// TIA Portal V20 export
// export: Created 2025-12-01T14:56:38.9745421Z, ExportSetting None, DisplayName Totally Integrated Automation Portal, DisplayVersion V20 Update 3, DisplayName TIA Portal Openness, DisplayVersion V20 Update 3, DisplayName TIA Portal Version Control Interface, DisplayVersion V20 Update 3, DisplayName STEP 7 Professional, DisplayVersion V20 Update 3, DisplayName STEP 7 Safety, DisplayVersion V20 Update 2, DisplayName WinCC Basic/Comfort/Advanced, DisplayVersion V20 Update 3, DisplayName WinCC Professional, DisplayVersion V20 Update 3, DisplayName WinCC Unified, DisplayVersion V20 Update 3
FUNCTION_BLOCK "FB41_Mesa_ApiladorDesApilador_E0E1E3_S0S1S3"   // FB41, LAD
TITLE = Control del Ramal de Salidas
{ S7_Optimized_Access := 'FALSE' }
AUTHOR : MESA_MAQ
NAME : 20160509
VERSION : 3.6
// stored: AutoNumber false, SetENOAutomatically false
   VAR_INPUT
      Mesa : UInt;   // Mesa de la FB
      Error_Tx : Bool;   // Error en el Tx
      EnTension : Bool;   // Existe Tension en la Mesa
      Termico_Tx : Bool;   // Proteccion del Tx
      pHsMx_Carretilla : Bool;   // Detector de Carretilla Presente
      pHsMx_1 : Bool;   // pHs de la Mesa (Para Entrada por E3)
      pHsMx_2 : Bool;   // pHs de la Mesa (Para Entrada por E1)
      pHsMx_PR1 : Bool;   // pHs de Protrusion de la Mesa. Nota: No existe >> ON
      pHsMx_PR3 : Bool;   // pHs de Protrusion de la Mesa. Nota: No existe >> ON
      Avance_Tx : Bool;   // Avance del Tx
      Retroceso_Tx : Bool;   // Retroceso del Tx
      TP1_Up : Bool;   // TP1 Arriba. Nota Movimiento E1 >> S3
      TP1_Down : Bool;   // TP1 Abajo. Nota Movimiento E1 >> S3
      EnMovimiento_TP1 : Bool;   // En movimiento el TP1
      MAnt_DescargaAct : Bool;   // E1 >> Mesa Anterior DescargaAct
      AVTF_MAnt_Mx : Bool;   // E1 >> Mesa Anterior AVTF
      P_Mens_MAnt_Mx : Bool;   // E1 >> Mesa Anterior P_Mens
      MAnt_ExistePila : Bool;   // E1 >> Mesa Anterior Existe Pila
      MSig_DescargaAct : Bool;   // E3 >> Mesa Anterior DescargaAct
      AVTF_MSig_Mx : Bool;   // E3 >> Mesa Anterior AVTF
      P_Mens_MSig_Mx : Bool;   // E3 >> Mesa Anterior P_Mens
      MSig_ExistePila : Bool;   // E3 >> Mesa Anterior Existe Pila
      PTF_Mx_MSig : Bool;   // S1 >> Mesa Siguiente PTF
      FTF_Mx_MSig : Bool;   // S1 >> Mesa Siguiente FTF
      PTF_Mx_MAnt : Bool;   // S3 >> Mesa Siguiente PTF
      FTF_Mx_MAnt : Bool;   // S3 >> Mesa Siguiente FTF
      MAnt_CargaAct : Bool;
      MSig_CargaAct : Bool;
      ConCarga_Apilador : Bool;   // Existe Carga >>> Interlock Maquina
      Quieto_Apilador : Bool;   // Quieto >>> Interlock Maquina
      Lleno_Apilador : Bool;   // Lleno >>> Interlock Maquina
      FinMovimiento_Apilador : Bool;   // Fin Movimiento >>> Interlock Maquina
      Mx_VelocidadLenta_In : Bool;   // Forzar a Velociada Lenta
      Mx_Centraje : Bool;   // Config Mx >>> Centrar la Entrada
      F_ENV_MENS_Mx : Bool;   // Fin de Envio de Mensaje
      OrdSal_Pila_Mx_MAnt : Bool;   // Orden de Salida por S1 >> Pila
      OrdSal_Paleta_Mx_MAnt : Bool;   // Orden de Salida por S1 >> Paleta
      OrdSal_Pila_Mx_MSig : Bool;   // Orden de Salida por S3 >> Pila
      OrdSal_Paleta_Mx_MSig : Bool;   // Orden de Salida por S3 >> Paleta
      OrdSal_S00 : Bool;   // Orden de Salida por S0
      V_CNT_pHsMx : Int := 1000;   // Valor de Presencia
      V_CNT_pHsMx_FTF : Int := 200;   // Valor para activar FTF. Nota: < = V_CNT_pHsMx.
      V_CNTSeg_pHsMx : Int := 2000;   // Valor de Seguriadad para Presencia
      V_Subir_TP_Min : Int := 2000;   // Valor Minimo para Subir Tope
      V_Bajar_TP_Max : Int := 4000;   // Valor Maximo para Bajar Tope
      V_CNT_PasoLenta : Int := 2000;   // Valor de Paso a Lenta
      V_CNT_ApHsMx : Int := 500;   // Valor de Ausencia
      V_CNTSeg_ApHsMx : Int := 2000;   // Valor de Seguriadad para Ausencia
      V_TMP_Entrada : Int := 5000;   // Valor de Entrada de Carga >> E0
      V_TMP_Retirar : Int := 5000;   // Valor de Retirada de Carga >> S0
      V_CNT_Centrado : Int := 1000;   // Valor de Centrado de Carga
      V_CNT_Reposo : Int := 1500;   // Valor de Reposo de Carga Nota: > Centrado
      V_TOut_Tx_Mx : Int := 30000;   // TimeOut de Entrada por E1
      V_TOut_TP { ExternalWritable := 'False'} : Int := 5000;   // TimeOut de Tope
      V_TMP_Protrusion : Int := 200;   // TMP de Protrusion
      V_CNT_PerdidapHs : Int := 1000;   // CNT de Perdida de pHs
   END_VAR
   VAR_OUTPUT
      P_EnvMens_PMx : Bool;   // Permiso de Enviar Mensaje de Presencia
      P_EnvMens_AMx : Bool;   // Permiso de Enviar Mensaje de Ausencia
      P_RecepOK_Mx : Bool;   // Recepcion OK
      PTF_MAnt_Mx : Bool;   // E1 >> Mesa Anterior PTF
      FTF_MAnt_Mx : Bool;   // E1 >> Mesa Anterior FTF
      PTF_MSig_Mx : Bool;   // E3 >> Mesa Anterior PTF
      FTF_MSig_Mx : Bool;   // E3 >> Mesa Anterior FTF
      AVTF_Mx_MAnt : Bool;   // S1 >> Mesa Siguiente AVTF
      P_Mens_Mx_MAnt : Bool;   // S1 >> Mesa Siguiente P_Mens
      AVTF_Mx_MSig : Bool;   // S3 >> Mesa Siguiente AVTF
      P_Mens_Mx_MSig : Bool;   // S3 >> Mesa Siguiente P_Mens
      PasarReposo_Apilador : Bool;   // Pasar a Reposo >>> Interlock Maquina
      CogerPila_Apilador : Bool;   // Coger la Pila >>> Interlock Maquina
      DispensarPaleta_Apilador : Bool;   // Dispensar Paleta >>> Interlock Maquina
      DispensarpPila_Apilador : Bool;   // Dispensar Pila >>> Interlock Maquina
   END_VAR
   VAR_IN_OUT
      StatusLleno_Apilador : Bool;   // Status Lleno >>> Interlock Maquina
      StatusSemiLleno_Apilador : Bool;   // Status SemiLleno >>> Interlock Maquina
      StatusVacio_Apilador : Bool;   // Status Vacio >>> Interlock Maquina
   END_VAR
   VAR
      Anular_prE1 : Bool;   // ???
      Anular_prS3 : Bool;   // ???
      Mx_ET00 : Bool;
      Mx_ET01 : Bool;
      Mx_ET02 : Bool;
      Mx_ET08 : Bool;
      Mx_ET09 : Bool;
      Mx_ET10 : Bool;
      Mx_ET11 : Bool;
      Mx_ET12 : Bool;
      Mx_ET110 : Bool;
      Mx_ET111 : Bool;
      Mx_ET210 : Bool;
      Mx_ET211 : Bool;
      Mx_ET40 : Bool;
      Mx_ET41 : Bool;
      Mx_ET42 : Bool;
      Mx_ET43 : Bool;
      Mx_ET140 : Bool;
      Mx_ET141 : Bool;
      Mx_ET50 : Bool;
      Mx_ET51 : Bool;
      Mx_ET52 : Bool;
      Mx_ET53 : Bool;
      Mx_ET150 : Bool;
      Mx_ET151 : Bool;
      Mx_ET250 : Bool;
      Mx_ET251 : Bool;
      Mx_ET90 : Bool;
      Mx_ET91 : Bool;
      Mx_ET190 : Bool;
      Mx_ET191 : Bool;
      Mx_ET192 : Bool;
      ProtocoloIniciado : Bool;   // Iniciado el Envio del Mensaje de Presencia
      CNT_pHsMx_FTF_OK : Bool;   // Enviar ya FTF
      Memoria_EnReposoMaquina : Bool;   // Memoria >> Maquina en Reposo
      Carga_MAnt_Mx : Bool;   // Operacion de Carga MAnt >>> Mx
      Carga_MSig_Mx : Bool;   // Operacion de Carga MSig >>> Mx
      Descarga_Mx_MAnt : Bool;   // Operacion de DesCarga Mx >>> MAnt
      Descarga_Mx_MSig : Bool;   // Operacion de DesCarga Ms >>> MSig
      ActivaDesCarga_Mx_MAnt : Bool;
      ActivaDesCarga_Mx_MSig : Bool;
      STAT_EnvMens_PMx : Bool;   // Interna >> Envio del Mensaje de Presencia
      STAT_EnvMens_AMx : Bool;   // Interna >> Envio de Mensaje de Ausencia
      STAT_FTF_MAnt_Mx : Bool;   // Interna >> FTF de MAnt >> Mx
      STAT_FTF_MSig_Mx : Bool;   // Interna >> FTF de MSig >> Mx
      STAT_AVTF_Mx_MAnt : Bool;   // Interna >> AVTF de Mx >> MAnt
      STAT_AVTF_Mx_MSig : Bool;   // Interna >> AVTF de Mx >> MSig
      STAT_PasarReposo : Bool;   // Interna >> Pasar a Reposo >> Maquina
      STAT_CogerPila : Bool;   // Interna >> Coger la Pila >> Maquina
      STAT_DispensarPaleta : Bool;   // Interna >> Dispensar Paleta >> Maquina
      STAT_DispensarPila : Bool;   // Interna >> Dispensar Pila >> Maquina
      CNT_pHsMx { S7_SetPoint := 'True'} : "FB910_CNT_UHS";   // CNT de la Presencia
      CNTSeg_pHsMx { S7_SetPoint := 'True'} : "FB910_CNT_UHS";   // CNT de Seguridad de la Presencia
      CNT_ApHsMx { S7_SetPoint := 'True'} : "FB910_CNT_UHS";   // CNT de la Ausencia
      CNTSeg_ApHsMx { S7_SetPoint := 'True'} : "FB910_CNT_UHS";   // CNT de Seguridad de la Ausencia
      TMP_Entrada { S7_SetPoint := 'True'} : "FB910_CNT_UHS";   // TMP de Entrada de Carga
      TMP_Retirar { S7_SetPoint := 'True'} : "FB910_CNT_UHS";   // TMP de Retirada de Carga
      CNT_Centrado { S7_SetPoint := 'True'} : "FB910_CNT_UHS";   // Contador de Centrado de Carga
      TMP_EnTension { S7_SetPoint := 'True'} : "FB910_CNT_UHS";
      TOut_Av_Mx { S7_SetPoint := 'True'} : "FB910_CNT_UHS";   // Time Out de Entrada de E1
      TOut_Rt_Mx { S7_SetPoint := 'True'} : "FB910_CNT_UHS";   // Time Out de Entrada de E3
      TOut_Subir_TP { S7_SetPoint := 'True'} : "FB910_CNT_UHS";   // Time Out de Subida del TP
      TOut_Bajar_TP { S7_SetPoint := 'True'} : "FB910_CNT_UHS";   // Time Out de Bajada del TP
      TMP_Protrusion { S7_SetPoint := 'True'} : "FB910_CNT_UHS";   // TMP de la Protrusion
      CNT_PerdidapHs { S7_SetPoint := 'True'} : "FB910_CNT_UHS";   // CNT de Perdida de pHs
   END_VAR
   VAR_TEMP
      EstadoZona : "EstadoZona";   // Estado de Zona de la Mesa
      EstadoVI : "EstadosMesa";   // Estado del Vehiculo Inteliguente de la Mesa
      ConfigFB : "UDT_ConfigFB";   // Configuracion de la FB de la Mesa
      V_Protrusion : Int;
      Mx_SinPresenciaEnReset : Bool;
      Aux_ET00 : Bool;
   END_VAR
   VAR_TEMP   // added for the SCL form of the ladder/FBD networks
      _w1 : Bool;
      _w2 : Bool;
   END_VAR
BEGIN

REGION Network 1: Inicializaciones Especiales
   // Nota: En esta mesa no se envia presencia en el reset  >>>    #Mx_SinPresenciaEnReset
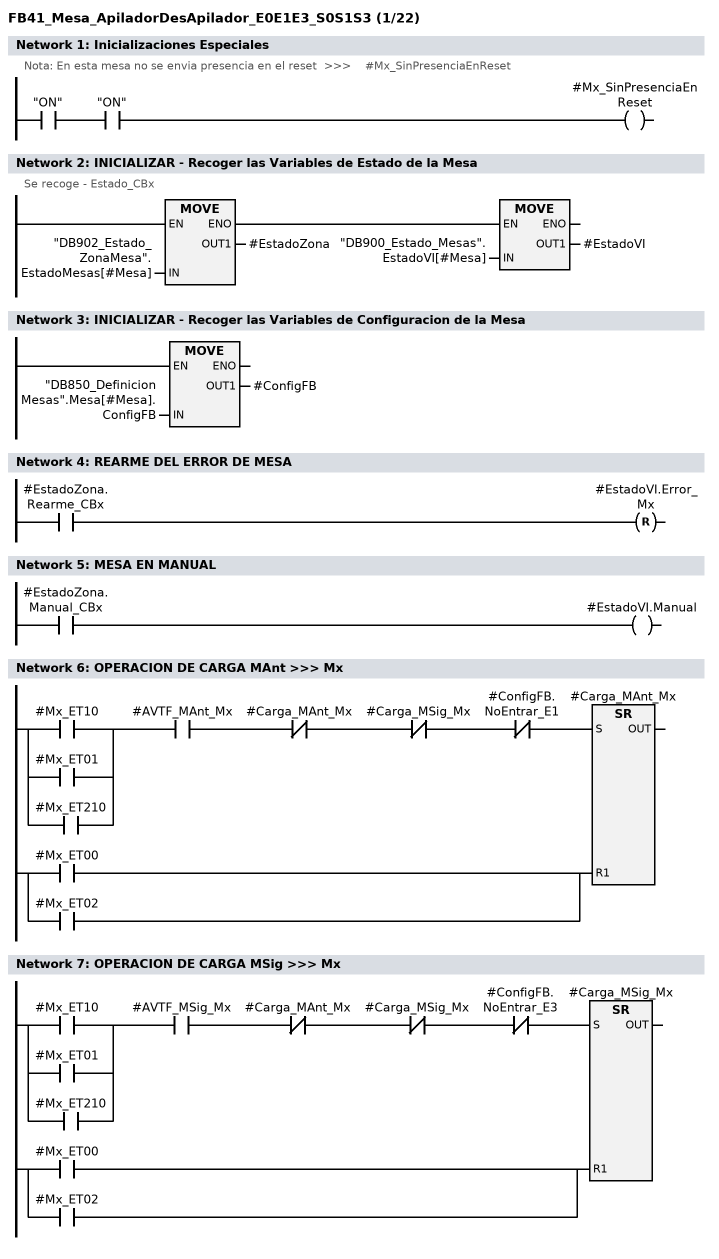
   RUNG wire#powerrail
      Contact( "ON" )
      Contact( "ON" )
      Coil( #Mx_SinPresenciaEnReset )
   END_RUNG
   // the same network as SCL:
   #Mx_SinPresenciaEnReset := "ON" AND "ON";
END_REGION

REGION Network 2: INICIALIZAR - Recoger las Variables de Estado de la Mesa
   // Se recoge - Estado_CBx
   RUNG wire#powerrail
      Move(in := "DB902_Estado_ZonaMesa".EstadoMesas[#Mesa], out1 => #EstadoZona)
      Move(in := "DB900_Estado_Mesas".EstadoVI[#Mesa], out1 => #EstadoVI)
   END_RUNG
   // the same network as SCL:
   #EstadoZona := "DB902_Estado_ZonaMesa".EstadoMesas[#Mesa];
   #EstadoVI := "DB900_Estado_Mesas".EstadoVI[#Mesa];
END_REGION

REGION Network 3: INICIALIZAR - Recoger las Variables de Configuracion de la Mesa
   RUNG wire#powerrail
      Move(in := "DB850_DefinicionMesas".Mesa[#Mesa].ConfigFB, out1 => #ConfigFB)
   END_RUNG
   // the same network as SCL:
   #ConfigFB := "DB850_DefinicionMesas".Mesa[#Mesa].ConfigFB;
END_REGION

REGION Network 4: REARME DEL ERROR DE MESA
   RUNG wire#powerrail
      Contact( #EstadoZona.Rearme_CBx )
      R_Coil( #EstadoVI.Error_Mx )
   END_RUNG
   // the same network as SCL:
   IF #EstadoZona.Rearme_CBx THEN #EstadoVI.Error_Mx := FALSE; END_IF;
END_REGION

REGION Network 5: MESA EN MANUAL
   RUNG wire#powerrail
      Contact( #EstadoZona.Manual_CBx )
      Coil( #EstadoVI.Manual )
   END_RUNG
   // the same network as SCL:
   #EstadoVI.Manual := #EstadoZona.Manual_CBx;
END_REGION

REGION Network 6: OPERACION DE CARGA MAnt >>> Mx
   RUNG wire#powerrail
      Contact( #Mx_ET10 )
      wire#w1
      Contact( #AVTF_MAnt_Mx )
      I_Contact( #Carga_MAnt_Mx )
      I_Contact( #Carga_MSig_Mx )
      I_Contact( #ConfigFB.NoEntrar_E1 )
      S_SR(operand := #Carga_MAnt_Mx, r1 := wire#w2)
   END_RUNG
   RUNG wire#powerrail
      Contact( #Mx_ET01 )
   END_RUNG wire#w1
   RUNG wire#powerrail
      Contact( #Mx_ET210 )
   END_RUNG wire#w1
   RUNG wire#powerrail
      Contact( #Mx_ET00 )
   END_RUNG wire#w2
   RUNG wire#powerrail
      Contact( #Mx_ET02 )
   END_RUNG wire#w2
   // the same network as SCL:
   IF (#Mx_ET10 OR #Mx_ET01 OR #Mx_ET210) AND #AVTF_MAnt_Mx AND NOT #Carga_MAnt_Mx AND NOT #Carga_MSig_Mx AND NOT #ConfigFB.NoEntrar_E1 THEN
       #Carga_MAnt_Mx := TRUE;   // SR flip-flop
   END_IF;
   IF #Mx_ET00 OR #Mx_ET02 THEN #Carga_MAnt_Mx := FALSE; END_IF;
END_REGION

REGION Network 7: OPERACION DE CARGA MSig >>> Mx
   RUNG wire#powerrail
      Contact( #Mx_ET10 )
      wire#w1
      Contact( #AVTF_MSig_Mx )
      I_Contact( #Carga_MAnt_Mx )
      I_Contact( #Carga_MSig_Mx )
      I_Contact( #ConfigFB.NoEntrar_E3 )
      S_SR(operand := #Carga_MSig_Mx, r1 := wire#w2)
   END_RUNG
   RUNG wire#powerrail
      Contact( #Mx_ET01 )
   END_RUNG wire#w1
   RUNG wire#powerrail
      Contact( #Mx_ET210 )
   END_RUNG wire#w1
   RUNG wire#powerrail
      Contact( #Mx_ET00 )
   END_RUNG wire#w2
   RUNG wire#powerrail
      Contact( #Mx_ET02 )
   END_RUNG wire#w2
   // the same network as SCL:
   IF (#Mx_ET10 OR #Mx_ET01 OR #Mx_ET210) AND #AVTF_MSig_Mx AND NOT #Carga_MAnt_Mx AND NOT #Carga_MSig_Mx AND NOT #ConfigFB.NoEntrar_E3 THEN
       #Carga_MSig_Mx := TRUE;   // SR flip-flop
   END_IF;
   IF #Mx_ET00 OR #Mx_ET02 THEN #Carga_MSig_Mx := FALSE; END_IF;
END_REGION

REGION Network 8: OPERACION DE DESCARGA Mx >>> MAnt
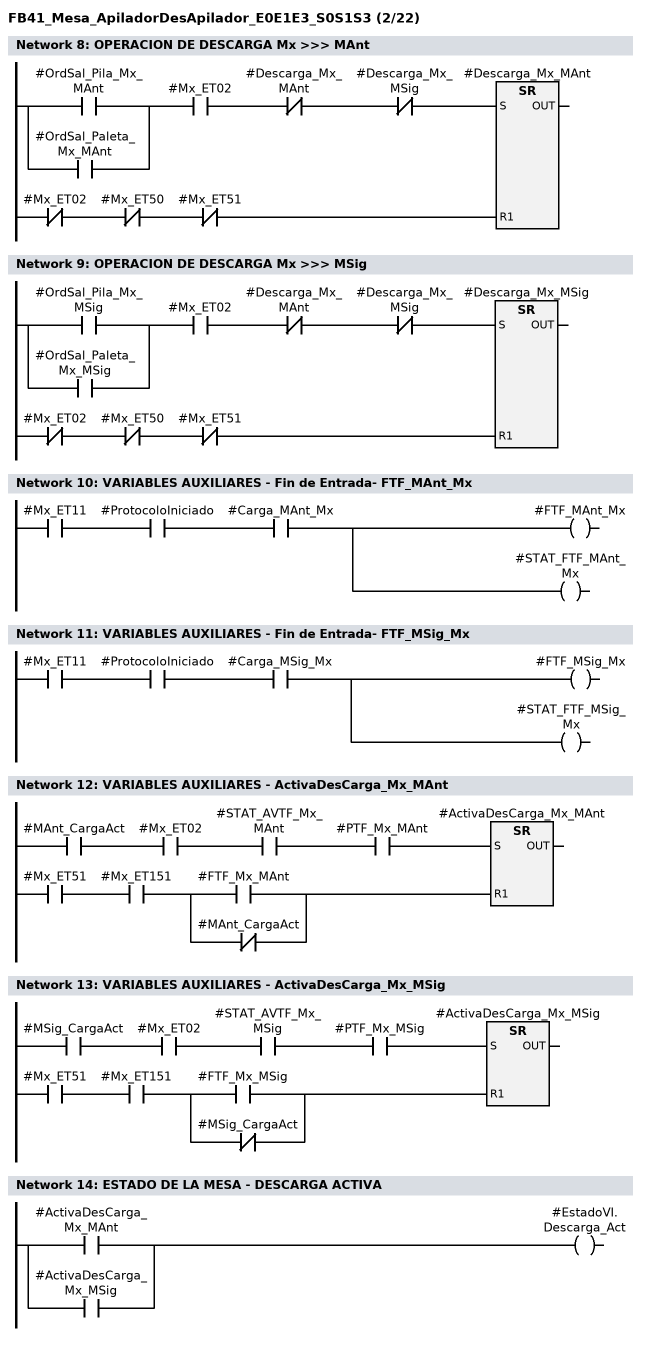
   RUNG wire#powerrail
      Contact( #OrdSal_Pila_Mx_MAnt )
      wire#w1
      Contact( #Mx_ET02 )
      I_Contact( #Descarga_Mx_MAnt )
      I_Contact( #Descarga_Mx_MSig )
      S_SR(operand := #Descarga_Mx_MAnt, r1 := wire#w2)
   END_RUNG
   RUNG wire#powerrail
      Contact( #OrdSal_Paleta_Mx_MAnt )
   END_RUNG wire#w1
   RUNG wire#powerrail
      I_Contact( #Mx_ET02 )
      I_Contact( #Mx_ET50 )
      I_Contact( #Mx_ET51 )
   END_RUNG wire#w2
   // the same network as SCL:
   IF (#OrdSal_Pila_Mx_MAnt OR #OrdSal_Paleta_Mx_MAnt) AND #Mx_ET02 AND NOT #Descarga_Mx_MAnt AND NOT #Descarga_Mx_MSig THEN
       #Descarga_Mx_MAnt := TRUE;   // SR flip-flop
   END_IF;
   IF NOT #Mx_ET02 AND NOT #Mx_ET50 AND NOT #Mx_ET51 THEN #Descarga_Mx_MAnt := FALSE; END_IF;
END_REGION

REGION Network 9: OPERACION DE DESCARGA Mx >>> MSig
   RUNG wire#powerrail
      Contact( #OrdSal_Pila_Mx_MSig )
      wire#w1
      Contact( #Mx_ET02 )
      I_Contact( #Descarga_Mx_MAnt )
      I_Contact( #Descarga_Mx_MSig )
      S_SR(operand := #Descarga_Mx_MSig, r1 := wire#w2)
   END_RUNG
   RUNG wire#powerrail
      Contact( #OrdSal_Paleta_Mx_MSig )
   END_RUNG wire#w1
   RUNG wire#powerrail
      I_Contact( #Mx_ET02 )
      I_Contact( #Mx_ET50 )
      I_Contact( #Mx_ET51 )
   END_RUNG wire#w2
   // the same network as SCL:
   IF (#OrdSal_Pila_Mx_MSig OR #OrdSal_Paleta_Mx_MSig) AND #Mx_ET02 AND NOT #Descarga_Mx_MAnt AND NOT #Descarga_Mx_MSig THEN
       #Descarga_Mx_MSig := TRUE;   // SR flip-flop
   END_IF;
   IF NOT #Mx_ET02 AND NOT #Mx_ET50 AND NOT #Mx_ET51 THEN #Descarga_Mx_MSig := FALSE; END_IF;
END_REGION

REGION Network 10: VARIABLES AUXILIARES - Fin de Entrada- FTF_MAnt_Mx
   RUNG wire#powerrail
      Contact( #Mx_ET11 )
      Contact( #ProtocoloIniciado )
      Contact( #Carga_MAnt_Mx )
      wire#w1
      Coil( #FTF_MAnt_Mx )
   END_RUNG
   RUNG wire#w1
      Coil( #STAT_FTF_MAnt_Mx )
   END_RUNG
   // the same network as SCL:
   #FTF_MAnt_Mx := #Mx_ET11 AND #ProtocoloIniciado AND #Carga_MAnt_Mx;
   #STAT_FTF_MAnt_Mx := #FTF_MAnt_Mx;
END_REGION

REGION Network 11: VARIABLES AUXILIARES - Fin de Entrada- FTF_MSig_Mx
   RUNG wire#powerrail
      Contact( #Mx_ET11 )
      Contact( #ProtocoloIniciado )
      Contact( #Carga_MSig_Mx )
      wire#w1
      Coil( #FTF_MSig_Mx )
   END_RUNG
   RUNG wire#w1
      Coil( #STAT_FTF_MSig_Mx )
   END_RUNG
   // the same network as SCL:
   #FTF_MSig_Mx := #Mx_ET11 AND #ProtocoloIniciado AND #Carga_MSig_Mx;
   #STAT_FTF_MSig_Mx := #FTF_MSig_Mx;
END_REGION

REGION Network 12: VARIABLES AUXILIARES - ActivaDesCarga_Mx_MAnt
   RUNG wire#powerrail
      Contact( #MAnt_CargaAct )
      Contact( #Mx_ET02 )
      Contact( #STAT_AVTF_Mx_MAnt )
      Contact( #PTF_Mx_MAnt )
      S_SR(operand := #ActivaDesCarga_Mx_MAnt, r1 := wire#w2)
   END_RUNG
   RUNG wire#powerrail
      Contact( #Mx_ET51 )
      Contact( #Mx_ET151 )
      wire#w1
      Contact( #FTF_Mx_MAnt )
   END_RUNG wire#w2
   RUNG wire#w1
      I_Contact( #MAnt_CargaAct )
   END_RUNG wire#w2
   // the same network as SCL:
   IF #MAnt_CargaAct AND #Mx_ET02 AND #STAT_AVTF_Mx_MAnt AND #PTF_Mx_MAnt THEN
       #ActivaDesCarga_Mx_MAnt := TRUE;   // SR flip-flop
   END_IF;
   IF #Mx_ET51 AND #Mx_ET151 AND (#FTF_Mx_MAnt OR NOT #MAnt_CargaAct) THEN
       #ActivaDesCarga_Mx_MAnt := FALSE;
   END_IF;
END_REGION

REGION Network 13: VARIABLES AUXILIARES - ActivaDesCarga_Mx_MSig
   RUNG wire#powerrail
      Contact( #MSig_CargaAct )
      Contact( #Mx_ET02 )
      Contact( #STAT_AVTF_Mx_MSig )
      Contact( #PTF_Mx_MSig )
      S_SR(operand := #ActivaDesCarga_Mx_MSig, r1 := wire#w2)
   END_RUNG
   RUNG wire#powerrail
      Contact( #Mx_ET51 )
      Contact( #Mx_ET151 )
      wire#w1
      Contact( #FTF_Mx_MSig )
   END_RUNG wire#w2
   RUNG wire#w1
      I_Contact( #MSig_CargaAct )
   END_RUNG wire#w2
   // the same network as SCL:
   IF #MSig_CargaAct AND #Mx_ET02 AND #STAT_AVTF_Mx_MSig AND #PTF_Mx_MSig THEN
       #ActivaDesCarga_Mx_MSig := TRUE;   // SR flip-flop
   END_IF;
   IF #Mx_ET51 AND #Mx_ET151 AND (#FTF_Mx_MSig OR NOT #MSig_CargaAct) THEN
       #ActivaDesCarga_Mx_MSig := FALSE;
   END_IF;
END_REGION

REGION Network 14: ESTADO DE LA MESA - DESCARGA ACTIVA
   RUNG wire#powerrail
      Contact( #ActivaDesCarga_Mx_MAnt )
      wire#w1
      Coil( #EstadoVI.Descarga_Act )
   END_RUNG
   RUNG wire#powerrail
      Contact( #ActivaDesCarga_Mx_MSig )
   END_RUNG wire#w1
   // the same network as SCL:
   #EstadoVI.Descarga_Act := #ActivaDesCarga_Mx_MAnt OR #ActivaDesCarga_Mx_MSig;
END_REGION

REGION Network 15: ET192 - CONTROL RETIRADA MESA - PROTOCOLO ORDEN
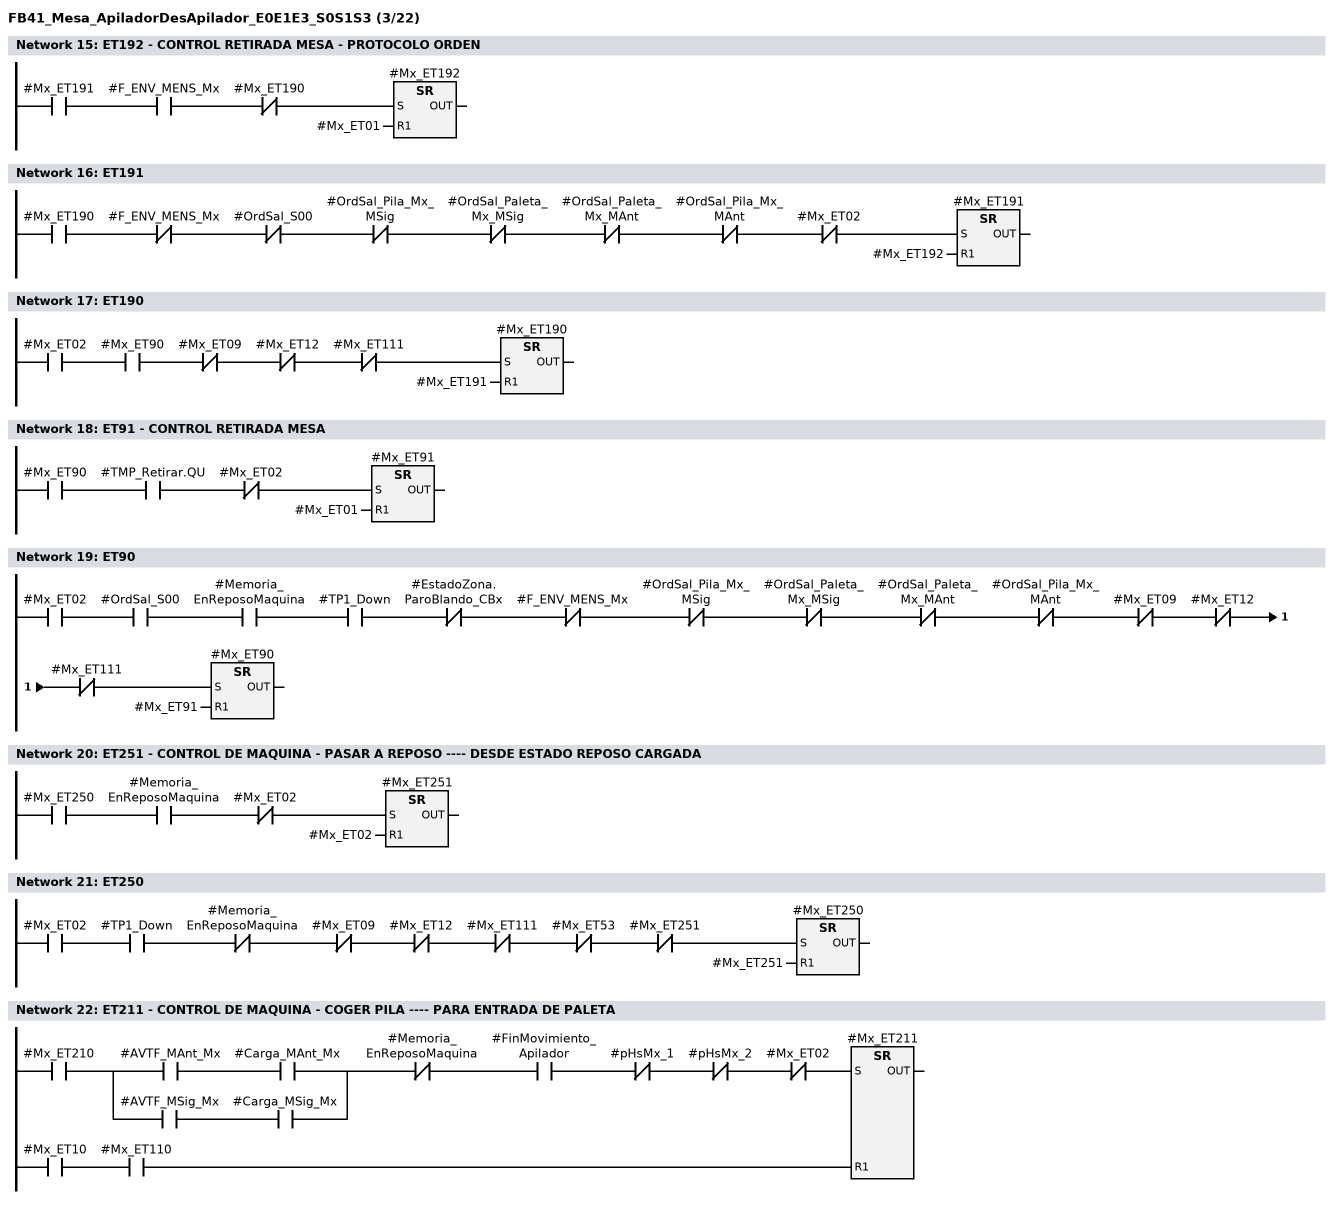
   RUNG wire#powerrail
      Contact( #Mx_ET191 )
      Contact( #F_ENV_MENS_Mx )
      I_Contact( #Mx_ET190 )
      S_SR(operand := #Mx_ET192, r1 := #Mx_ET01)
   END_RUNG
   // the same network as SCL:
   IF #Mx_ET191 AND #F_ENV_MENS_Mx AND NOT #Mx_ET190 THEN
       #Mx_ET192 := TRUE;   // SR flip-flop
   END_IF;
   IF #Mx_ET01 THEN #Mx_ET192 := FALSE; END_IF;
END_REGION

REGION Network 16: ET191
   RUNG wire#powerrail
      Contact( #Mx_ET190 )
      I_Contact( #F_ENV_MENS_Mx )
      I_Contact( #OrdSal_S00 )
      I_Contact( #OrdSal_Pila_Mx_MSig )
      I_Contact( #OrdSal_Paleta_Mx_MSig )
      I_Contact( #OrdSal_Paleta_Mx_MAnt )
      I_Contact( #OrdSal_Pila_Mx_MAnt )
      I_Contact( #Mx_ET02 )
      S_SR(operand := #Mx_ET191, r1 := #Mx_ET192)
   END_RUNG
   // the same network as SCL:
   IF #Mx_ET190 AND NOT #F_ENV_MENS_Mx AND NOT #OrdSal_S00 AND NOT #OrdSal_Pila_Mx_MSig AND NOT #OrdSal_Paleta_Mx_MSig AND NOT #OrdSal_Paleta_Mx_MAnt AND NOT #OrdSal_Pila_Mx_MAnt AND NOT #Mx_ET02 THEN
       #Mx_ET191 := TRUE;   // SR flip-flop
   END_IF;
   IF #Mx_ET192 THEN #Mx_ET191 := FALSE; END_IF;
END_REGION

REGION Network 17: ET190
   RUNG wire#powerrail
      Contact( #Mx_ET02 )
      Contact( #Mx_ET90 )
      I_Contact( #Mx_ET09 )
      I_Contact( #Mx_ET12 )
      I_Contact( #Mx_ET111 )
      S_SR(operand := #Mx_ET190, r1 := #Mx_ET191)
   END_RUNG
   // the same network as SCL:
   IF #Mx_ET02 AND #Mx_ET90 AND NOT #Mx_ET09 AND NOT #Mx_ET12 AND NOT #Mx_ET111 THEN
       #Mx_ET190 := TRUE;   // SR flip-flop
   END_IF;
   IF #Mx_ET191 THEN #Mx_ET190 := FALSE; END_IF;
END_REGION

REGION Network 18: ET91 - CONTROL RETIRADA MESA
   RUNG wire#powerrail
      Contact( #Mx_ET90 )
      Contact( #TMP_Retirar.QU )
      I_Contact( #Mx_ET02 )
      S_SR(operand := #Mx_ET91, r1 := #Mx_ET01)
   END_RUNG
   // the same network as SCL:
   IF #Mx_ET90 AND #TMP_Retirar.QU AND NOT #Mx_ET02 THEN
       #Mx_ET91 := TRUE;   // SR flip-flop
   END_IF;
   IF #Mx_ET01 THEN #Mx_ET91 := FALSE; END_IF;
END_REGION

REGION Network 19: ET90
   RUNG wire#powerrail
      Contact( #Mx_ET02 )
      Contact( #OrdSal_S00 )
      Contact( #Memoria_EnReposoMaquina )
      Contact( #TP1_Down )
      I_Contact( #EstadoZona.ParoBlando_CBx )
      I_Contact( #F_ENV_MENS_Mx )
      I_Contact( #OrdSal_Pila_Mx_MSig )
      I_Contact( #OrdSal_Paleta_Mx_MSig )
      I_Contact( #OrdSal_Paleta_Mx_MAnt )
      I_Contact( #OrdSal_Pila_Mx_MAnt )
      I_Contact( #Mx_ET09 )
      I_Contact( #Mx_ET12 )
      I_Contact( #Mx_ET111 )
      S_SR(operand := #Mx_ET90, r1 := #Mx_ET91)
   END_RUNG
   // the same network as SCL:
   IF #Mx_ET02 AND #OrdSal_S00 AND #Memoria_EnReposoMaquina AND #TP1_Down AND NOT #EstadoZona.ParoBlando_CBx AND NOT #F_ENV_MENS_Mx AND NOT #OrdSal_Pila_Mx_MSig AND NOT #OrdSal_Paleta_Mx_MSig AND NOT #OrdSal_Paleta_Mx_MAnt AND NOT #OrdSal_Pila_Mx_MAnt AND NOT #Mx_ET09 AND NOT #Mx_ET12 AND NOT #Mx_ET111 THEN
       #Mx_ET90 := TRUE;   // SR flip-flop
   END_IF;
   IF #Mx_ET91 THEN #Mx_ET90 := FALSE; END_IF;
END_REGION

REGION Network 20: ET251 - CONTROL DE MAQUINA - PASAR A REPOSO ---- DESDE ESTADO REPOSO CARGADA
   RUNG wire#powerrail
      Contact( #Mx_ET250 )
      Contact( #Memoria_EnReposoMaquina )
      I_Contact( #Mx_ET02 )
      S_SR(operand := #Mx_ET251, r1 := #Mx_ET02)
   END_RUNG
   // the same network as SCL:
   IF #Mx_ET250 AND #Memoria_EnReposoMaquina AND NOT #Mx_ET02 THEN
       #Mx_ET251 := TRUE;   // SR flip-flop
   END_IF;
   IF #Mx_ET02 THEN #Mx_ET251 := FALSE; END_IF;
END_REGION

REGION Network 21: ET250
   RUNG wire#powerrail
      Contact( #Mx_ET02 )
      Contact( #TP1_Down )
      I_Contact( #Memoria_EnReposoMaquina )
      I_Contact( #Mx_ET09 )
      I_Contact( #Mx_ET12 )
      I_Contact( #Mx_ET111 )
      I_Contact( #Mx_ET53 )
      I_Contact( #Mx_ET251 )
      S_SR(operand := #Mx_ET250, r1 := #Mx_ET251)
   END_RUNG
   // the same network as SCL:
   IF #Mx_ET02 AND #TP1_Down AND NOT #Memoria_EnReposoMaquina AND NOT #Mx_ET09 AND NOT #Mx_ET12 AND NOT #Mx_ET111 AND NOT #Mx_ET53 AND NOT #Mx_ET251 THEN
       #Mx_ET250 := TRUE;   // SR flip-flop
   END_IF;
   IF #Mx_ET251 THEN #Mx_ET250 := FALSE; END_IF;
END_REGION

REGION Network 22: ET211 - CONTROL DE MAQUINA - COGER PILA ---- PARA ENTRADA DE PALETA
   RUNG wire#powerrail
      Contact( #Mx_ET210 )
      wire#w1
      Contact( #AVTF_MAnt_Mx )
      Contact( #Carga_MAnt_Mx )
      wire#w2
      I_Contact( #Memoria_EnReposoMaquina )
      Contact( #FinMovimiento_Apilador )
      I_Contact( #pHsMx_1 )
      I_Contact( #pHsMx_2 )
      I_Contact( #Mx_ET02 )
      S_SR(operand := #Mx_ET211, r1 := wire#w3)
   END_RUNG
   RUNG wire#w1
      Contact( #AVTF_MSig_Mx )
      Contact( #Carga_MSig_Mx )
   END_RUNG wire#w2
   RUNG wire#powerrail
      Contact( #Mx_ET10 )
      Contact( #Mx_ET110 )
   END_RUNG wire#w3
   // the same network as SCL:
   IF #Mx_ET210 AND ((#AVTF_MAnt_Mx AND #Carga_MAnt_Mx) OR (#AVTF_MSig_Mx AND #Carga_MSig_Mx)) AND NOT #Memoria_EnReposoMaquina AND #FinMovimiento_Apilador AND NOT #pHsMx_1 AND NOT #pHsMx_2 AND NOT #Mx_ET02 THEN
       #Mx_ET211 := TRUE;   // SR flip-flop
   END_IF;
   IF #Mx_ET10 AND #Mx_ET110 THEN #Mx_ET211 := FALSE; END_IF;
END_REGION

REGION Network 23: ET210
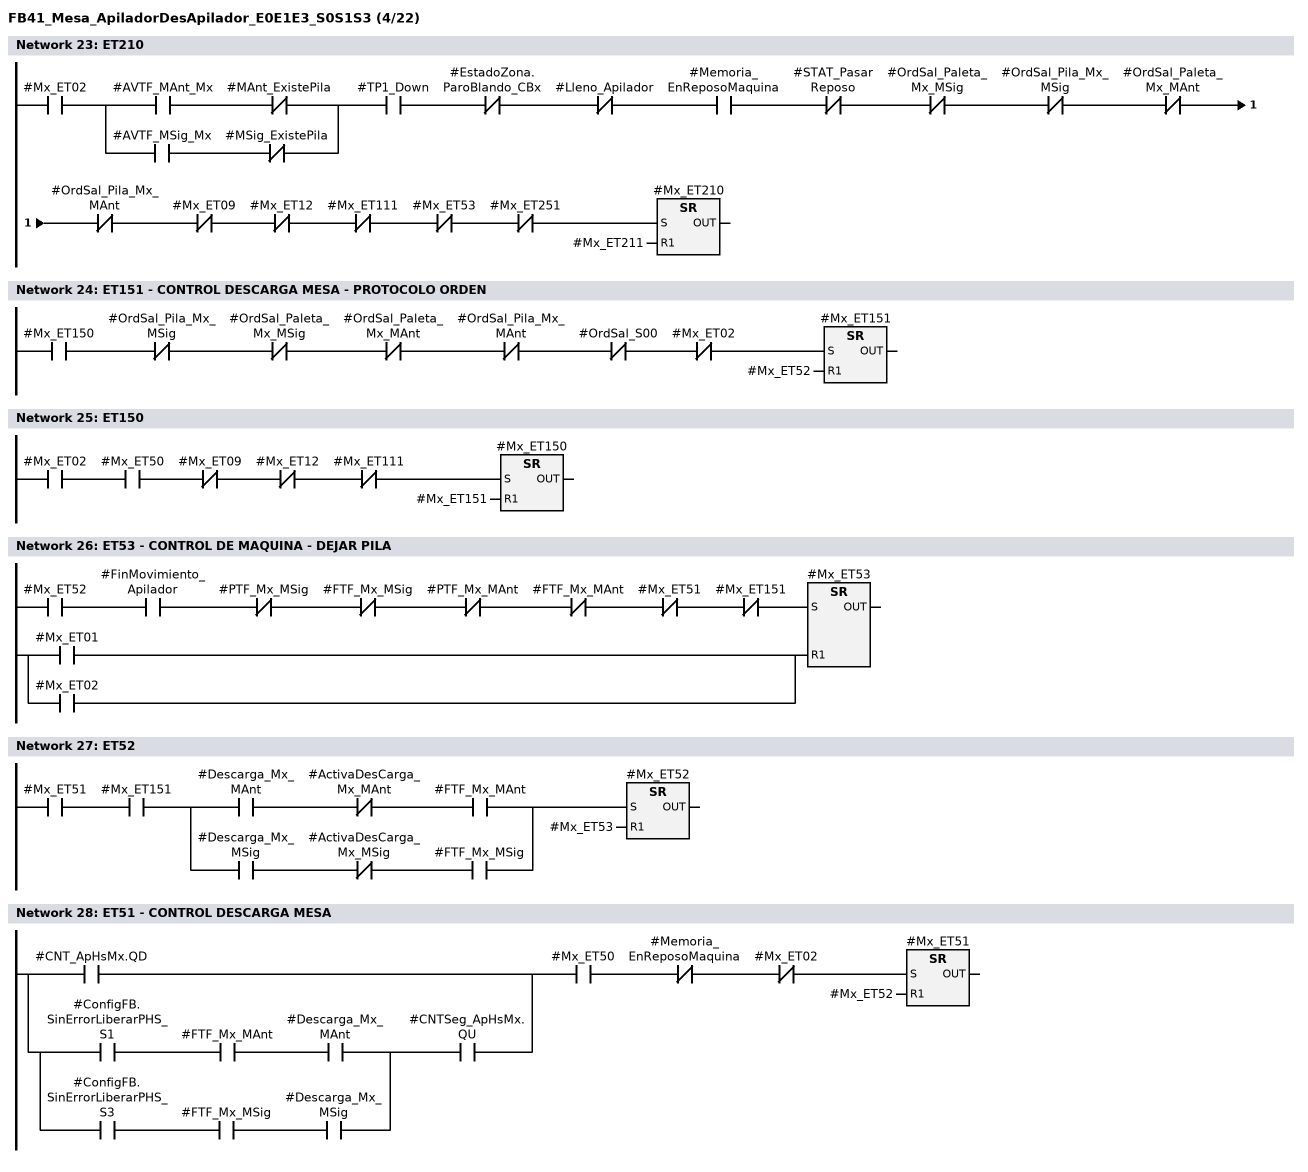
   RUNG wire#powerrail
      Contact( #Mx_ET02 )
      wire#w1
      Contact( #AVTF_MAnt_Mx )
      I_Contact( #MAnt_ExistePila )
      wire#w2
      Contact( #TP1_Down )
      I_Contact( #EstadoZona.ParoBlando_CBx )
      I_Contact( #Lleno_Apilador )
      Contact( #Memoria_EnReposoMaquina )
      I_Contact( #STAT_PasarReposo )
      I_Contact( #OrdSal_Paleta_Mx_MSig )
      I_Contact( #OrdSal_Pila_Mx_MSig )
      I_Contact( #OrdSal_Paleta_Mx_MAnt )
      I_Contact( #OrdSal_Pila_Mx_MAnt )
      I_Contact( #Mx_ET09 )
      I_Contact( #Mx_ET12 )
      I_Contact( #Mx_ET111 )
      I_Contact( #Mx_ET53 )
      I_Contact( #Mx_ET251 )
      S_SR(operand := #Mx_ET210, r1 := #Mx_ET211)
   END_RUNG
   RUNG wire#w1
      Contact( #AVTF_MSig_Mx )
      I_Contact( #MSig_ExistePila )
   END_RUNG wire#w2
   // the same network as SCL:
   IF #Mx_ET02 AND ((#AVTF_MAnt_Mx AND NOT #MAnt_ExistePila) OR (#AVTF_MSig_Mx AND NOT #MSig_ExistePila)) AND #TP1_Down AND NOT #EstadoZona.ParoBlando_CBx AND NOT #Lleno_Apilador AND #Memoria_EnReposoMaquina AND NOT #STAT_PasarReposo AND NOT #OrdSal_Paleta_Mx_MSig AND NOT #OrdSal_Pila_Mx_MSig AND NOT #OrdSal_Paleta_Mx_MAnt AND NOT #OrdSal_Pila_Mx_MAnt AND NOT #Mx_ET09 AND NOT #Mx_ET12 AND NOT #Mx_ET111 AND NOT #Mx_ET53 AND NOT #Mx_ET251 THEN
       #Mx_ET210 := TRUE;   // SR flip-flop
   END_IF;
   IF #Mx_ET211 THEN #Mx_ET210 := FALSE; END_IF;
END_REGION

REGION Network 24: ET151 - CONTROL DESCARGA MESA - PROTOCOLO ORDEN
   RUNG wire#powerrail
      Contact( #Mx_ET150 )
      I_Contact( #OrdSal_Pila_Mx_MSig )
      I_Contact( #OrdSal_Paleta_Mx_MSig )
      I_Contact( #OrdSal_Paleta_Mx_MAnt )
      I_Contact( #OrdSal_Pila_Mx_MAnt )
      I_Contact( #OrdSal_S00 )
      I_Contact( #Mx_ET02 )
      S_SR(operand := #Mx_ET151, r1 := #Mx_ET52)
   END_RUNG
   // the same network as SCL:
   IF #Mx_ET150 AND NOT #OrdSal_Pila_Mx_MSig AND NOT #OrdSal_Paleta_Mx_MSig AND NOT #OrdSal_Paleta_Mx_MAnt AND NOT #OrdSal_Pila_Mx_MAnt AND NOT #OrdSal_S00 AND NOT #Mx_ET02 THEN
       #Mx_ET151 := TRUE;   // SR flip-flop
   END_IF;
   IF #Mx_ET52 THEN #Mx_ET151 := FALSE; END_IF;
END_REGION

REGION Network 25: ET150
   RUNG wire#powerrail
      Contact( #Mx_ET02 )
      Contact( #Mx_ET50 )
      I_Contact( #Mx_ET09 )
      I_Contact( #Mx_ET12 )
      I_Contact( #Mx_ET111 )
      S_SR(operand := #Mx_ET150, r1 := #Mx_ET151)
   END_RUNG
   // the same network as SCL:
   IF #Mx_ET02 AND #Mx_ET50 AND NOT #Mx_ET09 AND NOT #Mx_ET12 AND NOT #Mx_ET111 THEN
       #Mx_ET150 := TRUE;   // SR flip-flop
   END_IF;
   IF #Mx_ET151 THEN #Mx_ET150 := FALSE; END_IF;
END_REGION

REGION Network 26: ET53 - CONTROL DE MAQUINA - DEJAR PILA
   RUNG wire#powerrail
      Contact( #Mx_ET52 )
      Contact( #FinMovimiento_Apilador )
      I_Contact( #PTF_Mx_MSig )
      I_Contact( #FTF_Mx_MSig )
      I_Contact( #PTF_Mx_MAnt )
      I_Contact( #FTF_Mx_MAnt )
      I_Contact( #Mx_ET51 )
      I_Contact( #Mx_ET151 )
      S_SR(operand := #Mx_ET53, r1 := wire#w1)
   END_RUNG
   RUNG wire#powerrail
      Contact( #Mx_ET01 )
   END_RUNG wire#w1
   RUNG wire#powerrail
      Contact( #Mx_ET02 )
   END_RUNG wire#w1
   // the same network as SCL:
   IF #Mx_ET52 AND #FinMovimiento_Apilador AND NOT #PTF_Mx_MSig AND NOT #FTF_Mx_MSig AND NOT #PTF_Mx_MAnt AND NOT #FTF_Mx_MAnt AND NOT #Mx_ET51 AND NOT #Mx_ET151 THEN
       #Mx_ET53 := TRUE;   // SR flip-flop
   END_IF;
   IF #Mx_ET01 OR #Mx_ET02 THEN #Mx_ET53 := FALSE; END_IF;
END_REGION

REGION Network 27: ET52
   RUNG wire#powerrail
      Contact( #Mx_ET51 )
      Contact( #Mx_ET151 )
      wire#w1
      Contact( #Descarga_Mx_MAnt )
      I_Contact( #ActivaDesCarga_Mx_MAnt )
      Contact( #FTF_Mx_MAnt )
      wire#w2
      S_SR(operand := #Mx_ET52, r1 := #Mx_ET53)
   END_RUNG
   RUNG wire#w1
      Contact( #Descarga_Mx_MSig )
      I_Contact( #ActivaDesCarga_Mx_MSig )
      Contact( #FTF_Mx_MSig )
   END_RUNG wire#w2
   // the same network as SCL:
   IF #Mx_ET51 AND #Mx_ET151 AND ((#Descarga_Mx_MAnt AND NOT #ActivaDesCarga_Mx_MAnt AND #FTF_Mx_MAnt) OR (#Descarga_Mx_MSig AND NOT #ActivaDesCarga_Mx_MSig AND #FTF_Mx_MSig)) THEN
       #Mx_ET52 := TRUE;   // SR flip-flop
   END_IF;
   IF #Mx_ET53 THEN #Mx_ET52 := FALSE; END_IF;
END_REGION

REGION Network 28: ET51 - CONTROL DESCARGA MESA
   RUNG wire#powerrail
      Contact( #CNT_ApHsMx.QD )
      wire#w1
      Contact( #Mx_ET50 )
      I_Contact( #Memoria_EnReposoMaquina )
      I_Contact( #Mx_ET02 )
      S_SR(operand := #Mx_ET51, r1 := #Mx_ET52)
   END_RUNG
   RUNG wire#powerrail
      Contact( #ConfigFB.SinErrorLiberarPHS_S1 )
      Contact( #FTF_Mx_MAnt )
      Contact( #Descarga_Mx_MAnt )
      wire#w2
      Contact( #CNTSeg_ApHsMx.QU )
   END_RUNG wire#w1
   RUNG wire#powerrail
      Contact( #ConfigFB.SinErrorLiberarPHS_S3 )
      Contact( #FTF_Mx_MSig )
      Contact( #Descarga_Mx_MSig )
   END_RUNG wire#w2
   // the same network as SCL:
   IF (#CNT_ApHsMx.QD OR (((#ConfigFB.SinErrorLiberarPHS_S1 AND #FTF_Mx_MAnt AND #Descarga_Mx_MAnt) OR (#ConfigFB.SinErrorLiberarPHS_S3 AND #FTF_Mx_MSig AND #Descarga_Mx_MSig)) AND #CNTSeg_ApHsMx.QU)) AND #Mx_ET50 AND NOT #Memoria_EnReposoMaquina AND NOT #Mx_ET02 THEN
       #Mx_ET51 := TRUE;   // SR flip-flop
   END_IF;
   IF #Mx_ET52 THEN #Mx_ET51 := FALSE; END_IF;
END_REGION

REGION Network 29: ET50
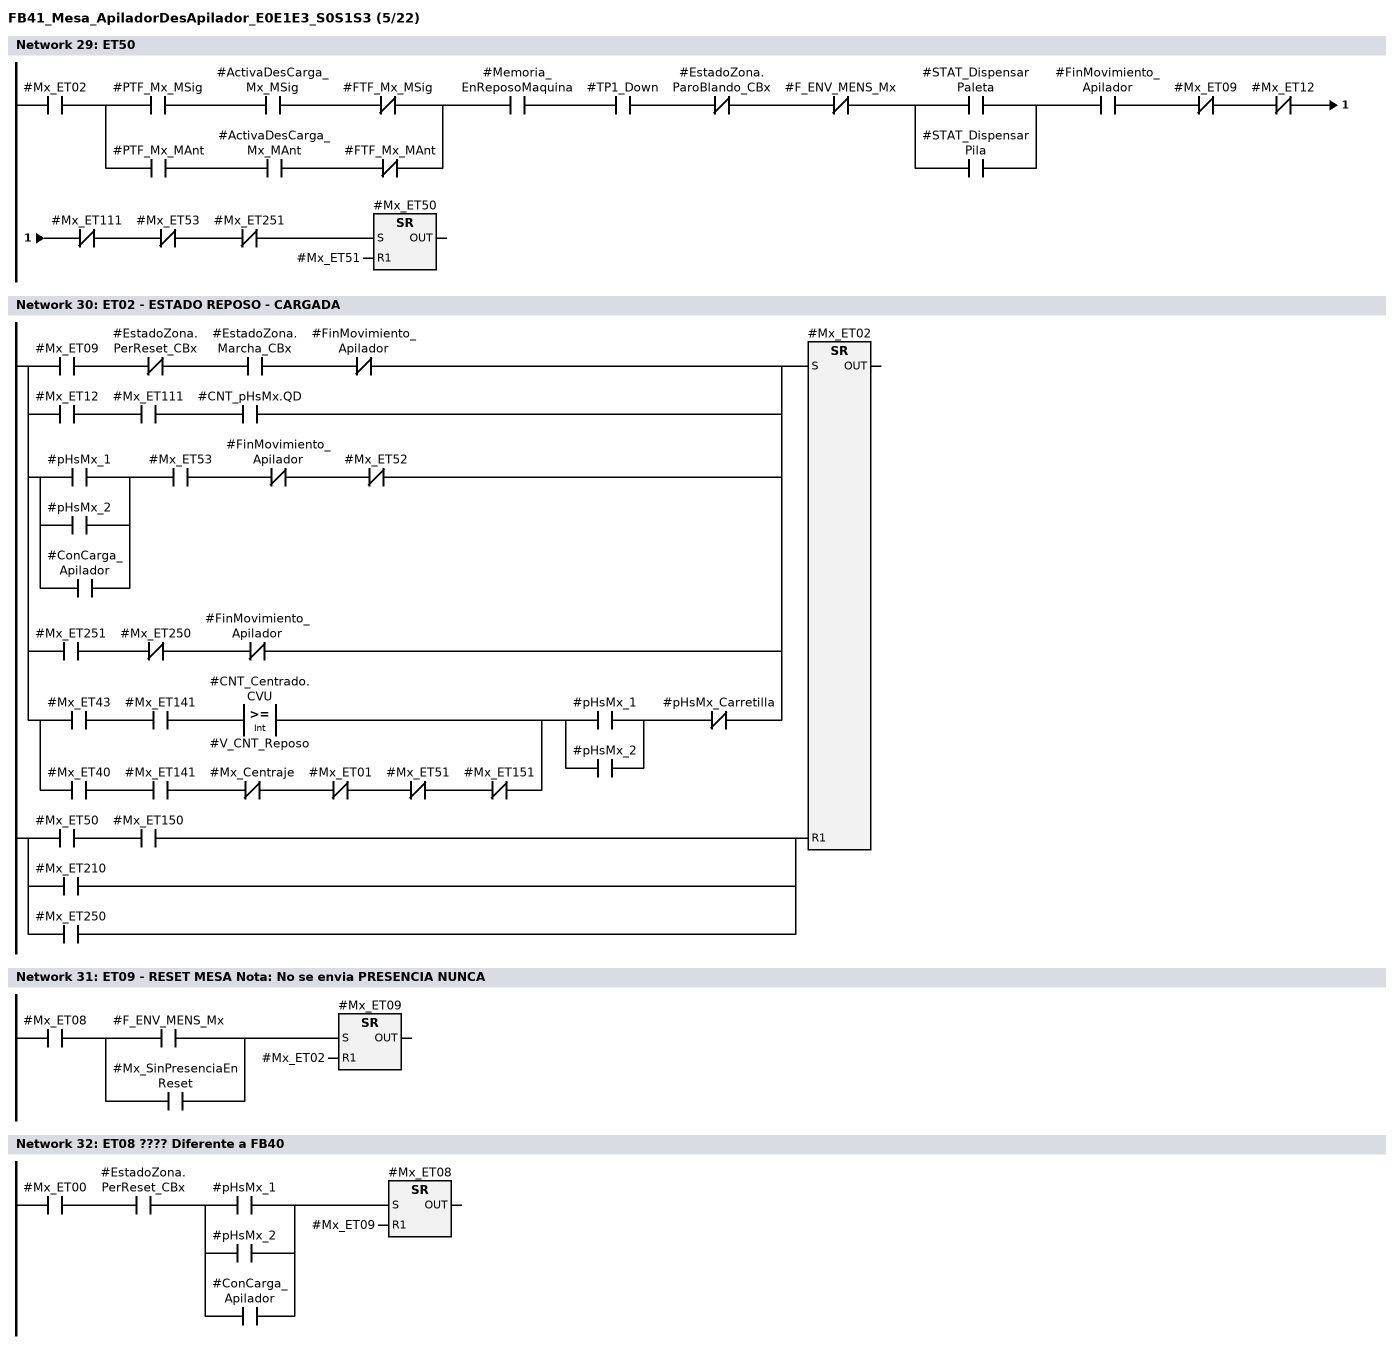
   RUNG wire#powerrail
      Contact( #Mx_ET02 )
      wire#w1
      Contact( #PTF_Mx_MSig )
      Contact( #ActivaDesCarga_Mx_MSig )
      I_Contact( #FTF_Mx_MSig )
      wire#w2
      Contact( #Memoria_EnReposoMaquina )
      Contact( #TP1_Down )
      I_Contact( #EstadoZona.ParoBlando_CBx )
      I_Contact( #F_ENV_MENS_Mx )
      wire#w3
      Contact( #STAT_DispensarPaleta )
      wire#w4
      Contact( #FinMovimiento_Apilador )
      I_Contact( #Mx_ET09 )
      I_Contact( #Mx_ET12 )
      I_Contact( #Mx_ET111 )
      I_Contact( #Mx_ET53 )
      I_Contact( #Mx_ET251 )
      S_SR(operand := #Mx_ET50, r1 := #Mx_ET51)
   END_RUNG
   RUNG wire#w1
      Contact( #PTF_Mx_MAnt )
      Contact( #ActivaDesCarga_Mx_MAnt )
      I_Contact( #FTF_Mx_MAnt )
   END_RUNG wire#w2
   RUNG wire#w3
      Contact( #STAT_DispensarPila )
   END_RUNG wire#w4
   // the same network as SCL:
   IF #Mx_ET02 AND ((#PTF_Mx_MSig AND #ActivaDesCarga_Mx_MSig AND NOT #FTF_Mx_MSig) OR (#PTF_Mx_MAnt AND #ActivaDesCarga_Mx_MAnt AND NOT #FTF_Mx_MAnt)) AND #Memoria_EnReposoMaquina AND #TP1_Down AND NOT #EstadoZona.ParoBlando_CBx AND NOT #F_ENV_MENS_Mx AND (#STAT_DispensarPaleta OR #STAT_DispensarPila) AND #FinMovimiento_Apilador AND NOT #Mx_ET09 AND NOT #Mx_ET12 AND NOT #Mx_ET111 AND NOT #Mx_ET53 AND NOT #Mx_ET251 THEN
       #Mx_ET50 := TRUE;   // SR flip-flop
   END_IF;
   IF #Mx_ET51 THEN #Mx_ET50 := FALSE; END_IF;
END_REGION

REGION Network 30: ET02 - ESTADO REPOSO - CARGADA
   RUNG wire#powerrail
      Contact( #Mx_ET09 )
      I_Contact( #EstadoZona.PerReset_CBx )
      Contact( #EstadoZona.Marcha_CBx )
      I_Contact( #FinMovimiento_Apilador )
      wire#w1
      S_SR(operand := #Mx_ET02, r1 := wire#w5)
   END_RUNG
   RUNG wire#powerrail
      Contact( #Mx_ET12 )
      Contact( #Mx_ET111 )
      Contact( #CNT_pHsMx.QD )
   END_RUNG wire#w1
   RUNG wire#powerrail
      Contact( #pHsMx_1 )
      wire#w2
      Contact( #Mx_ET53 )
      I_Contact( #FinMovimiento_Apilador )
      I_Contact( #Mx_ET52 )
   END_RUNG wire#w1
   RUNG wire#powerrail
      Contact( #pHsMx_2 )
   END_RUNG wire#w2
   RUNG wire#powerrail
      Contact( #ConCarga_Apilador )
   END_RUNG wire#w2
   RUNG wire#powerrail
      Contact( #Mx_ET251 )
      I_Contact( #Mx_ET250 )
      I_Contact( #FinMovimiento_Apilador )
   END_RUNG wire#w1
   RUNG wire#powerrail
      Contact( #Mx_ET43 )
      Contact( #Mx_ET141 )
      { S7_Templates := "SrcType := Int" } GE_Contact(in1 := #CNT_Centrado.CVU, in2 := #V_CNT_Reposo)
      wire#w3
      Contact( #pHsMx_1 )
      wire#w4
      I_Contact( #pHsMx_Carretilla )
   END_RUNG wire#w1
   RUNG wire#powerrail
      Contact( #Mx_ET40 )
      Contact( #Mx_ET141 )
      I_Contact( #Mx_Centraje )
      I_Contact( #Mx_ET01 )
      I_Contact( #Mx_ET51 )
      I_Contact( #Mx_ET151 )
   END_RUNG wire#w3
   RUNG wire#w3
      Contact( #pHsMx_2 )
   END_RUNG wire#w4
   RUNG wire#powerrail
      Contact( #Mx_ET50 )
      Contact( #Mx_ET150 )
   END_RUNG wire#w5
   RUNG wire#powerrail
      Contact( #Mx_ET210 )
   END_RUNG wire#w5
   RUNG wire#powerrail
      Contact( #Mx_ET250 )
   END_RUNG wire#w5
   // the same network as SCL:
   IF (#Mx_ET09 AND NOT #EstadoZona.PerReset_CBx AND #EstadoZona.Marcha_CBx AND NOT #FinMovimiento_Apilador) OR (#Mx_ET12 AND #Mx_ET111 AND #CNT_pHsMx.QD) OR ((#pHsMx_1 OR #pHsMx_2 OR #ConCarga_Apilador) AND #Mx_ET53 AND NOT #FinMovimiento_Apilador AND NOT #Mx_ET52) OR (#Mx_ET251 AND NOT #Mx_ET250 AND NOT #FinMovimiento_Apilador) OR (((#Mx_ET43 AND #Mx_ET141 AND (#CNT_Centrado.CVU >= #V_CNT_Reposo)) OR (#Mx_ET40 AND #Mx_ET141 AND NOT #Mx_Centraje AND NOT #Mx_ET01 AND NOT #Mx_ET51 AND NOT #Mx_ET151)) AND (#pHsMx_1 OR #pHsMx_2) AND NOT #pHsMx_Carretilla) THEN
       #Mx_ET02 := TRUE;   // SR flip-flop
   END_IF;
   IF (#Mx_ET50 AND #Mx_ET150) OR #Mx_ET210 OR #Mx_ET250 THEN #Mx_ET02 := FALSE; END_IF;
END_REGION

REGION Network 31: ET09 - RESET MESA Nota: No se envia PRESENCIA NUNCA
   RUNG wire#powerrail
      Contact( #Mx_ET08 )
      wire#w1
      Contact( #F_ENV_MENS_Mx )
      wire#w2
      S_SR(operand := #Mx_ET09, r1 := #Mx_ET02)
   END_RUNG
   RUNG wire#w1
      Contact( #Mx_SinPresenciaEnReset )
   END_RUNG wire#w2
   // the same network as SCL:
   IF #Mx_ET08 AND (#F_ENV_MENS_Mx OR #Mx_SinPresenciaEnReset) THEN
       #Mx_ET09 := TRUE;   // SR flip-flop
   END_IF;
   IF #Mx_ET02 THEN #Mx_ET09 := FALSE; END_IF;
END_REGION

REGION Network 32: ET08 ???? Diferente a FB40
   RUNG wire#powerrail
      Contact( #Mx_ET00 )
      Contact( #EstadoZona.PerReset_CBx )
      wire#w1
      Contact( #pHsMx_1 )
      wire#w2
      S_SR(operand := #Mx_ET08, r1 := #Mx_ET09)
   END_RUNG
   RUNG wire#w1
      Contact( #pHsMx_2 )
   END_RUNG wire#w2
   RUNG wire#w1
      Contact( #ConCarga_Apilador )
   END_RUNG wire#w2
   // the same network as SCL:
   IF #Mx_ET00 AND #EstadoZona.PerReset_CBx AND (#pHsMx_1 OR #pHsMx_2 OR #ConCarga_Apilador) THEN
       #Mx_ET08 := TRUE;   // SR flip-flop
   END_IF;
   IF #Mx_ET09 THEN #Mx_ET08 := FALSE; END_IF;
END_REGION

REGION Network 33: ET141 - CONTROL ENTRADA MESA - MENSAJE DE PRESENCIA
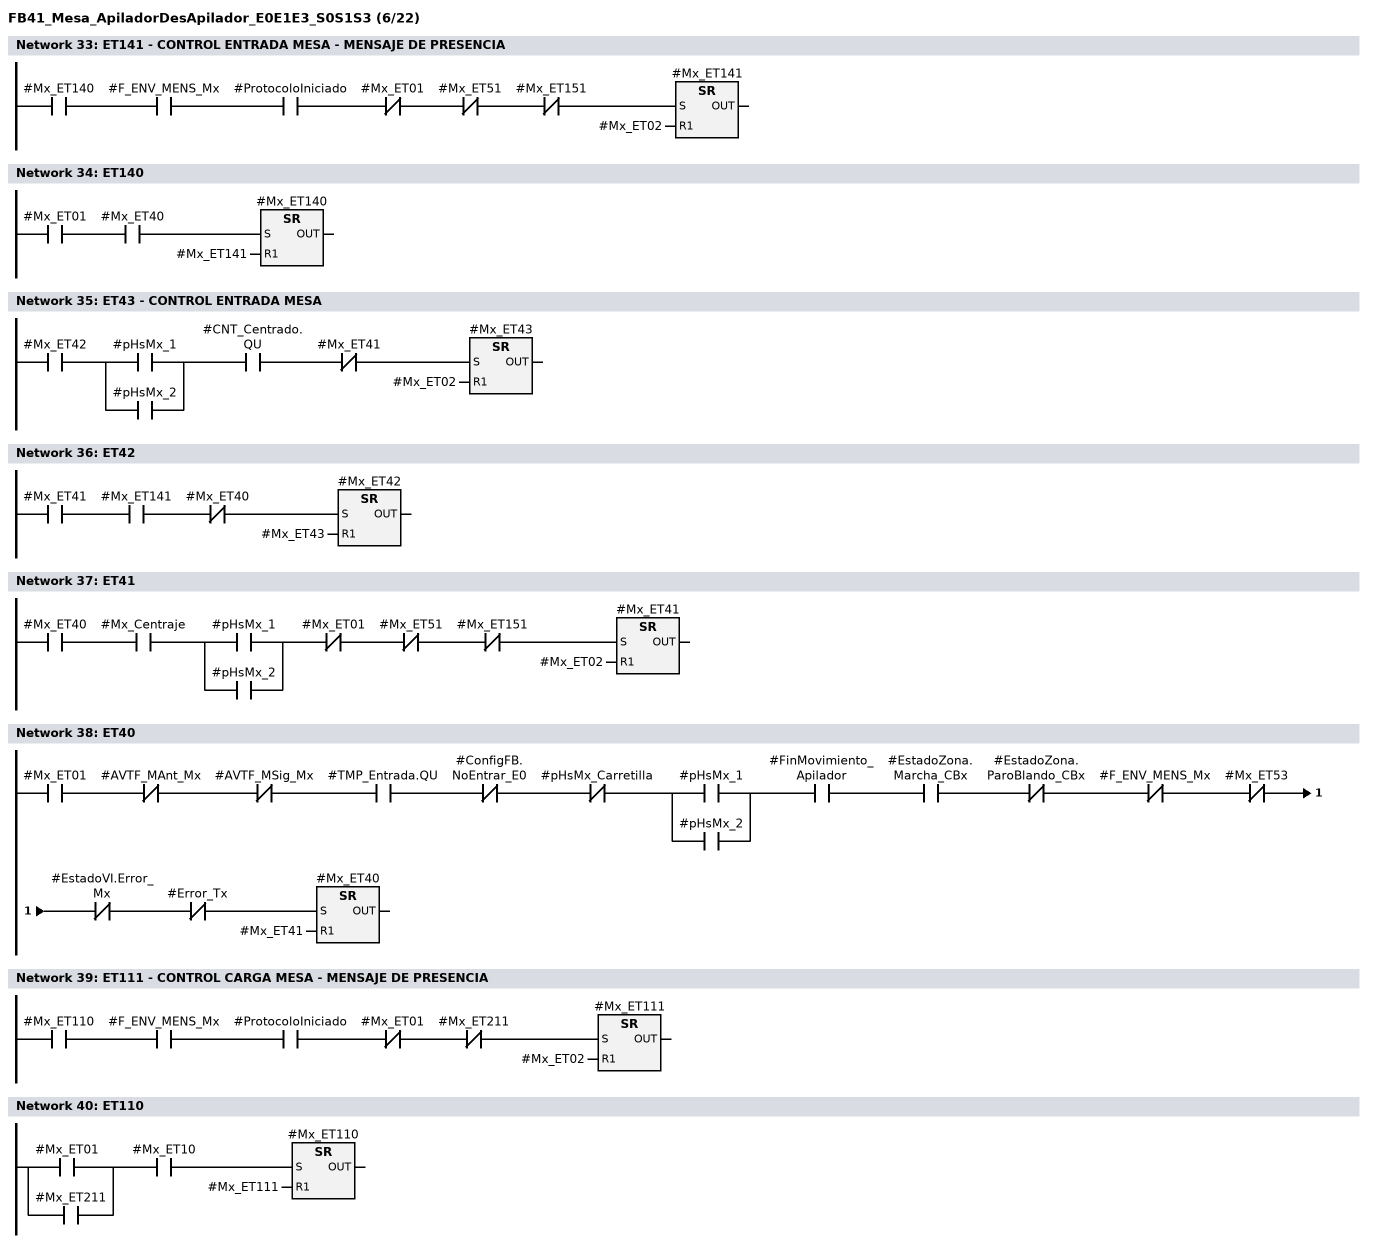
   RUNG wire#powerrail
      Contact( #Mx_ET140 )
      Contact( #F_ENV_MENS_Mx )
      Contact( #ProtocoloIniciado )
      I_Contact( #Mx_ET01 )
      I_Contact( #Mx_ET51 )
      I_Contact( #Mx_ET151 )
      S_SR(operand := #Mx_ET141, r1 := #Mx_ET02)
   END_RUNG
   // the same network as SCL:
   IF #Mx_ET140 AND #F_ENV_MENS_Mx AND #ProtocoloIniciado AND NOT #Mx_ET01 AND NOT #Mx_ET51 AND NOT #Mx_ET151 THEN
       #Mx_ET141 := TRUE;   // SR flip-flop
   END_IF;
   IF #Mx_ET02 THEN #Mx_ET141 := FALSE; END_IF;
END_REGION

REGION Network 34: ET140
   RUNG wire#powerrail
      Contact( #Mx_ET01 )
      Contact( #Mx_ET40 )
      S_SR(operand := #Mx_ET140, r1 := #Mx_ET141)
   END_RUNG
   // the same network as SCL:
   IF #Mx_ET01 AND #Mx_ET40 THEN
       #Mx_ET140 := TRUE;   // SR flip-flop
   END_IF;
   IF #Mx_ET141 THEN #Mx_ET140 := FALSE; END_IF;
END_REGION

REGION Network 35: ET43 - CONTROL ENTRADA MESA
   RUNG wire#powerrail
      Contact( #Mx_ET42 )
      wire#w1
      Contact( #pHsMx_1 )
      wire#w2
      Contact( #CNT_Centrado.QU )
      I_Contact( #Mx_ET41 )
      S_SR(operand := #Mx_ET43, r1 := #Mx_ET02)
   END_RUNG
   RUNG wire#w1
      Contact( #pHsMx_2 )
   END_RUNG wire#w2
   // the same network as SCL:
   IF #Mx_ET42 AND (#pHsMx_1 OR #pHsMx_2) AND #CNT_Centrado.QU AND NOT #Mx_ET41 THEN
       #Mx_ET43 := TRUE;   // SR flip-flop
   END_IF;
   IF #Mx_ET02 THEN #Mx_ET43 := FALSE; END_IF;
END_REGION

REGION Network 36: ET42
   RUNG wire#powerrail
      Contact( #Mx_ET41 )
      Contact( #Mx_ET141 )
      I_Contact( #Mx_ET40 )
      S_SR(operand := #Mx_ET42, r1 := #Mx_ET43)
   END_RUNG
   // the same network as SCL:
   IF #Mx_ET41 AND #Mx_ET141 AND NOT #Mx_ET40 THEN
       #Mx_ET42 := TRUE;   // SR flip-flop
   END_IF;
   IF #Mx_ET43 THEN #Mx_ET42 := FALSE; END_IF;
END_REGION

REGION Network 37: ET41
   RUNG wire#powerrail
      Contact( #Mx_ET40 )
      Contact( #Mx_Centraje )
      wire#w1
      Contact( #pHsMx_1 )
      wire#w2
      I_Contact( #Mx_ET01 )
      I_Contact( #Mx_ET51 )
      I_Contact( #Mx_ET151 )
      S_SR(operand := #Mx_ET41, r1 := #Mx_ET02)
   END_RUNG
   RUNG wire#w1
      Contact( #pHsMx_2 )
   END_RUNG wire#w2
   // the same network as SCL:
   IF #Mx_ET40 AND #Mx_Centraje AND (#pHsMx_1 OR #pHsMx_2) AND NOT #Mx_ET01 AND NOT #Mx_ET51 AND NOT #Mx_ET151 THEN
       #Mx_ET41 := TRUE;   // SR flip-flop
   END_IF;
   IF #Mx_ET02 THEN #Mx_ET41 := FALSE; END_IF;
END_REGION

REGION Network 38: ET40
   RUNG wire#powerrail
      Contact( #Mx_ET01 )
      I_Contact( #AVTF_MAnt_Mx )
      I_Contact( #AVTF_MSig_Mx )
      Contact( #TMP_Entrada.QU )
      I_Contact( #ConfigFB.NoEntrar_E0 )
      I_Contact( #pHsMx_Carretilla )
      wire#w1
      Contact( #pHsMx_1 )
      wire#w2
      Contact( #FinMovimiento_Apilador )
      Contact( #EstadoZona.Marcha_CBx )
      I_Contact( #EstadoZona.ParoBlando_CBx )
      I_Contact( #F_ENV_MENS_Mx )
      I_Contact( #Mx_ET53 )
      I_Contact( #EstadoVI.Error_Mx )
      I_Contact( #Error_Tx )
      S_SR(operand := #Mx_ET40, r1 := #Mx_ET41)
   END_RUNG
   RUNG wire#w1
      Contact( #pHsMx_2 )
   END_RUNG wire#w2
   // the same network as SCL:
   IF #Mx_ET01 AND NOT #AVTF_MAnt_Mx AND NOT #AVTF_MSig_Mx AND #TMP_Entrada.QU AND NOT #ConfigFB.NoEntrar_E0 AND NOT #pHsMx_Carretilla AND (#pHsMx_1 OR #pHsMx_2) AND #FinMovimiento_Apilador AND #EstadoZona.Marcha_CBx AND NOT #EstadoZona.ParoBlando_CBx AND NOT #F_ENV_MENS_Mx AND NOT #Mx_ET53 AND NOT #EstadoVI.Error_Mx AND NOT #Error_Tx THEN
       #Mx_ET40 := TRUE;   // SR flip-flop
   END_IF;
   IF #Mx_ET41 THEN #Mx_ET40 := FALSE; END_IF;
END_REGION

REGION Network 39: ET111 - CONTROL CARGA MESA - MENSAJE DE PRESENCIA
   RUNG wire#powerrail
      Contact( #Mx_ET110 )
      Contact( #F_ENV_MENS_Mx )
      Contact( #ProtocoloIniciado )
      I_Contact( #Mx_ET01 )
      I_Contact( #Mx_ET211 )
      S_SR(operand := #Mx_ET111, r1 := #Mx_ET02)
   END_RUNG
   // the same network as SCL:
   IF #Mx_ET110 AND #F_ENV_MENS_Mx AND #ProtocoloIniciado AND NOT #Mx_ET01 AND NOT #Mx_ET211 THEN
       #Mx_ET111 := TRUE;   // SR flip-flop
   END_IF;
   IF #Mx_ET02 THEN #Mx_ET111 := FALSE; END_IF;
END_REGION

REGION Network 40: ET110
   RUNG wire#powerrail
      Contact( #Mx_ET01 )
      wire#w1
      Contact( #Mx_ET10 )
      S_SR(operand := #Mx_ET110, r1 := #Mx_ET111)
   END_RUNG
   RUNG wire#powerrail
      Contact( #Mx_ET211 )
   END_RUNG wire#w1
   // the same network as SCL:
   IF (#Mx_ET01 OR #Mx_ET211) AND #Mx_ET10 THEN
       #Mx_ET110 := TRUE;   // SR flip-flop
   END_IF;
   IF #Mx_ET111 THEN #Mx_ET110 := FALSE; END_IF;
END_REGION

REGION Network 41: ET12 - CONTROL CARGA MESA
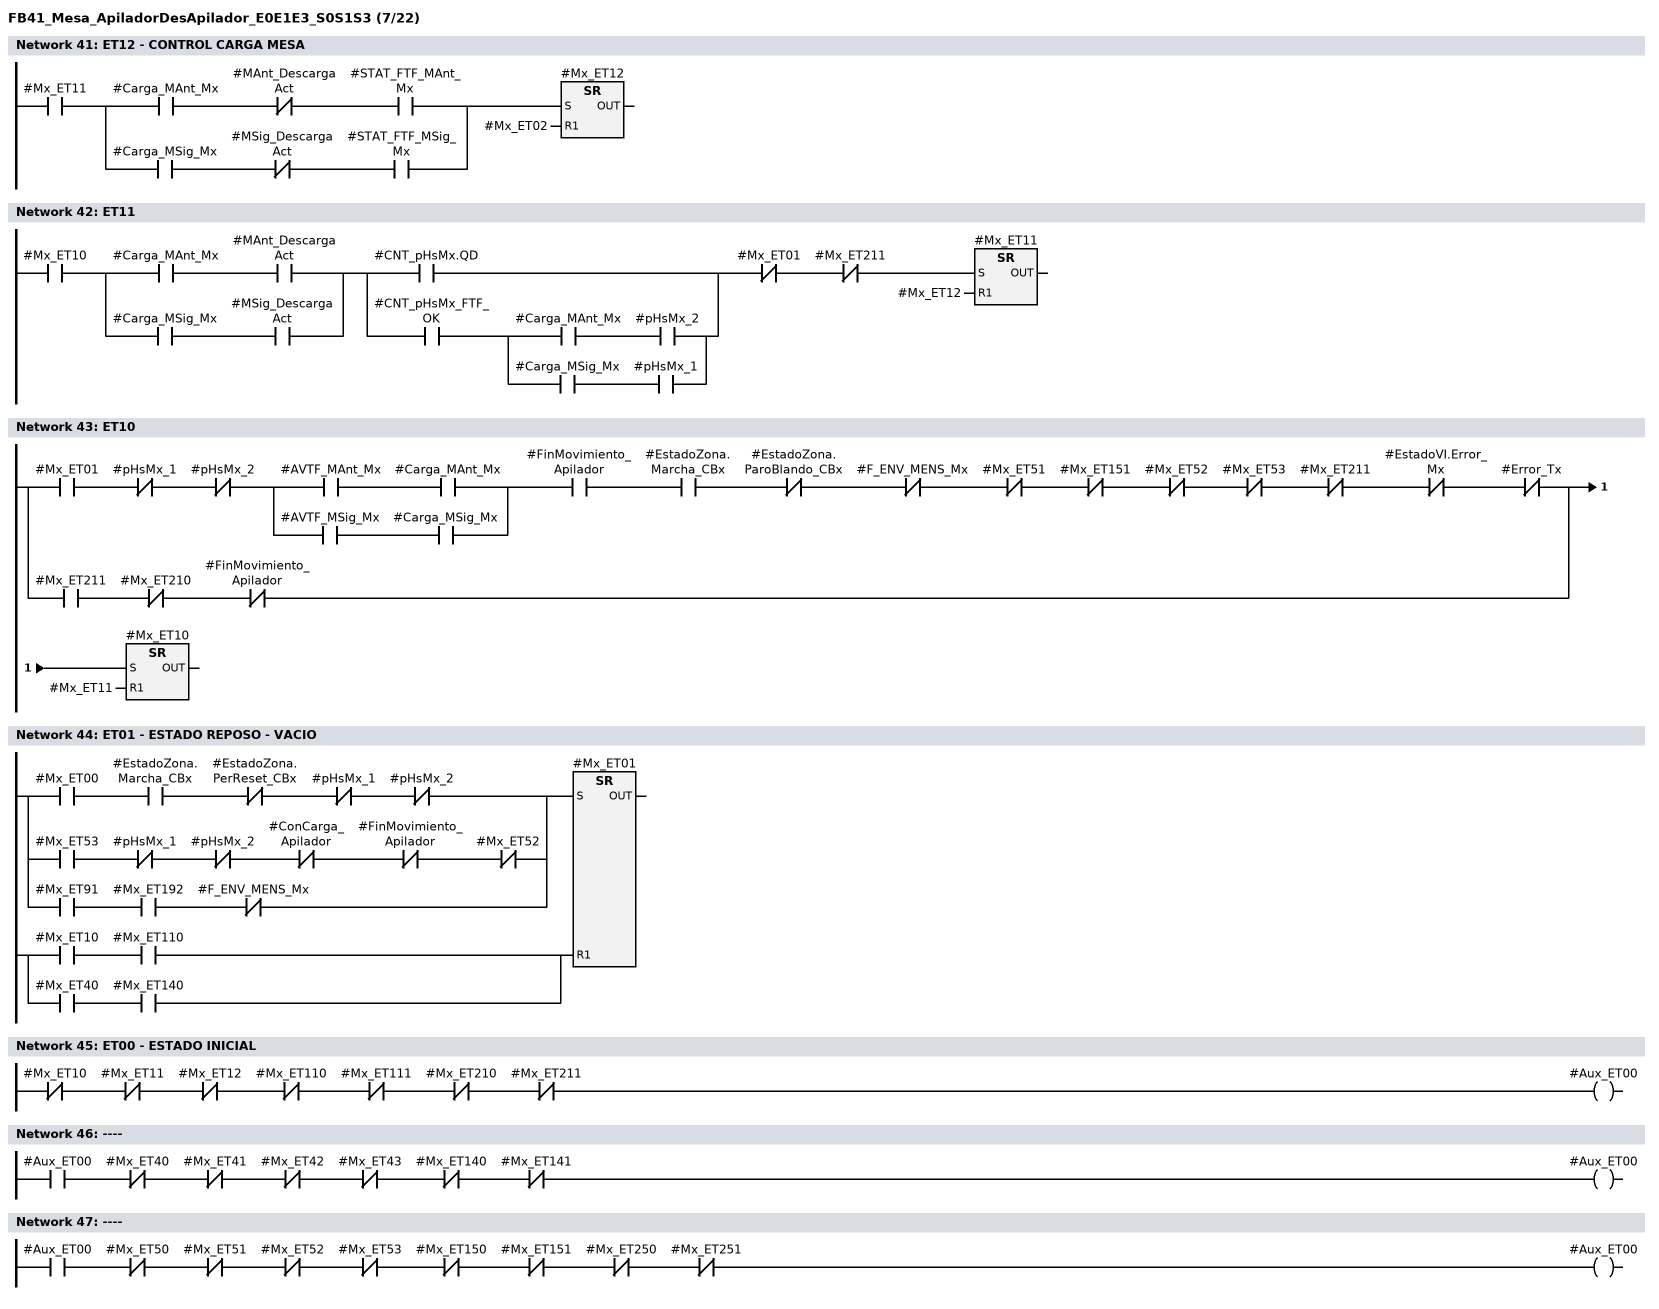
   RUNG wire#powerrail
      Contact( #Mx_ET11 )
      wire#w1
      Contact( #Carga_MAnt_Mx )
      I_Contact( #MAnt_DescargaAct )
      Contact( #STAT_FTF_MAnt_Mx )
      wire#w2
      S_SR(operand := #Mx_ET12, r1 := #Mx_ET02)
   END_RUNG
   RUNG wire#w1
      Contact( #Carga_MSig_Mx )
      I_Contact( #MSig_DescargaAct )
      Contact( #STAT_FTF_MSig_Mx )
   END_RUNG wire#w2
   // the same network as SCL:
   IF #Mx_ET11 AND ((#Carga_MAnt_Mx AND NOT #MAnt_DescargaAct AND #STAT_FTF_MAnt_Mx) OR (#Carga_MSig_Mx AND NOT #MSig_DescargaAct AND #STAT_FTF_MSig_Mx)) THEN
       #Mx_ET12 := TRUE;   // SR flip-flop
   END_IF;
   IF #Mx_ET02 THEN #Mx_ET12 := FALSE; END_IF;
END_REGION

REGION Network 42: ET11
   RUNG wire#powerrail
      Contact( #Mx_ET10 )
      wire#w1
      Contact( #Carga_MAnt_Mx )
      Contact( #MAnt_DescargaAct )
      wire#w2
      Contact( #CNT_pHsMx.QD )
      wire#w3
      I_Contact( #Mx_ET01 )
      I_Contact( #Mx_ET211 )
      S_SR(operand := #Mx_ET11, r1 := #Mx_ET12)
   END_RUNG
   RUNG wire#w1
      Contact( #Carga_MSig_Mx )
      Contact( #MSig_DescargaAct )
   END_RUNG wire#w2
   RUNG wire#w2
      Contact( #CNT_pHsMx_FTF_OK )
      wire#w4
      Contact( #Carga_MAnt_Mx )
      Contact( #pHsMx_2 )
   END_RUNG wire#w3
   RUNG wire#w4
      Contact( #Carga_MSig_Mx )
      Contact( #pHsMx_1 )
   END_RUNG wire#w3
   // the same network as SCL:
   IF #Mx_ET10 AND ((#Carga_MAnt_Mx AND #MAnt_DescargaAct) OR (#Carga_MSig_Mx AND #MSig_DescargaAct)) AND (#CNT_pHsMx.QD OR (#CNT_pHsMx_FTF_OK AND ((#Carga_MAnt_Mx AND #pHsMx_2) OR (#Carga_MSig_Mx AND #pHsMx_1)))) AND NOT #Mx_ET01 AND NOT #Mx_ET211 THEN
       #Mx_ET11 := TRUE;   // SR flip-flop
   END_IF;
   IF #Mx_ET12 THEN #Mx_ET11 := FALSE; END_IF;
END_REGION

REGION Network 43: ET10
   RUNG wire#powerrail
      Contact( #Mx_ET01 )
      I_Contact( #pHsMx_1 )
      I_Contact( #pHsMx_2 )
      wire#w1
      Contact( #AVTF_MAnt_Mx )
      Contact( #Carga_MAnt_Mx )
      wire#w2
      Contact( #FinMovimiento_Apilador )
      Contact( #EstadoZona.Marcha_CBx )
      I_Contact( #EstadoZona.ParoBlando_CBx )
      I_Contact( #F_ENV_MENS_Mx )
      I_Contact( #Mx_ET51 )
      I_Contact( #Mx_ET151 )
      I_Contact( #Mx_ET52 )
      I_Contact( #Mx_ET53 )
      I_Contact( #Mx_ET211 )
      I_Contact( #EstadoVI.Error_Mx )
      I_Contact( #Error_Tx )
      wire#w3
      S_SR(operand := #Mx_ET10, r1 := #Mx_ET11)
   END_RUNG
   RUNG wire#w1
      Contact( #AVTF_MSig_Mx )
      Contact( #Carga_MSig_Mx )
   END_RUNG wire#w2
   RUNG wire#powerrail
      Contact( #Mx_ET211 )
      I_Contact( #Mx_ET210 )
      I_Contact( #FinMovimiento_Apilador )
   END_RUNG wire#w3
   // the same network as SCL:
   IF (#Mx_ET01 AND NOT #pHsMx_1 AND NOT #pHsMx_2 AND ((#AVTF_MAnt_Mx AND #Carga_MAnt_Mx) OR (#AVTF_MSig_Mx AND #Carga_MSig_Mx)) AND #FinMovimiento_Apilador AND #EstadoZona.Marcha_CBx AND NOT #EstadoZona.ParoBlando_CBx AND NOT #F_ENV_MENS_Mx AND NOT #Mx_ET51 AND NOT #Mx_ET151 AND NOT #Mx_ET52 AND NOT #Mx_ET53 AND NOT #Mx_ET211 AND NOT #EstadoVI.Error_Mx AND NOT #Error_Tx) OR (#Mx_ET211 AND NOT #Mx_ET210 AND NOT #FinMovimiento_Apilador) THEN
       #Mx_ET10 := TRUE;   // SR flip-flop
   END_IF;
   IF #Mx_ET11 THEN #Mx_ET10 := FALSE; END_IF;
END_REGION

REGION Network 44: ET01 - ESTADO REPOSO - VACIO
   RUNG wire#powerrail
      Contact( #Mx_ET00 )
      Contact( #EstadoZona.Marcha_CBx )
      I_Contact( #EstadoZona.PerReset_CBx )
      I_Contact( #pHsMx_1 )
      I_Contact( #pHsMx_2 )
      wire#w1
      S_SR(operand := #Mx_ET01, r1 := wire#w2)
   END_RUNG
   RUNG wire#powerrail
      Contact( #Mx_ET53 )
      I_Contact( #pHsMx_1 )
      I_Contact( #pHsMx_2 )
      I_Contact( #ConCarga_Apilador )
      I_Contact( #FinMovimiento_Apilador )
      I_Contact( #Mx_ET52 )
   END_RUNG wire#w1
   RUNG wire#powerrail
      Contact( #Mx_ET91 )
      Contact( #Mx_ET192 )
      I_Contact( #F_ENV_MENS_Mx )
   END_RUNG wire#w1
   RUNG wire#powerrail
      Contact( #Mx_ET10 )
      Contact( #Mx_ET110 )
   END_RUNG wire#w2
   RUNG wire#powerrail
      Contact( #Mx_ET40 )
      Contact( #Mx_ET140 )
   END_RUNG wire#w2
   // the same network as SCL:
   IF (#Mx_ET00 AND #EstadoZona.Marcha_CBx AND NOT #EstadoZona.PerReset_CBx AND NOT #pHsMx_1 AND NOT #pHsMx_2) OR (#Mx_ET53 AND NOT #pHsMx_1 AND NOT #pHsMx_2 AND NOT #ConCarga_Apilador AND NOT #FinMovimiento_Apilador AND NOT #Mx_ET52) OR (#Mx_ET91 AND #Mx_ET192 AND NOT #F_ENV_MENS_Mx) THEN
       #Mx_ET01 := TRUE;   // SR flip-flop
   END_IF;
   IF (#Mx_ET10 AND #Mx_ET110) OR (#Mx_ET40 AND #Mx_ET140) THEN #Mx_ET01 := FALSE; END_IF;
END_REGION

REGION Network 45: ET00 - ESTADO INICIAL
   RUNG wire#powerrail
      I_Contact( #Mx_ET10 )
      I_Contact( #Mx_ET11 )
      I_Contact( #Mx_ET12 )
      I_Contact( #Mx_ET110 )
      I_Contact( #Mx_ET111 )
      I_Contact( #Mx_ET210 )
      I_Contact( #Mx_ET211 )
      Coil( #Aux_ET00 )
   END_RUNG
   // the same network as SCL:
   #Aux_ET00 := NOT #Mx_ET10 AND NOT #Mx_ET11 AND NOT #Mx_ET12 AND NOT #Mx_ET110 AND NOT #Mx_ET111 AND NOT #Mx_ET210 AND NOT #Mx_ET211;
END_REGION

REGION Network 46: ----
   RUNG wire#powerrail
      Contact( #Aux_ET00 )
      I_Contact( #Mx_ET40 )
      I_Contact( #Mx_ET41 )
      I_Contact( #Mx_ET42 )
      I_Contact( #Mx_ET43 )
      I_Contact( #Mx_ET140 )
      I_Contact( #Mx_ET141 )
      Coil( #Aux_ET00 )
   END_RUNG
   // the same network as SCL:
   #Aux_ET00 := #Aux_ET00 AND NOT #Mx_ET40 AND NOT #Mx_ET41 AND NOT #Mx_ET42 AND NOT #Mx_ET43 AND NOT #Mx_ET140 AND NOT #Mx_ET141;
END_REGION

REGION Network 47: ----
   RUNG wire#powerrail
      Contact( #Aux_ET00 )
      I_Contact( #Mx_ET50 )
      I_Contact( #Mx_ET51 )
      I_Contact( #Mx_ET52 )
      I_Contact( #Mx_ET53 )
      I_Contact( #Mx_ET150 )
      I_Contact( #Mx_ET151 )
      I_Contact( #Mx_ET250 )
      I_Contact( #Mx_ET251 )
      Coil( #Aux_ET00 )
   END_RUNG
   // the same network as SCL:
   #Aux_ET00 := #Aux_ET00 AND NOT #Mx_ET50 AND NOT #Mx_ET51 AND NOT #Mx_ET52 AND NOT #Mx_ET53 AND NOT #Mx_ET150 AND NOT #Mx_ET151 AND NOT #Mx_ET250 AND NOT #Mx_ET251;
END_REGION

REGION Network 48: -----
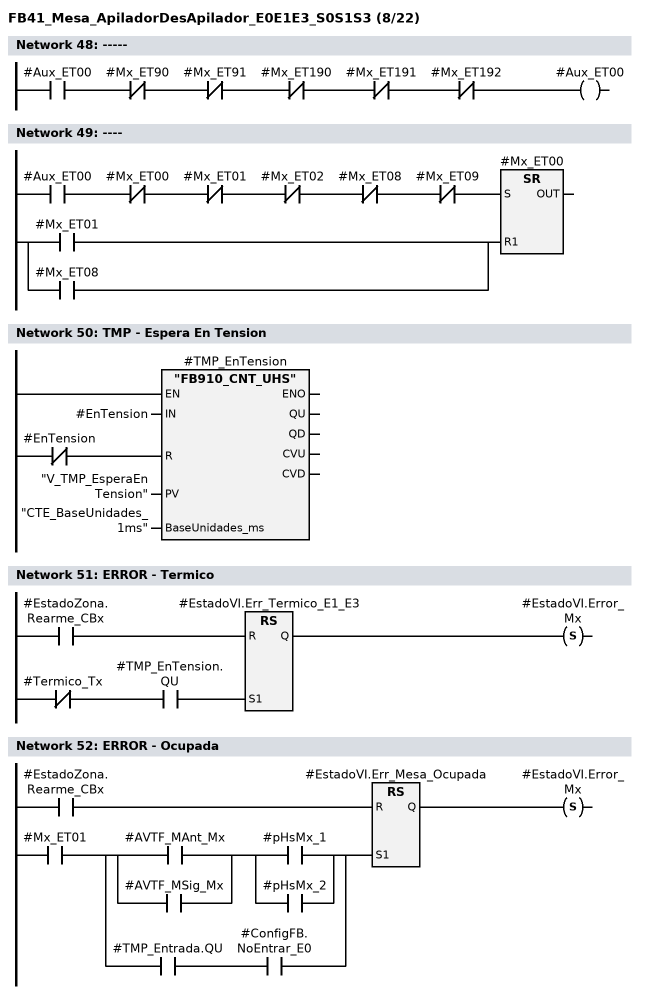
   RUNG wire#powerrail
      Contact( #Aux_ET00 )
      I_Contact( #Mx_ET90 )
      I_Contact( #Mx_ET91 )
      I_Contact( #Mx_ET190 )
      I_Contact( #Mx_ET191 )
      I_Contact( #Mx_ET192 )
      Coil( #Aux_ET00 )
   END_RUNG
   // the same network as SCL:
   #Aux_ET00 := #Aux_ET00 AND NOT #Mx_ET90 AND NOT #Mx_ET91 AND NOT #Mx_ET190 AND NOT #Mx_ET191 AND NOT #Mx_ET192;
END_REGION

REGION Network 49: ----
   RUNG wire#powerrail
      Contact( #Aux_ET00 )
      I_Contact( #Mx_ET00 )
      I_Contact( #Mx_ET01 )
      I_Contact( #Mx_ET02 )
      I_Contact( #Mx_ET08 )
      I_Contact( #Mx_ET09 )
      S_SR(operand := #Mx_ET00, r1 := wire#w1)
   END_RUNG
   RUNG wire#powerrail
      Contact( #Mx_ET01 )
   END_RUNG wire#w1
   RUNG wire#powerrail
      Contact( #Mx_ET08 )
   END_RUNG wire#w1
   // the same network as SCL:
   IF #Aux_ET00 AND NOT #Mx_ET00 AND NOT #Mx_ET01 AND NOT #Mx_ET02 AND NOT #Mx_ET08 AND NOT #Mx_ET09 THEN
       #Mx_ET00 := TRUE;   // SR flip-flop
   END_IF;
   IF #Mx_ET01 OR #Mx_ET08 THEN #Mx_ET00 := FALSE; END_IF;
END_REGION

REGION Network 50: TMP - Espera En Tension
   RUNG wire#powerrail
      #TMP_EnTension(R := wire#w1, IN := #EnTension, PV := "V_TMP_EsperaEnTension", BaseUnidades_ms := "CTE_BaseUnidades_1ms", QU =>, QD =>, CVU =>, CVD =>)
   END_RUNG
   RUNG wire#powerrail
      I_Contact( #EnTension )
   END_RUNG wire#w1
   // the same network as SCL:
   #TMP_EnTension(IN := #EnTension,   // "FB910_CNT_UHS"
                  R := NOT #EnTension,
                  PV := "V_TMP_EsperaEnTension",
                  BaseUnidades_ms := "CTE_BaseUnidades_1ms");
END_REGION

REGION Network 51: ERROR - Termico
   RUNG wire#powerrail
      Contact( #EstadoZona.Rearme_CBx )
      S_RS(operand := #EstadoVI.Err_Termico_E1_E3, s1 := wire#w1)
      S_Coil( #EstadoVI.Error_Mx )
   END_RUNG
   RUNG wire#powerrail
      I_Contact( #Termico_Tx )
      Contact( #TMP_EnTension.QU )
   END_RUNG wire#w1
   // the same network as SCL:
   IF #EstadoZona.Rearme_CBx THEN
       #EstadoVI.Err_Termico_E1_E3 := FALSE;   // RS flip-flop
   END_IF;
   IF NOT #Termico_Tx AND #TMP_EnTension.QU THEN #EstadoVI.Err_Termico_E1_E3 := TRUE; END_IF;
   IF #EstadoVI.Err_Termico_E1_E3 THEN #EstadoVI.Error_Mx := TRUE; END_IF;
END_REGION

REGION Network 52: ERROR - Ocupada
   RUNG wire#powerrail
      Contact( #EstadoZona.Rearme_CBx )
      S_RS(operand := #EstadoVI.Err_Mesa_Ocupada, s1 := wire#w3)
      S_Coil( #EstadoVI.Error_Mx )
   END_RUNG
   RUNG wire#powerrail
      Contact( #Mx_ET01 )
      wire#w1
      Contact( #AVTF_MAnt_Mx )
      wire#w2
      Contact( #pHsMx_1 )
   END_RUNG wire#w3
   RUNG wire#w1
      Contact( #AVTF_MSig_Mx )
   END_RUNG wire#w2
   RUNG wire#w2
      Contact( #pHsMx_2 )
   END_RUNG wire#w3
   RUNG wire#w1
      Contact( #TMP_Entrada.QU )
      Contact( #ConfigFB.NoEntrar_E0 )
   END_RUNG wire#w3
   // the same network as SCL:
   IF #EstadoZona.Rearme_CBx THEN
       #EstadoVI.Err_Mesa_Ocupada := FALSE;   // RS flip-flop
   END_IF;
   IF #Mx_ET01 AND (((#AVTF_MAnt_Mx OR #AVTF_MSig_Mx) AND (#pHsMx_1 OR #pHsMx_2)) OR (#TMP_Entrada.QU AND #ConfigFB.NoEntrar_E0)) THEN
       #EstadoVI.Err_Mesa_Ocupada := TRUE;
   END_IF;
   IF #EstadoVI.Err_Mesa_Ocupada THEN #EstadoVI.Error_Mx := TRUE; END_IF;
END_REGION

REGION Network 53: CNT - ERROR - Arrastre
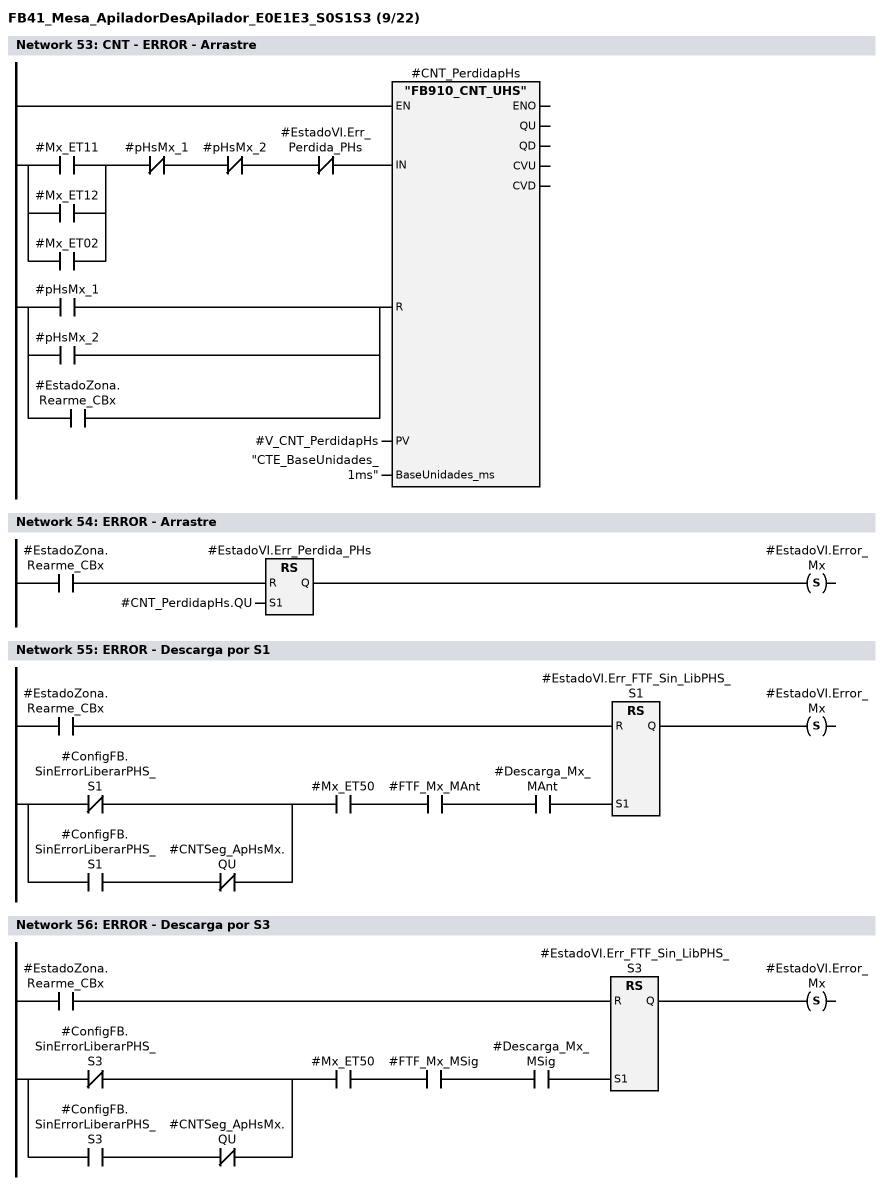
   RUNG wire#powerrail
      #CNT_PerdidapHs(IN := wire#w2, R := wire#w3, PV := #V_CNT_PerdidapHs, BaseUnidades_ms := "CTE_BaseUnidades_1ms", QU =>, QD =>, CVU =>, CVD =>)
   END_RUNG
   RUNG wire#powerrail
      Contact( #Mx_ET11 )
      wire#w1
      I_Contact( #pHsMx_1 )
      I_Contact( #pHsMx_2 )
      I_Contact( #EstadoVI.Err_Perdida_PHs )
   END_RUNG wire#w2
   RUNG wire#powerrail
      Contact( #Mx_ET12 )
   END_RUNG wire#w1
   RUNG wire#powerrail
      Contact( #Mx_ET02 )
   END_RUNG wire#w1
   RUNG wire#powerrail
      Contact( #pHsMx_1 )
   END_RUNG wire#w3
   RUNG wire#powerrail
      Contact( #pHsMx_2 )
   END_RUNG wire#w3
   RUNG wire#powerrail
      Contact( #EstadoZona.Rearme_CBx )
   END_RUNG wire#w3
   // the same network as SCL:
   #CNT_PerdidapHs(IN := (#Mx_ET11 OR #Mx_ET12 OR #Mx_ET02) AND NOT #pHsMx_1 AND NOT #pHsMx_2 AND NOT #EstadoVI.Err_Perdida_PHs,   // "FB910_CNT_UHS"
                   R := #pHsMx_1 OR #pHsMx_2 OR #EstadoZona.Rearme_CBx,
                   PV := #V_CNT_PerdidapHs,
                   BaseUnidades_ms := "CTE_BaseUnidades_1ms");
END_REGION

REGION Network 54: ERROR - Arrastre
   RUNG wire#powerrail
      Contact( #EstadoZona.Rearme_CBx )
      S_RS(operand := #EstadoVI.Err_Perdida_PHs, s1 := #CNT_PerdidapHs.QU)
      S_Coil( #EstadoVI.Error_Mx )
   END_RUNG
   // the same network as SCL:
   IF #EstadoZona.Rearme_CBx THEN
       #EstadoVI.Err_Perdida_PHs := FALSE;   // RS flip-flop
   END_IF;
   IF #CNT_PerdidapHs.QU THEN #EstadoVI.Err_Perdida_PHs := TRUE; END_IF;
   IF #EstadoVI.Err_Perdida_PHs THEN #EstadoVI.Error_Mx := TRUE; END_IF;
END_REGION

REGION Network 55: ERROR - Descarga por S1
   RUNG wire#powerrail
      Contact( #EstadoZona.Rearme_CBx )
      S_RS(operand := #EstadoVI.Err_FTF_Sin_LibPHS_S1, s1 := wire#w2)
      S_Coil( #EstadoVI.Error_Mx )
   END_RUNG
   RUNG wire#powerrail
      I_Contact( #ConfigFB.SinErrorLiberarPHS_S1 )
      wire#w1
      Contact( #Mx_ET50 )
      Contact( #FTF_Mx_MAnt )
      Contact( #Descarga_Mx_MAnt )
   END_RUNG wire#w2
   RUNG wire#powerrail
      Contact( #ConfigFB.SinErrorLiberarPHS_S1 )
      I_Contact( #CNTSeg_ApHsMx.QU )
   END_RUNG wire#w1
   // the same network as SCL:
   IF #EstadoZona.Rearme_CBx THEN
       #EstadoVI.Err_FTF_Sin_LibPHS_S1 := FALSE;   // RS flip-flop
   END_IF;
   IF (NOT #ConfigFB.SinErrorLiberarPHS_S1 OR (#ConfigFB.SinErrorLiberarPHS_S1 AND NOT #CNTSeg_ApHsMx.QU)) AND #Mx_ET50 AND #FTF_Mx_MAnt AND #Descarga_Mx_MAnt THEN
       #EstadoVI.Err_FTF_Sin_LibPHS_S1 := TRUE;
   END_IF;
   IF #EstadoVI.Err_FTF_Sin_LibPHS_S1 THEN #EstadoVI.Error_Mx := TRUE; END_IF;
END_REGION

REGION Network 56: ERROR - Descarga por S3
   RUNG wire#powerrail
      Contact( #EstadoZona.Rearme_CBx )
      S_RS(operand := #EstadoVI.Err_FTF_Sin_LibPHS_S3, s1 := wire#w2)
      S_Coil( #EstadoVI.Error_Mx )
   END_RUNG
   RUNG wire#powerrail
      I_Contact( #ConfigFB.SinErrorLiberarPHS_S3 )
      wire#w1
      Contact( #Mx_ET50 )
      Contact( #FTF_Mx_MSig )
      Contact( #Descarga_Mx_MSig )
   END_RUNG wire#w2
   RUNG wire#powerrail
      Contact( #ConfigFB.SinErrorLiberarPHS_S3 )
      I_Contact( #CNTSeg_ApHsMx.QU )
   END_RUNG wire#w1
   // the same network as SCL:
   IF #EstadoZona.Rearme_CBx THEN
       #EstadoVI.Err_FTF_Sin_LibPHS_S3 := FALSE;   // RS flip-flop
   END_IF;
   IF (NOT #ConfigFB.SinErrorLiberarPHS_S3 OR (#ConfigFB.SinErrorLiberarPHS_S3 AND NOT #CNTSeg_ApHsMx.QU)) AND #Mx_ET50 AND #FTF_Mx_MSig AND #Descarga_Mx_MSig THEN
       #EstadoVI.Err_FTF_Sin_LibPHS_S3 := TRUE;
   END_IF;
   IF #EstadoVI.Err_FTF_Sin_LibPHS_S3 THEN #EstadoVI.Error_Mx := TRUE; END_IF;
END_REGION

REGION Network 57: TMP - ERROR - TimeOut Avance
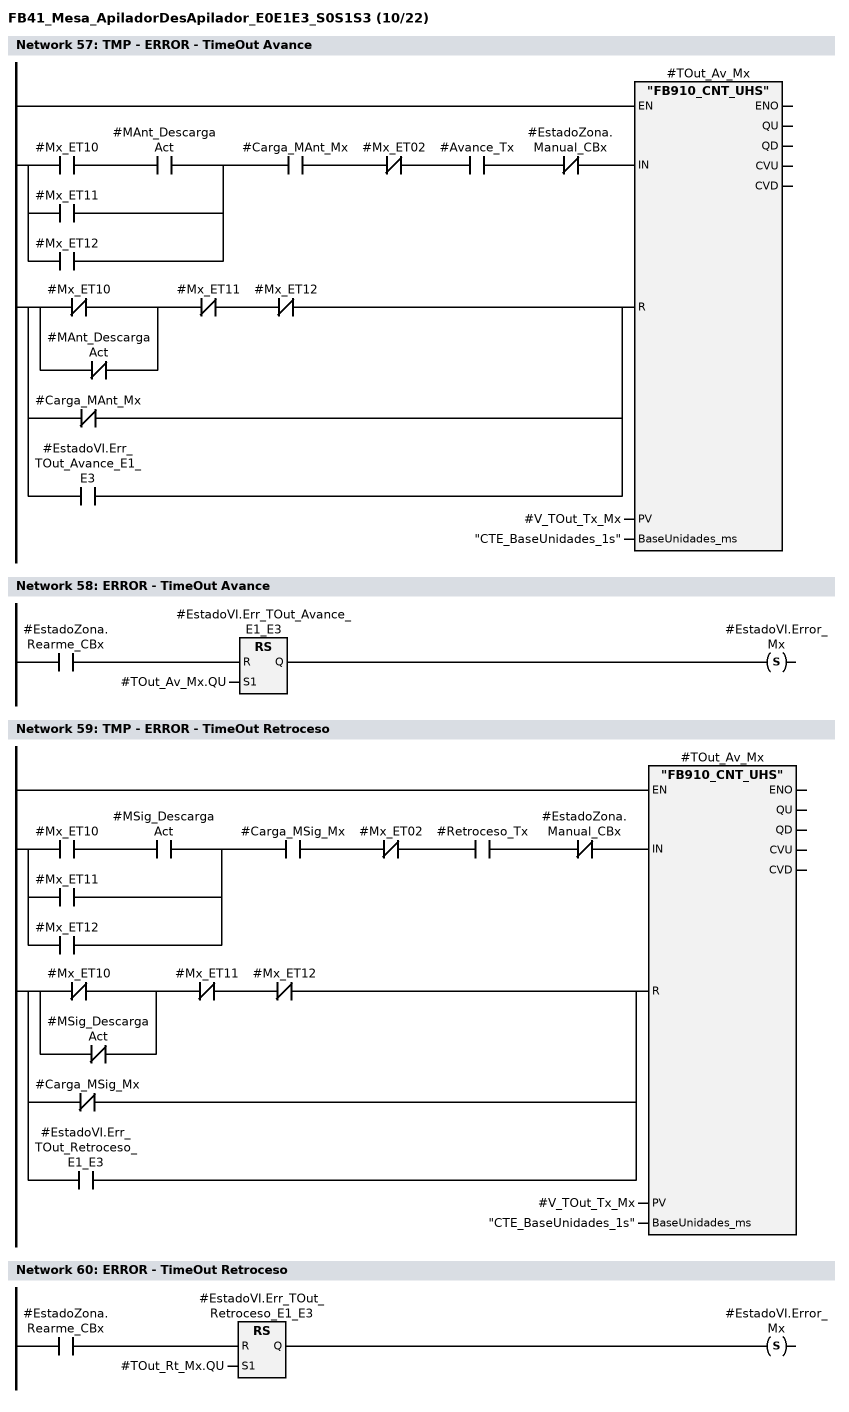
   RUNG wire#powerrail
      #TOut_Av_Mx(IN := wire#w2, R := wire#w4, PV := #V_TOut_Tx_Mx, BaseUnidades_ms := "CTE_BaseUnidades_1s", QU =>, QD =>, CVU =>, CVD =>)
   END_RUNG
   RUNG wire#powerrail
      Contact( #Mx_ET10 )
      Contact( #MAnt_DescargaAct )
      wire#w1
      Contact( #Carga_MAnt_Mx )
      I_Contact( #Mx_ET02 )
      Contact( #Avance_Tx )
      I_Contact( #EstadoZona.Manual_CBx )
   END_RUNG wire#w2
   RUNG wire#powerrail
      Contact( #Mx_ET11 )
   END_RUNG wire#w1
   RUNG wire#powerrail
      Contact( #Mx_ET12 )
   END_RUNG wire#w1
   RUNG wire#powerrail
      I_Contact( #Mx_ET10 )
      wire#w3
      I_Contact( #Mx_ET11 )
      I_Contact( #Mx_ET12 )
   END_RUNG wire#w4
   RUNG wire#powerrail
      I_Contact( #MAnt_DescargaAct )
   END_RUNG wire#w3
   RUNG wire#powerrail
      I_Contact( #Carga_MAnt_Mx )
   END_RUNG wire#w4
   RUNG wire#powerrail
      Contact( #EstadoVI.Err_TOut_Avance_E1_E3 )
   END_RUNG wire#w4
   // the same network as SCL:
   #TOut_Av_Mx(IN := ((#Mx_ET10 AND #MAnt_DescargaAct) OR #Mx_ET11 OR #Mx_ET12) AND #Carga_MAnt_Mx AND NOT #Mx_ET02 AND #Avance_Tx AND NOT #EstadoZona.Manual_CBx,   // "FB910_CNT_UHS"
               R := ((NOT #Mx_ET10 OR NOT #MAnt_DescargaAct) AND NOT #Mx_ET11 AND NOT #Mx_ET12) OR NOT #Carga_MAnt_Mx OR #EstadoVI.Err_TOut_Avance_E1_E3,
               PV := #V_TOut_Tx_Mx,
               BaseUnidades_ms := "CTE_BaseUnidades_1s");
END_REGION

REGION Network 58: ERROR - TimeOut Avance
   RUNG wire#powerrail
      Contact( #EstadoZona.Rearme_CBx )
      S_RS(operand := #EstadoVI.Err_TOut_Avance_E1_E3, s1 := #TOut_Av_Mx.QU)
      S_Coil( #EstadoVI.Error_Mx )
   END_RUNG
   // the same network as SCL:
   IF #EstadoZona.Rearme_CBx THEN
       #EstadoVI.Err_TOut_Avance_E1_E3 := FALSE;   // RS flip-flop
   END_IF;
   IF #TOut_Av_Mx.QU THEN #EstadoVI.Err_TOut_Avance_E1_E3 := TRUE; END_IF;
   IF #EstadoVI.Err_TOut_Avance_E1_E3 THEN #EstadoVI.Error_Mx := TRUE; END_IF;
END_REGION

REGION Network 59: TMP - ERROR - TimeOut Retroceso
   RUNG wire#powerrail
      #TOut_Av_Mx(IN := wire#w2, R := wire#w4, PV := #V_TOut_Tx_Mx, BaseUnidades_ms := "CTE_BaseUnidades_1s", QU =>, QD =>, CVU =>, CVD =>)
   END_RUNG
   RUNG wire#powerrail
      Contact( #Mx_ET10 )
      Contact( #MSig_DescargaAct )
      wire#w1
      Contact( #Carga_MSig_Mx )
      I_Contact( #Mx_ET02 )
      Contact( #Retroceso_Tx )
      I_Contact( #EstadoZona.Manual_CBx )
   END_RUNG wire#w2
   RUNG wire#powerrail
      Contact( #Mx_ET11 )
   END_RUNG wire#w1
   RUNG wire#powerrail
      Contact( #Mx_ET12 )
   END_RUNG wire#w1
   RUNG wire#powerrail
      I_Contact( #Mx_ET10 )
      wire#w3
      I_Contact( #Mx_ET11 )
      I_Contact( #Mx_ET12 )
   END_RUNG wire#w4
   RUNG wire#powerrail
      I_Contact( #MSig_DescargaAct )
   END_RUNG wire#w3
   RUNG wire#powerrail
      I_Contact( #Carga_MSig_Mx )
   END_RUNG wire#w4
   RUNG wire#powerrail
      Contact( #EstadoVI.Err_TOut_Retroceso_E1_E3 )
   END_RUNG wire#w4
   // the same network as SCL:
   #TOut_Av_Mx(IN := ((#Mx_ET10 AND #MSig_DescargaAct) OR #Mx_ET11 OR #Mx_ET12) AND #Carga_MSig_Mx AND NOT #Mx_ET02 AND #Retroceso_Tx AND NOT #EstadoZona.Manual_CBx,   // "FB910_CNT_UHS"
               R := ((NOT #Mx_ET10 OR NOT #MSig_DescargaAct) AND NOT #Mx_ET11 AND NOT #Mx_ET12) OR NOT #Carga_MSig_Mx OR #EstadoVI.Err_TOut_Retroceso_E1_E3,
               PV := #V_TOut_Tx_Mx,
               BaseUnidades_ms := "CTE_BaseUnidades_1s");
END_REGION

REGION Network 60: ERROR - TimeOut Retroceso
   RUNG wire#powerrail
      Contact( #EstadoZona.Rearme_CBx )
      S_RS(operand := #EstadoVI.Err_TOut_Retroceso_E1_E3, s1 := #TOut_Rt_Mx.QU)
      S_Coil( #EstadoVI.Error_Mx )
   END_RUNG
   // the same network as SCL:
   IF #EstadoZona.Rearme_CBx THEN
       #EstadoVI.Err_TOut_Retroceso_E1_E3 := FALSE;   // RS flip-flop
   END_IF;
   IF #TOut_Rt_Mx.QU THEN #EstadoVI.Err_TOut_Retroceso_E1_E3 := TRUE; END_IF;
   IF #EstadoVI.Err_TOut_Retroceso_E1_E3 THEN #EstadoVI.Error_Mx := TRUE; END_IF;
END_REGION

REGION Network 61: TMP - ERROR - TimeOut Subir TP
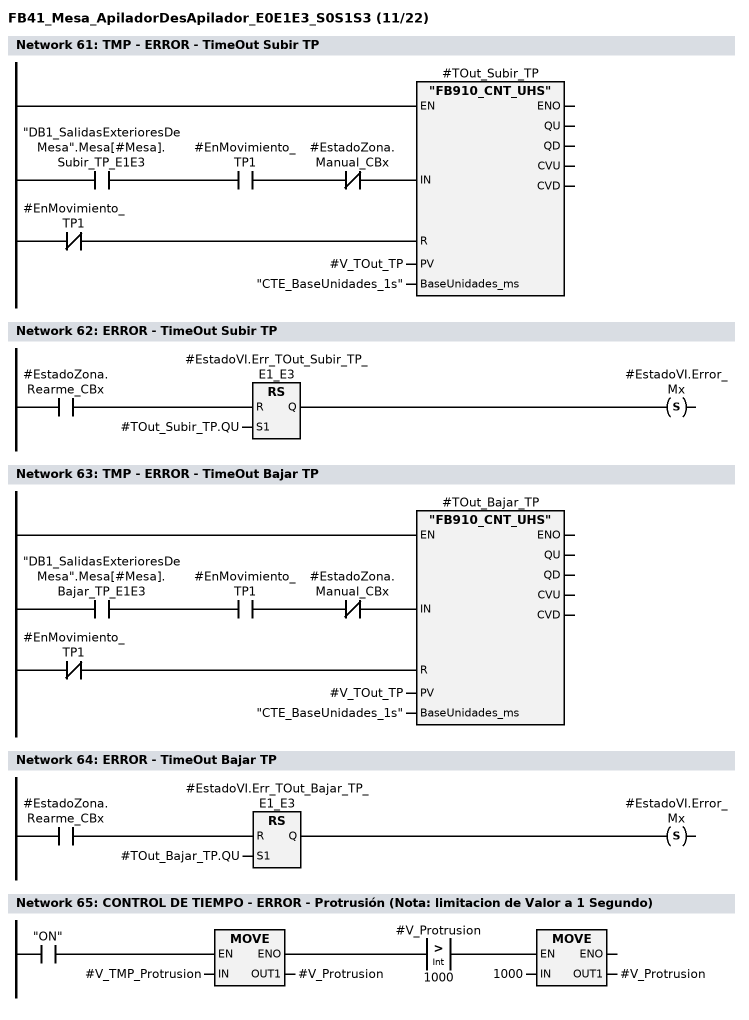
   RUNG wire#powerrail
      #TOut_Subir_TP(IN := wire#w1, R := wire#w2, PV := #V_TOut_TP, BaseUnidades_ms := "CTE_BaseUnidades_1s", QU =>, QD =>, CVU =>, CVD =>)
   END_RUNG
   RUNG wire#powerrail
      Contact( "DB1_SalidasExterioresDeMesa".Mesa[#Mesa].Subir_TP_E1E3 )
      Contact( #EnMovimiento_TP1 )
      I_Contact( #EstadoZona.Manual_CBx )
   END_RUNG wire#w1
   RUNG wire#powerrail
      I_Contact( #EnMovimiento_TP1 )
   END_RUNG wire#w2
   // the same network as SCL:
   #TOut_Subir_TP(IN := "DB1_SalidasExterioresDeMesa".Mesa[#Mesa].Subir_TP_E1E3 AND #EnMovimiento_TP1 AND NOT #EstadoZona.Manual_CBx,   // "FB910_CNT_UHS"
                  R := NOT #EnMovimiento_TP1,
                  PV := #V_TOut_TP,
                  BaseUnidades_ms := "CTE_BaseUnidades_1s");
END_REGION

REGION Network 62: ERROR - TimeOut Subir TP
   RUNG wire#powerrail
      Contact( #EstadoZona.Rearme_CBx )
      S_RS(operand := #EstadoVI.Err_TOut_Subir_TP_E1_E3, s1 := #TOut_Subir_TP.QU)
      S_Coil( #EstadoVI.Error_Mx )
   END_RUNG
   // the same network as SCL:
   IF #EstadoZona.Rearme_CBx THEN
       #EstadoVI.Err_TOut_Subir_TP_E1_E3 := FALSE;   // RS flip-flop
   END_IF;
   IF #TOut_Subir_TP.QU THEN #EstadoVI.Err_TOut_Subir_TP_E1_E3 := TRUE; END_IF;
   IF #EstadoVI.Err_TOut_Subir_TP_E1_E3 THEN #EstadoVI.Error_Mx := TRUE; END_IF;
END_REGION

REGION Network 63: TMP - ERROR - TimeOut Bajar TP
   RUNG wire#powerrail
      #TOut_Bajar_TP(IN := wire#w1, R := wire#w2, PV := #V_TOut_TP, BaseUnidades_ms := "CTE_BaseUnidades_1s", QU =>, QD =>, CVU =>, CVD =>)
   END_RUNG
   RUNG wire#powerrail
      Contact( "DB1_SalidasExterioresDeMesa".Mesa[#Mesa].Bajar_TP_E1E3 )
      Contact( #EnMovimiento_TP1 )
      I_Contact( #EstadoZona.Manual_CBx )
   END_RUNG wire#w1
   RUNG wire#powerrail
      I_Contact( #EnMovimiento_TP1 )
   END_RUNG wire#w2
   // the same network as SCL:
   #TOut_Bajar_TP(IN := "DB1_SalidasExterioresDeMesa".Mesa[#Mesa].Bajar_TP_E1E3 AND #EnMovimiento_TP1 AND NOT #EstadoZona.Manual_CBx,   // "FB910_CNT_UHS"
                  R := NOT #EnMovimiento_TP1,
                  PV := #V_TOut_TP,
                  BaseUnidades_ms := "CTE_BaseUnidades_1s");
END_REGION

REGION Network 64: ERROR - TimeOut Bajar TP
   RUNG wire#powerrail
      Contact( #EstadoZona.Rearme_CBx )
      S_RS(operand := #EstadoVI.Err_TOut_Bajar_TP_E1_E3, s1 := #TOut_Bajar_TP.QU)
      S_Coil( #EstadoVI.Error_Mx )
   END_RUNG
   // the same network as SCL:
   IF #EstadoZona.Rearme_CBx THEN
       #EstadoVI.Err_TOut_Bajar_TP_E1_E3 := FALSE;   // RS flip-flop
   END_IF;
   IF #TOut_Bajar_TP.QU THEN #EstadoVI.Err_TOut_Bajar_TP_E1_E3 := TRUE; END_IF;
   IF #EstadoVI.Err_TOut_Bajar_TP_E1_E3 THEN #EstadoVI.Error_Mx := TRUE; END_IF;
END_REGION

REGION Network 65: CONTROL DE TIEMPO - ERROR - Protrusión (Nota: limitacion de Valor a 1 Segundo)
   RUNG wire#powerrail
      Contact( "ON" )
      Move(in := #V_TMP_Protrusion, out1 => #V_Protrusion)
      { S7_Templates := "SrcType := Int" } GT_Contact(in1 := #V_Protrusion, in2 := 1000)
      Move(in := 1000, out1 => #V_Protrusion)
   END_RUNG
   // the same network as SCL:
   IF "ON" THEN #V_Protrusion := #V_TMP_Protrusion; END_IF;
   IF "ON" AND (#V_Protrusion > 1000) THEN #V_Protrusion := 1000; END_IF;
END_REGION

REGION Network 66: TMP - ERROR - Protrusión
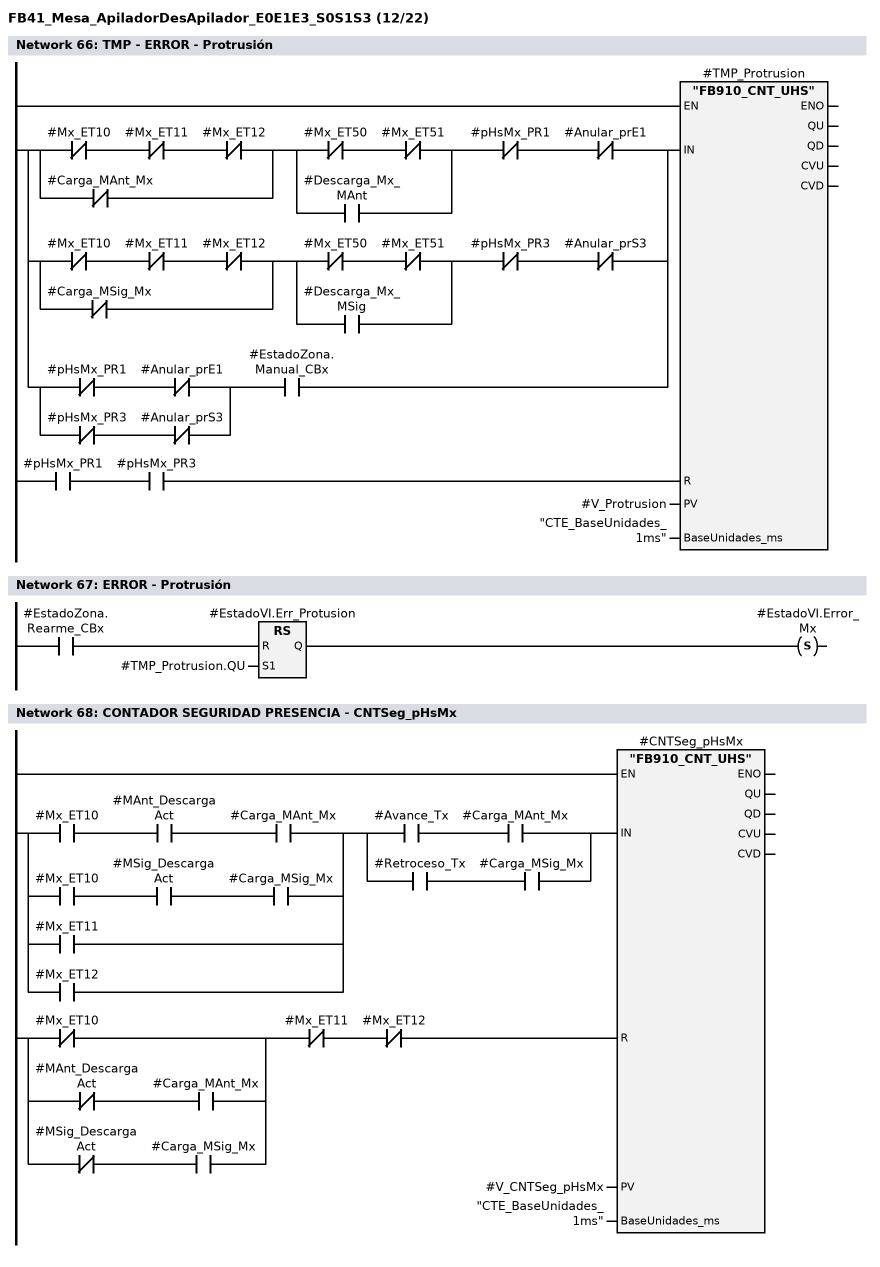
   RUNG wire#powerrail
      #TMP_Protrusion(IN := wire#w6, R := wire#w7, PV := #V_Protrusion, BaseUnidades_ms := "CTE_BaseUnidades_1ms", QU =>, QD =>, CVU =>, CVD =>)
   END_RUNG
   RUNG wire#powerrail
      I_Contact( #Mx_ET10 )
      I_Contact( #Mx_ET11 )
      I_Contact( #Mx_ET12 )
      wire#w1
      I_Contact( #Mx_ET50 )
      I_Contact( #Mx_ET51 )
      wire#w2
      I_Contact( #pHsMx_PR1 )
      I_Contact( #Anular_prE1 )
   END_RUNG wire#w6
   RUNG wire#powerrail
      I_Contact( #Carga_MAnt_Mx )
   END_RUNG wire#w1
   RUNG wire#w1
      Contact( #Descarga_Mx_MAnt )
   END_RUNG wire#w2
   RUNG wire#powerrail
      I_Contact( #Mx_ET10 )
      I_Contact( #Mx_ET11 )
      I_Contact( #Mx_ET12 )
      wire#w3
      I_Contact( #Mx_ET50 )
      I_Contact( #Mx_ET51 )
      wire#w4
      I_Contact( #pHsMx_PR3 )
      I_Contact( #Anular_prS3 )
   END_RUNG wire#w6
   RUNG wire#powerrail
      I_Contact( #Carga_MSig_Mx )
   END_RUNG wire#w3
   RUNG wire#w3
      Contact( #Descarga_Mx_MSig )
   END_RUNG wire#w4
   RUNG wire#powerrail
      I_Contact( #pHsMx_PR1 )
      I_Contact( #Anular_prE1 )
      wire#w5
      Contact( #EstadoZona.Manual_CBx )
   END_RUNG wire#w6
   RUNG wire#powerrail
      I_Contact( #pHsMx_PR3 )
      I_Contact( #Anular_prS3 )
   END_RUNG wire#w5
   RUNG wire#powerrail
      Contact( #pHsMx_PR1 )
      Contact( #pHsMx_PR3 )
   END_RUNG wire#w7
   // the same network as SCL:
   #TMP_Protrusion(IN := (((NOT #Mx_ET10 AND NOT #Mx_ET11 AND NOT #Mx_ET12) OR NOT #Carga_MAnt_Mx) AND ((NOT #Mx_ET50 AND NOT #Mx_ET51) OR #Descarga_Mx_MAnt) AND NOT #pHsMx_PR1 AND NOT #Anular_prE1) OR (((NOT #Mx_ET10 AND NOT #Mx_ET11 AND NOT #Mx_ET12) OR NOT #Carga_MSig_Mx) AND ((NOT #Mx_ET50 AND NOT #Mx_ET51) OR #Descarga_Mx_MSig) AND NOT #pHsMx_PR3 AND NOT #Anular_prS3) OR (((NOT #pHsMx_PR1 AND NOT #Anular_prE1) OR (NOT #pHsMx_PR3 AND NOT #Anular_prS3)) AND #EstadoZona.Manual_CBx),   // "FB910_CNT_UHS"
                   R := #pHsMx_PR1 AND #pHsMx_PR3,
                   PV := #V_Protrusion,
                   BaseUnidades_ms := "CTE_BaseUnidades_1ms");
END_REGION

REGION Network 67: ERROR - Protrusión
   RUNG wire#powerrail
      Contact( #EstadoZona.Rearme_CBx )
      S_RS(operand := #EstadoVI.Err_Protusion, s1 := #TMP_Protrusion.QU)
      S_Coil( #EstadoVI.Error_Mx )
   END_RUNG
   // the same network as SCL:
   IF #EstadoZona.Rearme_CBx THEN
       #EstadoVI.Err_Protusion := FALSE;   // RS flip-flop
   END_IF;
   IF #TMP_Protrusion.QU THEN #EstadoVI.Err_Protusion := TRUE; END_IF;
   IF #EstadoVI.Err_Protusion THEN #EstadoVI.Error_Mx := TRUE; END_IF;
END_REGION

REGION Network 68: CONTADOR SEGURIDAD PRESENCIA - CNTSeg_pHsMx
   RUNG wire#powerrail
      #CNTSeg_pHsMx(IN := wire#w2, R := wire#w4, PV := #V_CNTSeg_pHsMx, BaseUnidades_ms := "CTE_BaseUnidades_1ms", QU =>, QD =>, CVU =>, CVD =>)
   END_RUNG
   RUNG wire#powerrail
      Contact( #Mx_ET10 )
      Contact( #MAnt_DescargaAct )
      Contact( #Carga_MAnt_Mx )
      wire#w1
      Contact( #Avance_Tx )
      Contact( #Carga_MAnt_Mx )
   END_RUNG wire#w2
   RUNG wire#powerrail
      Contact( #Mx_ET10 )
      Contact( #MSig_DescargaAct )
      Contact( #Carga_MSig_Mx )
   END_RUNG wire#w1
   RUNG wire#powerrail
      Contact( #Mx_ET11 )
   END_RUNG wire#w1
   RUNG wire#powerrail
      Contact( #Mx_ET12 )
   END_RUNG wire#w1
   RUNG wire#w1
      Contact( #Retroceso_Tx )
      Contact( #Carga_MSig_Mx )
   END_RUNG wire#w2
   RUNG wire#powerrail
      I_Contact( #Mx_ET10 )
      wire#w3
      I_Contact( #Mx_ET11 )
      I_Contact( #Mx_ET12 )
   END_RUNG wire#w4
   RUNG wire#powerrail
      I_Contact( #MAnt_DescargaAct )
      Contact( #Carga_MAnt_Mx )
   END_RUNG wire#w3
   RUNG wire#powerrail
      I_Contact( #MSig_DescargaAct )
      Contact( #Carga_MSig_Mx )
   END_RUNG wire#w3
   // the same network as SCL:
   #CNTSeg_pHsMx(IN := ((#Mx_ET10 AND #MAnt_DescargaAct AND #Carga_MAnt_Mx) OR (#Mx_ET10 AND #MSig_DescargaAct AND #Carga_MSig_Mx) OR #Mx_ET11 OR #Mx_ET12) AND ((#Avance_Tx AND #Carga_MAnt_Mx) OR (#Retroceso_Tx AND #Carga_MSig_Mx)),   // "FB910_CNT_UHS"
                 R := (NOT #Mx_ET10 OR (NOT #MAnt_DescargaAct AND #Carga_MAnt_Mx) OR (NOT #MSig_DescargaAct AND #Carga_MSig_Mx)) AND NOT #Mx_ET11 AND NOT #Mx_ET12,
                 PV := #V_CNTSeg_pHsMx,
                 BaseUnidades_ms := "CTE_BaseUnidades_1ms");
END_REGION

REGION Network 69: CONTADOR DE PRESENCIA - CNT_pHsMx
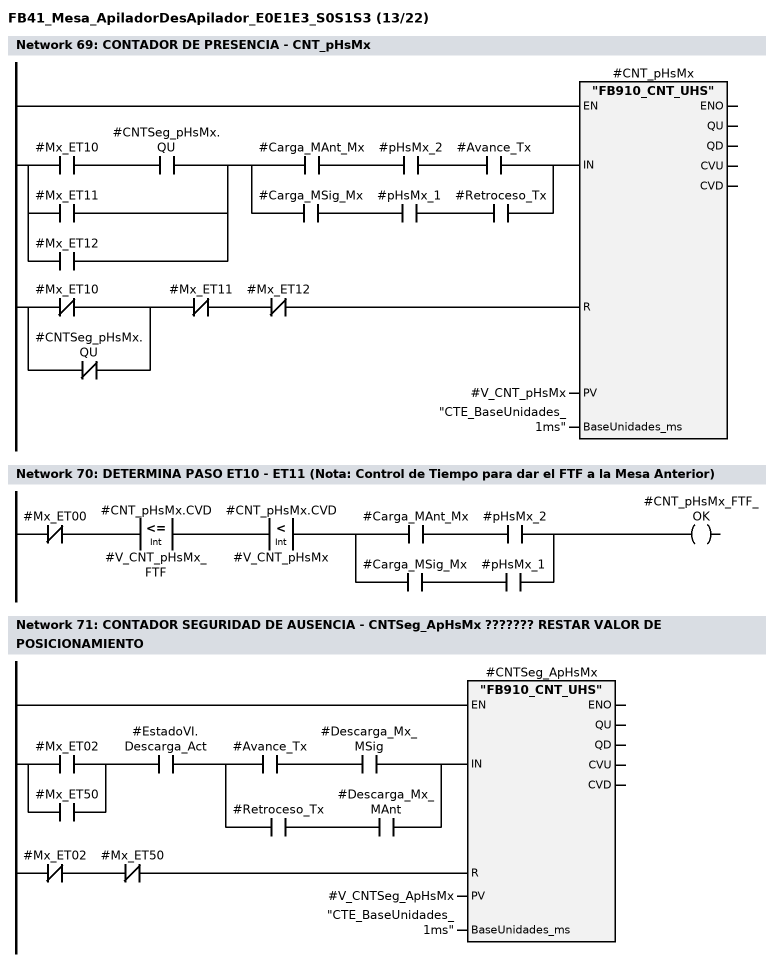
   RUNG wire#powerrail
      #CNT_pHsMx(IN := wire#w2, R := wire#w4, PV := #V_CNT_pHsMx, BaseUnidades_ms := "CTE_BaseUnidades_1ms", QU =>, QD =>, CVU =>, CVD =>)
   END_RUNG
   RUNG wire#powerrail
      Contact( #Mx_ET10 )
      Contact( #CNTSeg_pHsMx.QU )
      wire#w1
      Contact( #Carga_MAnt_Mx )
      Contact( #pHsMx_2 )
      Contact( #Avance_Tx )
   END_RUNG wire#w2
   RUNG wire#powerrail
      Contact( #Mx_ET11 )
   END_RUNG wire#w1
   RUNG wire#powerrail
      Contact( #Mx_ET12 )
   END_RUNG wire#w1
   RUNG wire#w1
      Contact( #Carga_MSig_Mx )
      Contact( #pHsMx_1 )
      Contact( #Retroceso_Tx )
   END_RUNG wire#w2
   RUNG wire#powerrail
      I_Contact( #Mx_ET10 )
      wire#w3
      I_Contact( #Mx_ET11 )
      I_Contact( #Mx_ET12 )
   END_RUNG wire#w4
   RUNG wire#powerrail
      I_Contact( #CNTSeg_pHsMx.QU )
   END_RUNG wire#w3
   // the same network as SCL:
   #CNT_pHsMx(IN := ((#Mx_ET10 AND #CNTSeg_pHsMx.QU) OR #Mx_ET11 OR #Mx_ET12) AND ((#Carga_MAnt_Mx AND #pHsMx_2 AND #Avance_Tx) OR (#Carga_MSig_Mx AND #pHsMx_1 AND #Retroceso_Tx)),   // "FB910_CNT_UHS"
              R := (NOT #Mx_ET10 OR NOT #CNTSeg_pHsMx.QU) AND NOT #Mx_ET11 AND NOT #Mx_ET12,
              PV := #V_CNT_pHsMx,
              BaseUnidades_ms := "CTE_BaseUnidades_1ms");
END_REGION

REGION Network 70: DETERMINA PASO ET10 - ET11 (Nota: Control de Tiempo para dar el FTF a la Mesa Anterior)
   RUNG wire#powerrail
      I_Contact( #Mx_ET00 )
      { S7_Templates := "SrcType := Int" } LE_Contact(in1 := #CNT_pHsMx.CVD, in2 := #V_CNT_pHsMx_FTF)
      { S7_Templates := "SrcType := Int" } LT_Contact(in1 := #CNT_pHsMx.CVD, in2 := #V_CNT_pHsMx)
      wire#w1
      Contact( #Carga_MAnt_Mx )
      Contact( #pHsMx_2 )
      wire#w2
      Coil( #CNT_pHsMx_FTF_OK )
   END_RUNG
   RUNG wire#w1
      Contact( #Carga_MSig_Mx )
      Contact( #pHsMx_1 )
   END_RUNG wire#w2
   // the same network as SCL:
   #CNT_pHsMx_FTF_OK := NOT #Mx_ET00 AND (#CNT_pHsMx.CVD <= #V_CNT_pHsMx_FTF) AND (#CNT_pHsMx.CVD < #V_CNT_pHsMx) AND ((#Carga_MAnt_Mx AND #pHsMx_2) OR (#Carga_MSig_Mx AND #pHsMx_1));
END_REGION

REGION Network 71: CONTADOR SEGURIDAD DE AUSENCIA - CNTSeg_ApHsMx ??????? RESTAR VALOR DE POSICIONAMIENTO
   RUNG wire#powerrail
      #CNTSeg_ApHsMx(IN := wire#w3, R := wire#w4, PV := #V_CNTSeg_ApHsMx, BaseUnidades_ms := "CTE_BaseUnidades_1ms", QU =>, QD =>, CVU =>, CVD =>)
   END_RUNG
   RUNG wire#powerrail
      Contact( #Mx_ET02 )
      wire#w1
      Contact( #EstadoVI.Descarga_Act )
      wire#w2
      Contact( #Avance_Tx )
      Contact( #Descarga_Mx_MSig )
   END_RUNG wire#w3
   RUNG wire#powerrail
      Contact( #Mx_ET50 )
   END_RUNG wire#w1
   RUNG wire#w2
      Contact( #Retroceso_Tx )
      Contact( #Descarga_Mx_MAnt )
   END_RUNG wire#w3
   RUNG wire#powerrail
      I_Contact( #Mx_ET02 )
      I_Contact( #Mx_ET50 )
   END_RUNG wire#w4
   // the same network as SCL:
   #CNTSeg_ApHsMx(IN := (#Mx_ET02 OR #Mx_ET50) AND #EstadoVI.Descarga_Act AND ((#Avance_Tx AND #Descarga_Mx_MSig) OR (#Retroceso_Tx AND #Descarga_Mx_MAnt)),   // "FB910_CNT_UHS"
                  R := NOT #Mx_ET02 AND NOT #Mx_ET50,
                  PV := #V_CNTSeg_ApHsMx,
                  BaseUnidades_ms := "CTE_BaseUnidades_1ms");
END_REGION

REGION Network 72: CONTADOR DE LA AUSENCIA - CNT_ApHsMX
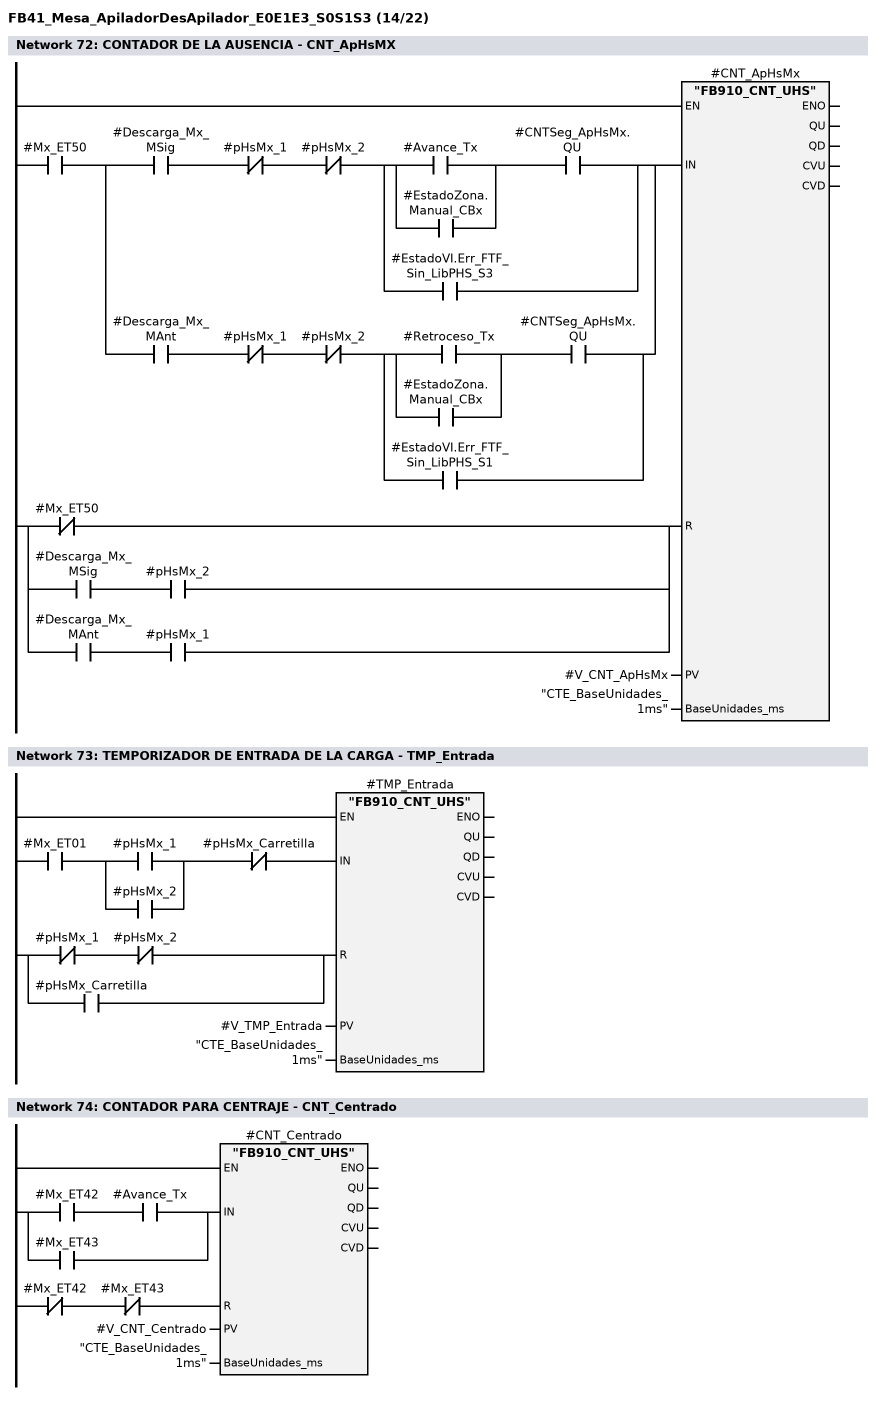
   RUNG wire#powerrail
      #CNT_ApHsMx(IN := wire#w6, R := wire#w7, PV := #V_CNT_ApHsMx, BaseUnidades_ms := "CTE_BaseUnidades_1ms", QU =>, QD =>, CVU =>, CVD =>)
   END_RUNG
   RUNG wire#powerrail
      Contact( #Mx_ET50 )
      wire#w1
      Contact( #Descarga_Mx_MSig )
      I_Contact( #pHsMx_1 )
      I_Contact( #pHsMx_2 )
      wire#w2
      Contact( #Avance_Tx )
      wire#w3
      Contact( #CNTSeg_ApHsMx.QU )
   END_RUNG wire#w6
   RUNG wire#w2
      Contact( #EstadoZona.Manual_CBx )
   END_RUNG wire#w3
   RUNG wire#w2
      Contact( #EstadoVI.Err_FTF_Sin_LibPHS_S3 )
   END_RUNG wire#w6
   RUNG wire#w1
      Contact( #Descarga_Mx_MAnt )
      I_Contact( #pHsMx_1 )
      I_Contact( #pHsMx_2 )
      wire#w4
      Contact( #Retroceso_Tx )
      wire#w5
      Contact( #CNTSeg_ApHsMx.QU )
   END_RUNG wire#w6
   RUNG wire#w4
      Contact( #EstadoZona.Manual_CBx )
   END_RUNG wire#w5
   RUNG wire#w4
      Contact( #EstadoVI.Err_FTF_Sin_LibPHS_S1 )
   END_RUNG wire#w6
   RUNG wire#powerrail
      I_Contact( #Mx_ET50 )
   END_RUNG wire#w7
   RUNG wire#powerrail
      Contact( #Descarga_Mx_MSig )
      Contact( #pHsMx_2 )
   END_RUNG wire#w7
   RUNG wire#powerrail
      Contact( #Descarga_Mx_MAnt )
      Contact( #pHsMx_1 )
   END_RUNG wire#w7
   // the same network as SCL:
   #CNT_ApHsMx(IN := #Mx_ET50 AND ((#Descarga_Mx_MSig AND NOT #pHsMx_1 AND NOT #pHsMx_2 AND (((#Avance_Tx OR #EstadoZona.Manual_CBx) AND #CNTSeg_ApHsMx.QU) OR #EstadoVI.Err_FTF_Sin_LibPHS_S3)) OR (#Descarga_Mx_MAnt AND NOT #pHsMx_1 AND NOT #pHsMx_2 AND (((#Retroceso_Tx OR #EstadoZona.Manual_CBx) AND #CNTSeg_ApHsMx.QU) OR #EstadoVI.Err_FTF_Sin_LibPHS_S1))),   // "FB910_CNT_UHS"
               R := NOT #Mx_ET50 OR (#Descarga_Mx_MSig AND #pHsMx_2) OR (#Descarga_Mx_MAnt AND #pHsMx_1),
               PV := #V_CNT_ApHsMx,
               BaseUnidades_ms := "CTE_BaseUnidades_1ms");
END_REGION

REGION Network 73: TEMPORIZADOR DE ENTRADA DE LA CARGA - TMP_Entrada
   RUNG wire#powerrail
      #TMP_Entrada(IN := wire#w3, R := wire#w4, PV := #V_TMP_Entrada, BaseUnidades_ms := "CTE_BaseUnidades_1ms", QU =>, QD =>, CVU =>, CVD =>)
   END_RUNG
   RUNG wire#powerrail
      Contact( #Mx_ET01 )
      wire#w1
      Contact( #pHsMx_1 )
      wire#w2
      I_Contact( #pHsMx_Carretilla )
   END_RUNG wire#w3
   RUNG wire#w1
      Contact( #pHsMx_2 )
   END_RUNG wire#w2
   RUNG wire#powerrail
      I_Contact( #pHsMx_1 )
      I_Contact( #pHsMx_2 )
   END_RUNG wire#w4
   RUNG wire#powerrail
      Contact( #pHsMx_Carretilla )
   END_RUNG wire#w4
   // the same network as SCL:
   #TMP_Entrada(IN := #Mx_ET01 AND (#pHsMx_1 OR #pHsMx_2) AND NOT #pHsMx_Carretilla,   // "FB910_CNT_UHS"
                R := (NOT #pHsMx_1 AND NOT #pHsMx_2) OR #pHsMx_Carretilla,
                PV := #V_TMP_Entrada,
                BaseUnidades_ms := "CTE_BaseUnidades_1ms");
END_REGION

REGION Network 74: CONTADOR PARA CENTRAJE - CNT_Centrado
   RUNG wire#powerrail
      #CNT_Centrado(IN := wire#w1, R := wire#w2, PV := #V_CNT_Centrado, BaseUnidades_ms := "CTE_BaseUnidades_1ms", QU =>, QD =>, CVU =>, CVD =>)
   END_RUNG
   RUNG wire#powerrail
      Contact( #Mx_ET42 )
      Contact( #Avance_Tx )
   END_RUNG wire#w1
   RUNG wire#powerrail
      Contact( #Mx_ET43 )
   END_RUNG wire#w1
   RUNG wire#powerrail
      I_Contact( #Mx_ET42 )
      I_Contact( #Mx_ET43 )
   END_RUNG wire#w2
   // the same network as SCL:
   #CNT_Centrado(IN := (#Mx_ET42 AND #Avance_Tx) OR #Mx_ET43,   // "FB910_CNT_UHS"
                 R := NOT #Mx_ET42 AND NOT #Mx_ET43,
                 PV := #V_CNT_Centrado,
                 BaseUnidades_ms := "CTE_BaseUnidades_1ms");
END_REGION

REGION Network 75: TEMPORIZADOR DE RETIRADA DE LA CARGA - TMP_Retirada
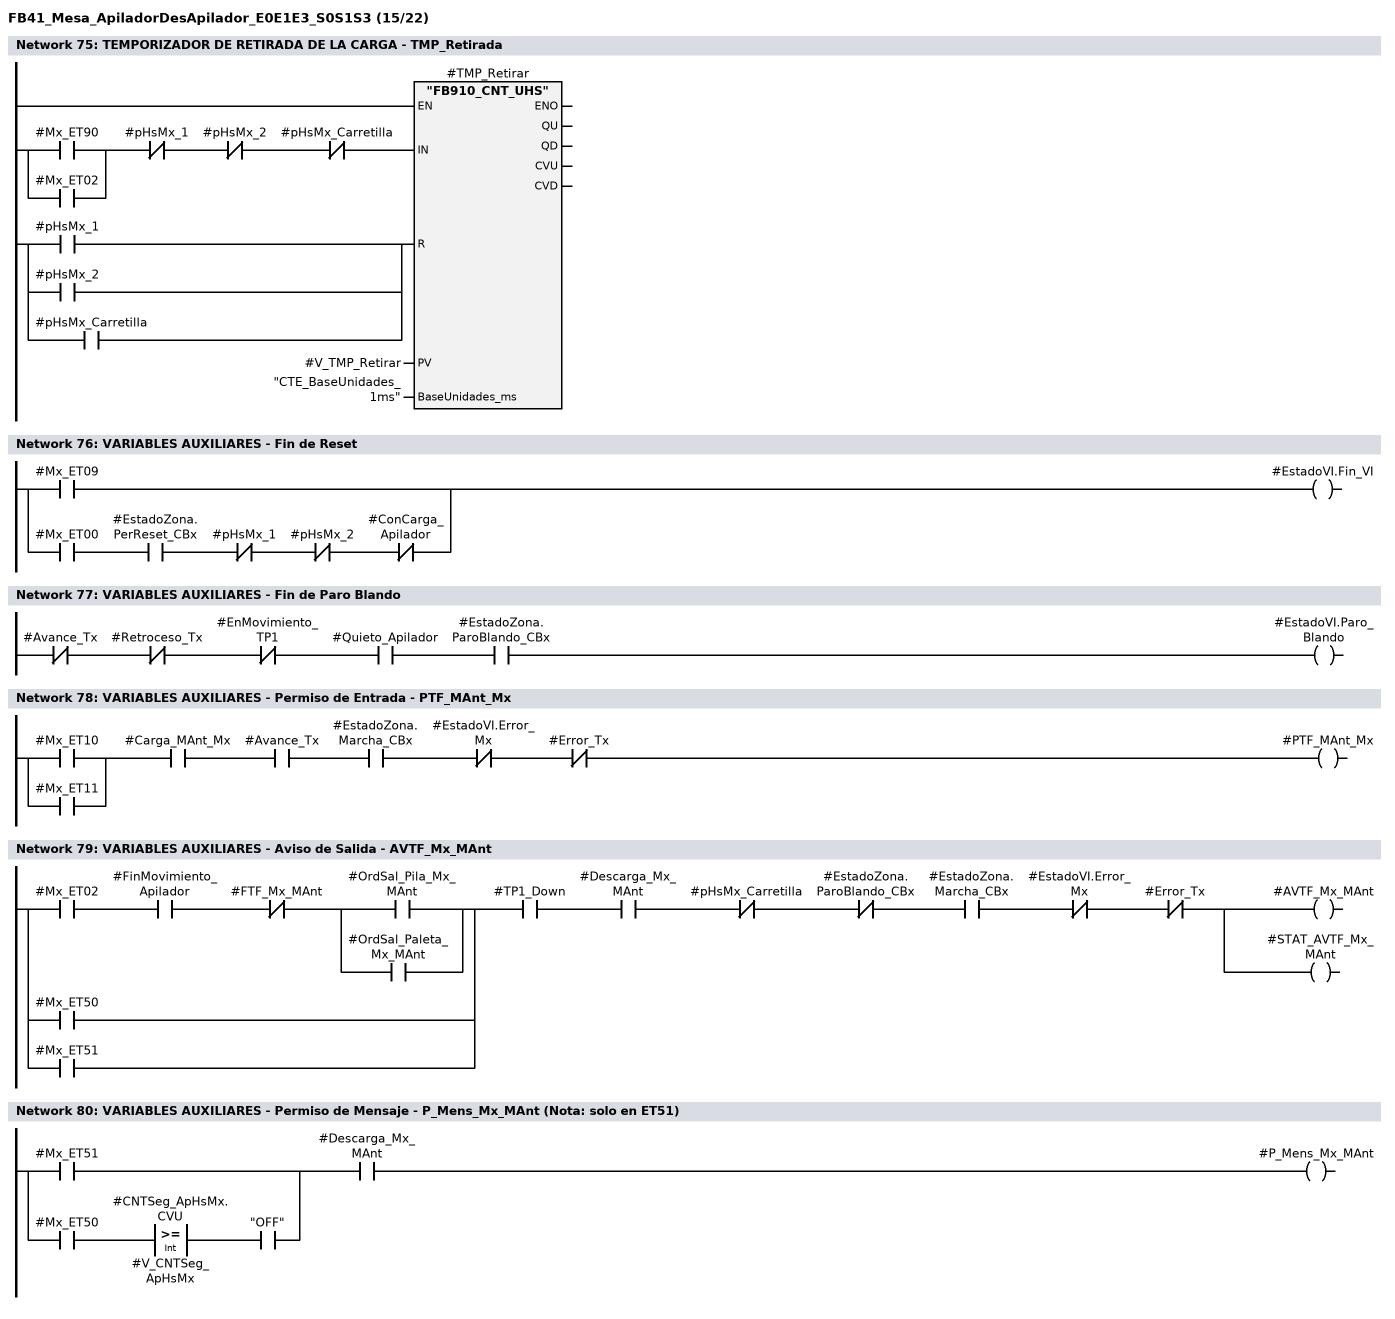
   RUNG wire#powerrail
      #TMP_Retirar(IN := wire#w2, R := wire#w3, PV := #V_TMP_Retirar, BaseUnidades_ms := "CTE_BaseUnidades_1ms", QU =>, QD =>, CVU =>, CVD =>)
   END_RUNG
   RUNG wire#powerrail
      Contact( #Mx_ET90 )
      wire#w1
      I_Contact( #pHsMx_1 )
      I_Contact( #pHsMx_2 )
      I_Contact( #pHsMx_Carretilla )
   END_RUNG wire#w2
   RUNG wire#powerrail
      Contact( #Mx_ET02 )
   END_RUNG wire#w1
   RUNG wire#powerrail
      Contact( #pHsMx_1 )
   END_RUNG wire#w3
   RUNG wire#powerrail
      Contact( #pHsMx_2 )
   END_RUNG wire#w3
   RUNG wire#powerrail
      Contact( #pHsMx_Carretilla )
   END_RUNG wire#w3
   // the same network as SCL:
   #TMP_Retirar(IN := (#Mx_ET90 OR #Mx_ET02) AND NOT #pHsMx_1 AND NOT #pHsMx_2 AND NOT #pHsMx_Carretilla,   // "FB910_CNT_UHS"
                R := #pHsMx_1 OR #pHsMx_2 OR #pHsMx_Carretilla,
                PV := #V_TMP_Retirar,
                BaseUnidades_ms := "CTE_BaseUnidades_1ms");
END_REGION

REGION Network 76: VARIABLES AUXILIARES - Fin de Reset
   RUNG wire#powerrail
      Contact( #Mx_ET09 )
      wire#w1
      Coil( #EstadoVI.Fin_VI )
   END_RUNG
   RUNG wire#powerrail
      Contact( #Mx_ET00 )
      Contact( #EstadoZona.PerReset_CBx )
      I_Contact( #pHsMx_1 )
      I_Contact( #pHsMx_2 )
      I_Contact( #ConCarga_Apilador )
   END_RUNG wire#w1
   // the same network as SCL:
   #EstadoVI.Fin_VI := #Mx_ET09 OR (#Mx_ET00 AND #EstadoZona.PerReset_CBx AND NOT #pHsMx_1 AND NOT #pHsMx_2 AND NOT #ConCarga_Apilador);
END_REGION

REGION Network 77: VARIABLES AUXILIARES - Fin de Paro Blando
   RUNG wire#powerrail
      I_Contact( #Avance_Tx )
      I_Contact( #Retroceso_Tx )
      I_Contact( #EnMovimiento_TP1 )
      Contact( #Quieto_Apilador )
      Contact( #EstadoZona.ParoBlando_CBx )
      Coil( #EstadoVI.Paro_Blando )
   END_RUNG
   // the same network as SCL:
   #EstadoVI.Paro_Blando := NOT #Avance_Tx AND NOT #Retroceso_Tx AND NOT #EnMovimiento_TP1 AND #Quieto_Apilador AND #EstadoZona.ParoBlando_CBx;
END_REGION

REGION Network 78: VARIABLES AUXILIARES - Permiso de Entrada - PTF_MAnt_Mx
   RUNG wire#powerrail
      Contact( #Mx_ET10 )
      wire#w1
      Contact( #Carga_MAnt_Mx )
      Contact( #Avance_Tx )
      Contact( #EstadoZona.Marcha_CBx )
      I_Contact( #EstadoVI.Error_Mx )
      I_Contact( #Error_Tx )
      Coil( #PTF_MAnt_Mx )
   END_RUNG
   RUNG wire#powerrail
      Contact( #Mx_ET11 )
   END_RUNG wire#w1
   // the same network as SCL:
   #PTF_MAnt_Mx := (#Mx_ET10 OR #Mx_ET11) AND #Carga_MAnt_Mx AND #Avance_Tx AND #EstadoZona.Marcha_CBx AND NOT #EstadoVI.Error_Mx AND NOT #Error_Tx;
END_REGION

REGION Network 79: VARIABLES AUXILIARES - Aviso de Salida - AVTF_Mx_MAnt
   RUNG wire#powerrail
      Contact( #Mx_ET02 )
      Contact( #FinMovimiento_Apilador )
      I_Contact( #FTF_Mx_MAnt )
      wire#w1
      Contact( #OrdSal_Pila_Mx_MAnt )
      wire#w2
      Contact( #TP1_Down )
      Contact( #Descarga_Mx_MAnt )
      I_Contact( #pHsMx_Carretilla )
      I_Contact( #EstadoZona.ParoBlando_CBx )
      Contact( #EstadoZona.Marcha_CBx )
      I_Contact( #EstadoVI.Error_Mx )
      I_Contact( #Error_Tx )
      wire#w3
      Coil( #AVTF_Mx_MAnt )
   END_RUNG
   RUNG wire#w1
      Contact( #OrdSal_Paleta_Mx_MAnt )
   END_RUNG wire#w2
   RUNG wire#powerrail
      Contact( #Mx_ET50 )
   END_RUNG wire#w2
   RUNG wire#powerrail
      Contact( #Mx_ET51 )
   END_RUNG wire#w2
   RUNG wire#w3
      Coil( #STAT_AVTF_Mx_MAnt )
   END_RUNG
   // the same network as SCL:
   #AVTF_Mx_MAnt := ((#Mx_ET02 AND #FinMovimiento_Apilador AND NOT #FTF_Mx_MAnt AND (#OrdSal_Pila_Mx_MAnt OR #OrdSal_Paleta_Mx_MAnt)) OR #Mx_ET50 OR #Mx_ET51) AND #TP1_Down AND #Descarga_Mx_MAnt AND NOT #pHsMx_Carretilla AND NOT #EstadoZona.ParoBlando_CBx AND #EstadoZona.Marcha_CBx AND NOT #EstadoVI.Error_Mx AND NOT #Error_Tx;
   #STAT_AVTF_Mx_MAnt := #AVTF_Mx_MAnt;
END_REGION

REGION Network 80: VARIABLES AUXILIARES - Permiso de Mensaje - P_Mens_Mx_MAnt (Nota: solo en ET51)
   RUNG wire#powerrail
      Contact( #Mx_ET51 )
      wire#w1
      Contact( #Descarga_Mx_MAnt )
      Coil( #P_Mens_Mx_MAnt )
   END_RUNG
   RUNG wire#powerrail
      Contact( #Mx_ET50 )
      { S7_Templates := "SrcType := Int" } GE_Contact(in1 := #CNTSeg_ApHsMx.CVU, in2 := #V_CNTSeg_ApHsMx)
      Contact( "OFF" )
   END_RUNG wire#w1
   // the same network as SCL:
   #P_Mens_Mx_MAnt := (#Mx_ET51 OR (#Mx_ET50 AND (#CNTSeg_ApHsMx.CVU >= #V_CNTSeg_ApHsMx) AND "OFF")) AND #Descarga_Mx_MAnt;
END_REGION

REGION Network 81: VARIABLES AUXILIARES - Permiso de Entrada - PTF_MSig_Mx
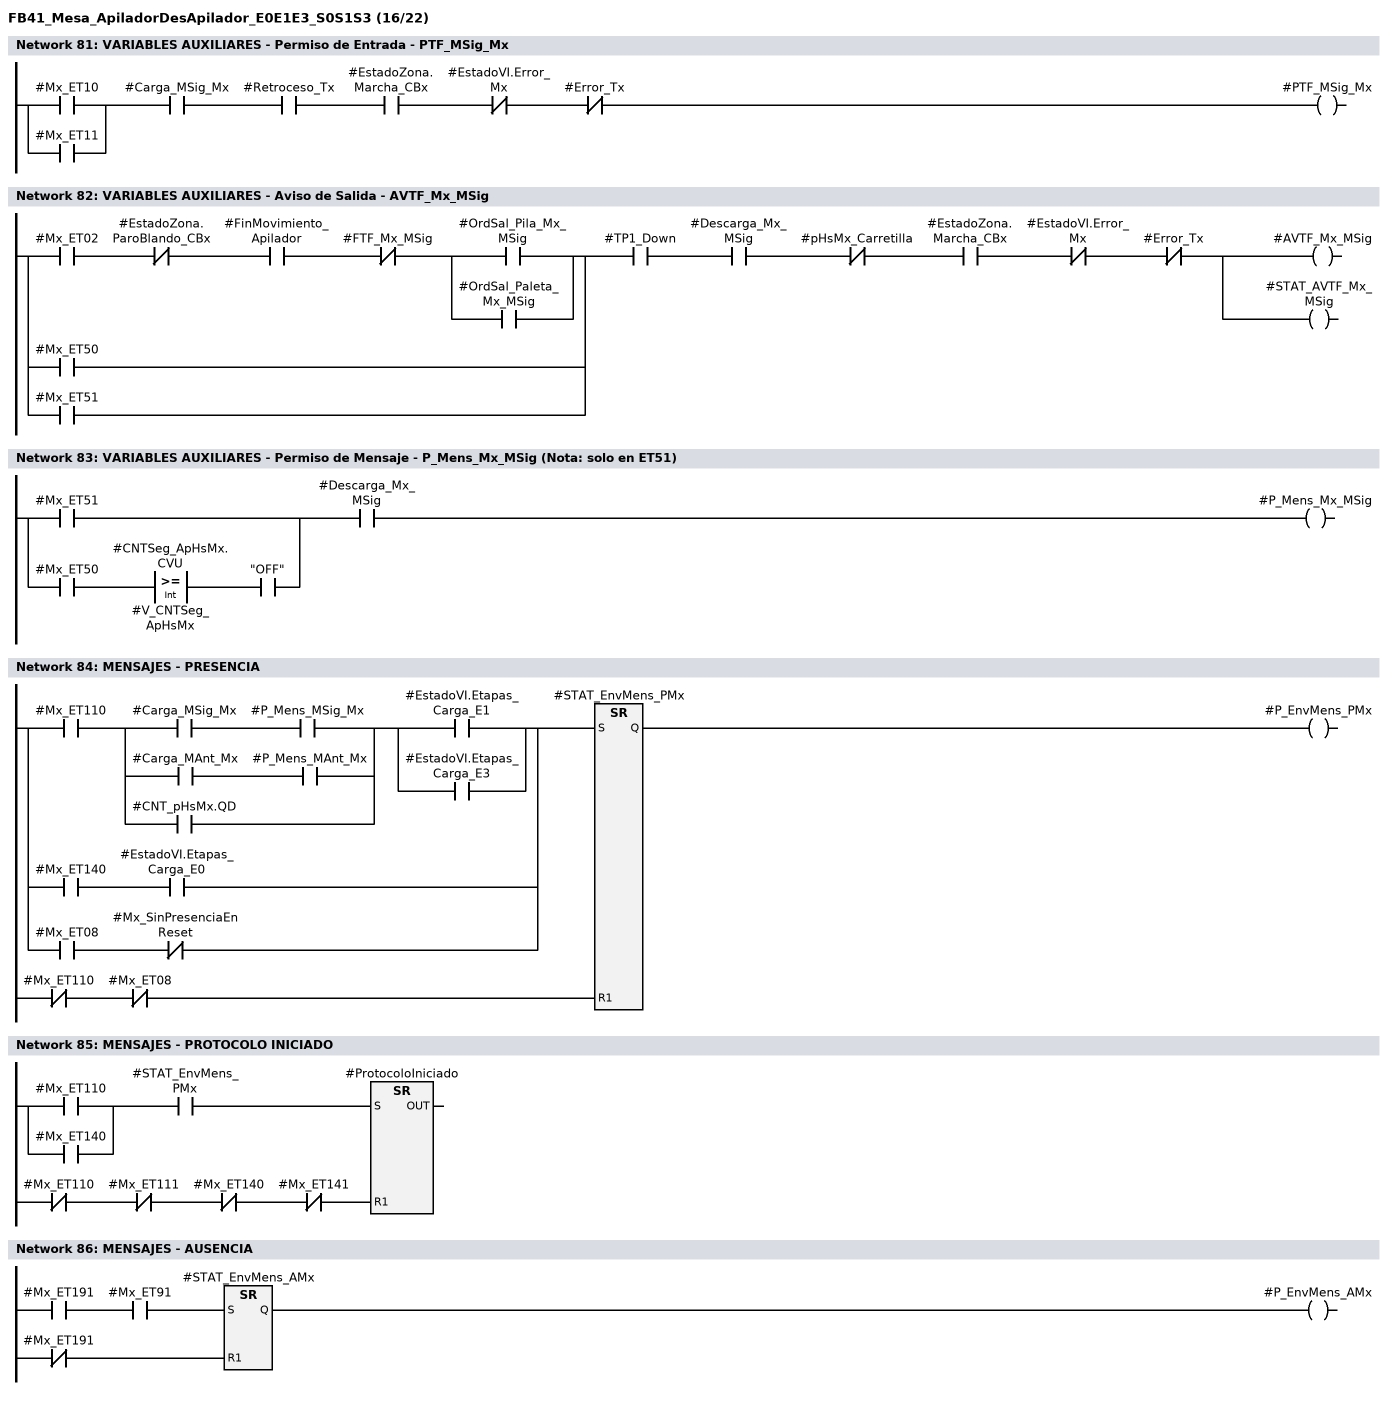
   RUNG wire#powerrail
      Contact( #Mx_ET10 )
      wire#w1
      Contact( #Carga_MSig_Mx )
      Contact( #Retroceso_Tx )
      Contact( #EstadoZona.Marcha_CBx )
      I_Contact( #EstadoVI.Error_Mx )
      I_Contact( #Error_Tx )
      Coil( #PTF_MSig_Mx )
   END_RUNG
   RUNG wire#powerrail
      Contact( #Mx_ET11 )
   END_RUNG wire#w1
   // the same network as SCL:
   #PTF_MSig_Mx := (#Mx_ET10 OR #Mx_ET11) AND #Carga_MSig_Mx AND #Retroceso_Tx AND #EstadoZona.Marcha_CBx AND NOT #EstadoVI.Error_Mx AND NOT #Error_Tx;
END_REGION

REGION Network 82: VARIABLES AUXILIARES - Aviso de Salida - AVTF_Mx_MSig
   RUNG wire#powerrail
      Contact( #Mx_ET02 )
      I_Contact( #EstadoZona.ParoBlando_CBx )
      Contact( #FinMovimiento_Apilador )
      I_Contact( #FTF_Mx_MSig )
      wire#w1
      Contact( #OrdSal_Pila_Mx_MSig )
      wire#w2
      Contact( #TP1_Down )
      Contact( #Descarga_Mx_MSig )
      I_Contact( #pHsMx_Carretilla )
      Contact( #EstadoZona.Marcha_CBx )
      I_Contact( #EstadoVI.Error_Mx )
      I_Contact( #Error_Tx )
      wire#w3
      Coil( #AVTF_Mx_MSig )
   END_RUNG
   RUNG wire#w1
      Contact( #OrdSal_Paleta_Mx_MSig )
   END_RUNG wire#w2
   RUNG wire#powerrail
      Contact( #Mx_ET50 )
   END_RUNG wire#w2
   RUNG wire#powerrail
      Contact( #Mx_ET51 )
   END_RUNG wire#w2
   RUNG wire#w3
      Coil( #STAT_AVTF_Mx_MSig )
   END_RUNG
   // the same network as SCL:
   #AVTF_Mx_MSig := ((#Mx_ET02 AND NOT #EstadoZona.ParoBlando_CBx AND #FinMovimiento_Apilador AND NOT #FTF_Mx_MSig AND (#OrdSal_Pila_Mx_MSig OR #OrdSal_Paleta_Mx_MSig)) OR #Mx_ET50 OR #Mx_ET51) AND #TP1_Down AND #Descarga_Mx_MSig AND NOT #pHsMx_Carretilla AND #EstadoZona.Marcha_CBx AND NOT #EstadoVI.Error_Mx AND NOT #Error_Tx;
   #STAT_AVTF_Mx_MSig := #AVTF_Mx_MSig;
END_REGION

REGION Network 83: VARIABLES AUXILIARES - Permiso de Mensaje - P_Mens_Mx_MSig (Nota: solo en ET51)
   RUNG wire#powerrail
      Contact( #Mx_ET51 )
      wire#w1
      Contact( #Descarga_Mx_MSig )
      Coil( #P_Mens_Mx_MSig )
   END_RUNG
   RUNG wire#powerrail
      Contact( #Mx_ET50 )
      { S7_Templates := "SrcType := Int" } GE_Contact(in1 := #CNTSeg_ApHsMx.CVU, in2 := #V_CNTSeg_ApHsMx)
      Contact( "OFF" )
   END_RUNG wire#w1
   // the same network as SCL:
   #P_Mens_Mx_MSig := (#Mx_ET51 OR (#Mx_ET50 AND (#CNTSeg_ApHsMx.CVU >= #V_CNTSeg_ApHsMx) AND "OFF")) AND #Descarga_Mx_MSig;
END_REGION

REGION Network 84: MENSAJES - PRESENCIA
   RUNG wire#powerrail
      Contact( #Mx_ET110 )
      wire#w1
      Contact( #Carga_MSig_Mx )
      Contact( #P_Mens_MSig_Mx )
      wire#w2
      Contact( #EstadoVI.Etapas_Carga_E1 )
      wire#w3
      S_SR(operand := #STAT_EnvMens_PMx, r1 := wire#w4)
      Coil( #P_EnvMens_PMx )
   END_RUNG
   RUNG wire#w1
      Contact( #Carga_MAnt_Mx )
      Contact( #P_Mens_MAnt_Mx )
   END_RUNG wire#w2
   RUNG wire#w1
      Contact( #CNT_pHsMx.QD )
   END_RUNG wire#w2
   RUNG wire#w2
      Contact( #EstadoVI.Etapas_Carga_E3 )
   END_RUNG wire#w3
   RUNG wire#powerrail
      Contact( #Mx_ET140 )
      Contact( #EstadoVI.Etapas_Carga_E0 )
   END_RUNG wire#w3
   RUNG wire#powerrail
      Contact( #Mx_ET08 )
      I_Contact( #Mx_SinPresenciaEnReset )
   END_RUNG wire#w3
   RUNG wire#powerrail
      I_Contact( #Mx_ET110 )
      I_Contact( #Mx_ET08 )
   END_RUNG wire#w4
   // the same network as SCL:
   IF (#Mx_ET110 AND ((#Carga_MSig_Mx AND #P_Mens_MSig_Mx) OR (#Carga_MAnt_Mx AND #P_Mens_MAnt_Mx) OR #CNT_pHsMx.QD) AND (#EstadoVI.Etapas_Carga_E1 OR #EstadoVI.Etapas_Carga_E3)) OR (#Mx_ET140 AND #EstadoVI.Etapas_Carga_E0) OR (#Mx_ET08 AND NOT #Mx_SinPresenciaEnReset) THEN
       #STAT_EnvMens_PMx := TRUE;   // SR flip-flop
   END_IF;
   IF NOT #Mx_ET110 AND NOT #Mx_ET08 THEN #STAT_EnvMens_PMx := FALSE; END_IF;
   #P_EnvMens_PMx := #STAT_EnvMens_PMx;
END_REGION

REGION Network 85: MENSAJES - PROTOCOLO INICIADO
   RUNG wire#powerrail
      Contact( #Mx_ET110 )
      wire#w1
      Contact( #STAT_EnvMens_PMx )
      S_SR(operand := #ProtocoloIniciado, r1 := wire#w2)
   END_RUNG
   RUNG wire#powerrail
      Contact( #Mx_ET140 )
   END_RUNG wire#w1
   RUNG wire#powerrail
      I_Contact( #Mx_ET110 )
      I_Contact( #Mx_ET111 )
      I_Contact( #Mx_ET140 )
      I_Contact( #Mx_ET141 )
   END_RUNG wire#w2
   // the same network as SCL:
   IF (#Mx_ET110 OR #Mx_ET140) AND #STAT_EnvMens_PMx THEN
       #ProtocoloIniciado := TRUE;   // SR flip-flop
   END_IF;
   IF NOT #Mx_ET110 AND NOT #Mx_ET111 AND NOT #Mx_ET140 AND NOT #Mx_ET141 THEN
       #ProtocoloIniciado := FALSE;
   END_IF;
END_REGION

REGION Network 86: MENSAJES - AUSENCIA
   RUNG wire#powerrail
      Contact( #Mx_ET191 )
      Contact( #Mx_ET91 )
      S_SR(operand := #STAT_EnvMens_AMx, r1 := wire#w1)
      Coil( #P_EnvMens_AMx )
   END_RUNG
   RUNG wire#powerrail
      I_Contact( #Mx_ET191 )
   END_RUNG wire#w1
   // the same network as SCL:
   IF #Mx_ET191 AND #Mx_ET91 THEN
       #STAT_EnvMens_AMx := TRUE;   // SR flip-flop
   END_IF;
   IF NOT #Mx_ET191 THEN #STAT_EnvMens_AMx := FALSE; END_IF;
   #P_EnvMens_AMx := #STAT_EnvMens_AMx;
END_REGION

REGION Network 87: MENSAJES - RECIBIDA LA ORDEN
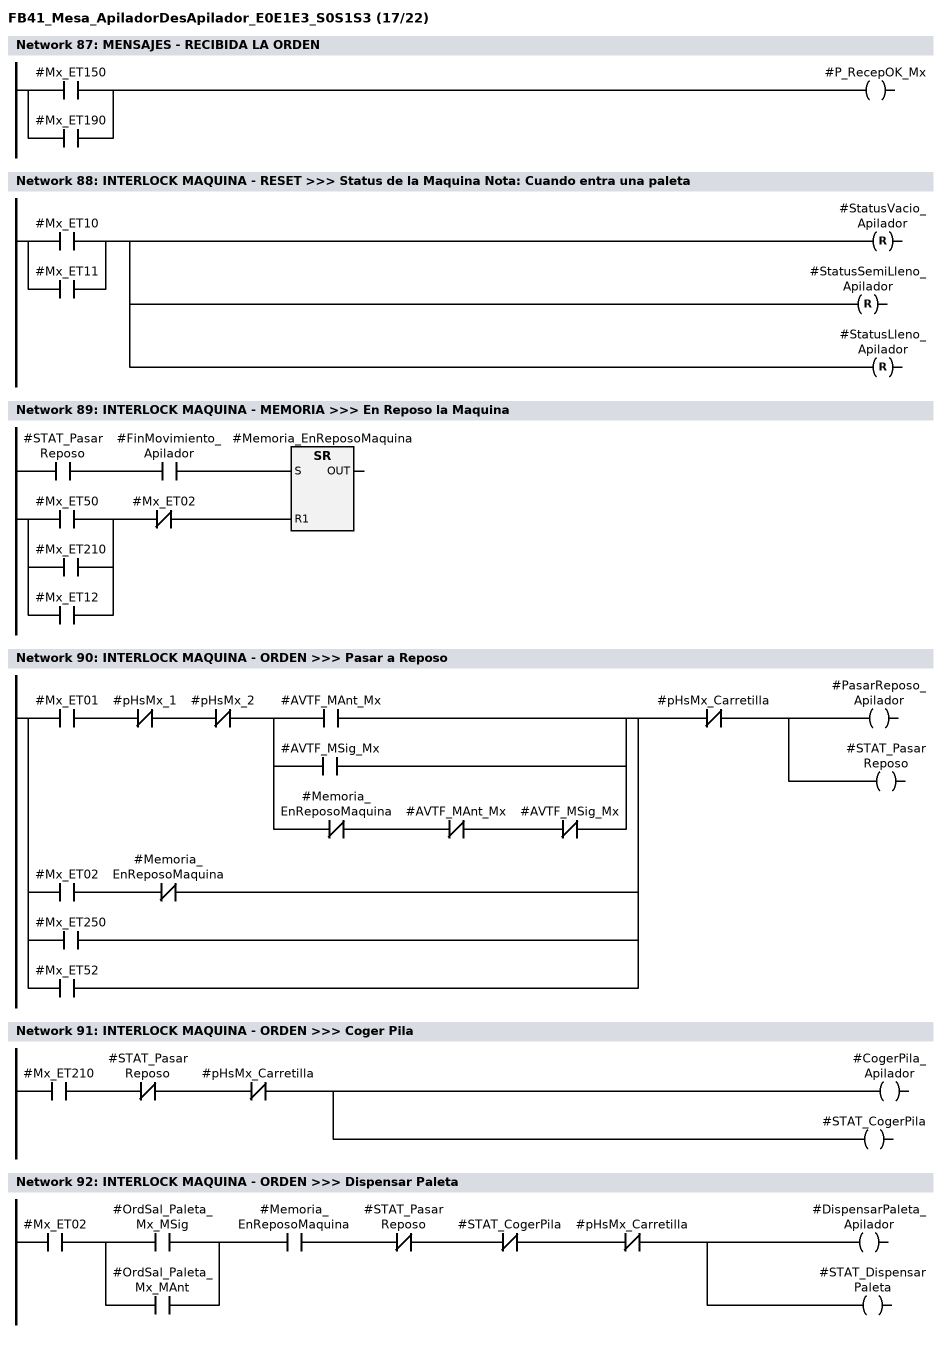
   RUNG wire#powerrail
      Contact( #Mx_ET150 )
      wire#w1
      Coil( #P_RecepOK_Mx )
   END_RUNG
   RUNG wire#powerrail
      Contact( #Mx_ET190 )
   END_RUNG wire#w1
   // the same network as SCL:
   #P_RecepOK_Mx := #Mx_ET150 OR #Mx_ET190;
END_REGION

REGION Network 88: INTERLOCK MAQUINA - RESET >>> Status de la Maquina Nota: Cuando entra una paleta
   RUNG wire#powerrail
      Contact( #Mx_ET10 )
      wire#w1
      R_Coil( #StatusVacio_Apilador )
   END_RUNG
   RUNG wire#powerrail
      Contact( #Mx_ET11 )
   END_RUNG wire#w1
   RUNG wire#w1
      R_Coil( #StatusSemiLleno_Apilador )
   END_RUNG
   RUNG wire#w1
      R_Coil( #StatusLleno_Apilador )
   END_RUNG
   // the same network as SCL:
   IF #Mx_ET10 OR #Mx_ET11 THEN
       #StatusVacio_Apilador := FALSE;
       #StatusSemiLleno_Apilador := FALSE;
       #StatusLleno_Apilador := FALSE;
   END_IF;
END_REGION

REGION Network 89: INTERLOCK MAQUINA - MEMORIA >>> En Reposo la Maquina
   RUNG wire#powerrail
      Contact( #STAT_PasarReposo )
      Contact( #FinMovimiento_Apilador )
      S_SR(operand := #Memoria_EnReposoMaquina, r1 := wire#w2)
   END_RUNG
   RUNG wire#powerrail
      Contact( #Mx_ET50 )
      wire#w1
      I_Contact( #Mx_ET02 )
   END_RUNG wire#w2
   RUNG wire#powerrail
      Contact( #Mx_ET210 )
   END_RUNG wire#w1
   RUNG wire#powerrail
      Contact( #Mx_ET12 )
   END_RUNG wire#w1
   // the same network as SCL:
   IF #STAT_PasarReposo AND #FinMovimiento_Apilador THEN
       #Memoria_EnReposoMaquina := TRUE;   // SR flip-flop
   END_IF;
   IF (#Mx_ET50 OR #Mx_ET210 OR #Mx_ET12) AND NOT #Mx_ET02 THEN #Memoria_EnReposoMaquina := FALSE; END_IF;
END_REGION

REGION Network 90: INTERLOCK MAQUINA - ORDEN >>> Pasar a Reposo
   RUNG wire#powerrail
      Contact( #Mx_ET01 )
      I_Contact( #pHsMx_1 )
      I_Contact( #pHsMx_2 )
      wire#w1
      Contact( #AVTF_MAnt_Mx )
      wire#w2
      I_Contact( #pHsMx_Carretilla )
      wire#w3
      Coil( #PasarReposo_Apilador )
   END_RUNG
   RUNG wire#w1
      Contact( #AVTF_MSig_Mx )
   END_RUNG wire#w2
   RUNG wire#w1
      I_Contact( #Memoria_EnReposoMaquina )
      I_Contact( #AVTF_MAnt_Mx )
      I_Contact( #AVTF_MSig_Mx )
   END_RUNG wire#w2
   RUNG wire#powerrail
      Contact( #Mx_ET02 )
      I_Contact( #Memoria_EnReposoMaquina )
   END_RUNG wire#w2
   RUNG wire#powerrail
      Contact( #Mx_ET250 )
   END_RUNG wire#w2
   RUNG wire#powerrail
      Contact( #Mx_ET52 )
   END_RUNG wire#w2
   RUNG wire#w3
      Coil( #STAT_PasarReposo )
   END_RUNG
   // the same network as SCL:
   #PasarReposo_Apilador := ((#Mx_ET01 AND NOT #pHsMx_1 AND NOT #pHsMx_2 AND (#AVTF_MAnt_Mx OR #AVTF_MSig_Mx OR (NOT #Memoria_EnReposoMaquina AND NOT #AVTF_MAnt_Mx AND NOT #AVTF_MSig_Mx))) OR (#Mx_ET02 AND NOT #Memoria_EnReposoMaquina) OR #Mx_ET250 OR #Mx_ET52) AND NOT #pHsMx_Carretilla;
   #STAT_PasarReposo := #PasarReposo_Apilador;
END_REGION

REGION Network 91: INTERLOCK MAQUINA - ORDEN >>> Coger Pila
   RUNG wire#powerrail
      Contact( #Mx_ET210 )
      I_Contact( #STAT_PasarReposo )
      I_Contact( #pHsMx_Carretilla )
      wire#w1
      Coil( #CogerPila_Apilador )
   END_RUNG
   RUNG wire#w1
      Coil( #STAT_CogerPila )
   END_RUNG
   // the same network as SCL:
   #CogerPila_Apilador := #Mx_ET210 AND NOT #STAT_PasarReposo AND NOT #pHsMx_Carretilla;
   #STAT_CogerPila := #CogerPila_Apilador;
END_REGION

REGION Network 92: INTERLOCK MAQUINA - ORDEN >>> Dispensar Paleta
   RUNG wire#powerrail
      Contact( #Mx_ET02 )
      wire#w1
      Contact( #OrdSal_Paleta_Mx_MSig )
      wire#w2
      Contact( #Memoria_EnReposoMaquina )
      I_Contact( #STAT_PasarReposo )
      I_Contact( #STAT_CogerPila )
      I_Contact( #pHsMx_Carretilla )
      wire#w3
      Coil( #DispensarPaleta_Apilador )
   END_RUNG
   RUNG wire#w1
      Contact( #OrdSal_Paleta_Mx_MAnt )
   END_RUNG wire#w2
   RUNG wire#w3
      Coil( #STAT_DispensarPaleta )
   END_RUNG
   // the same network as SCL:
   #DispensarPaleta_Apilador := #Mx_ET02 AND (#OrdSal_Paleta_Mx_MSig OR #OrdSal_Paleta_Mx_MAnt) AND #Memoria_EnReposoMaquina AND NOT #STAT_PasarReposo AND NOT #STAT_CogerPila AND NOT #pHsMx_Carretilla;
   #STAT_DispensarPaleta := #DispensarPaleta_Apilador;
END_REGION

REGION Network 93: INTERLOCK MAQUINA - ORDEN >>> Dispensar Pila
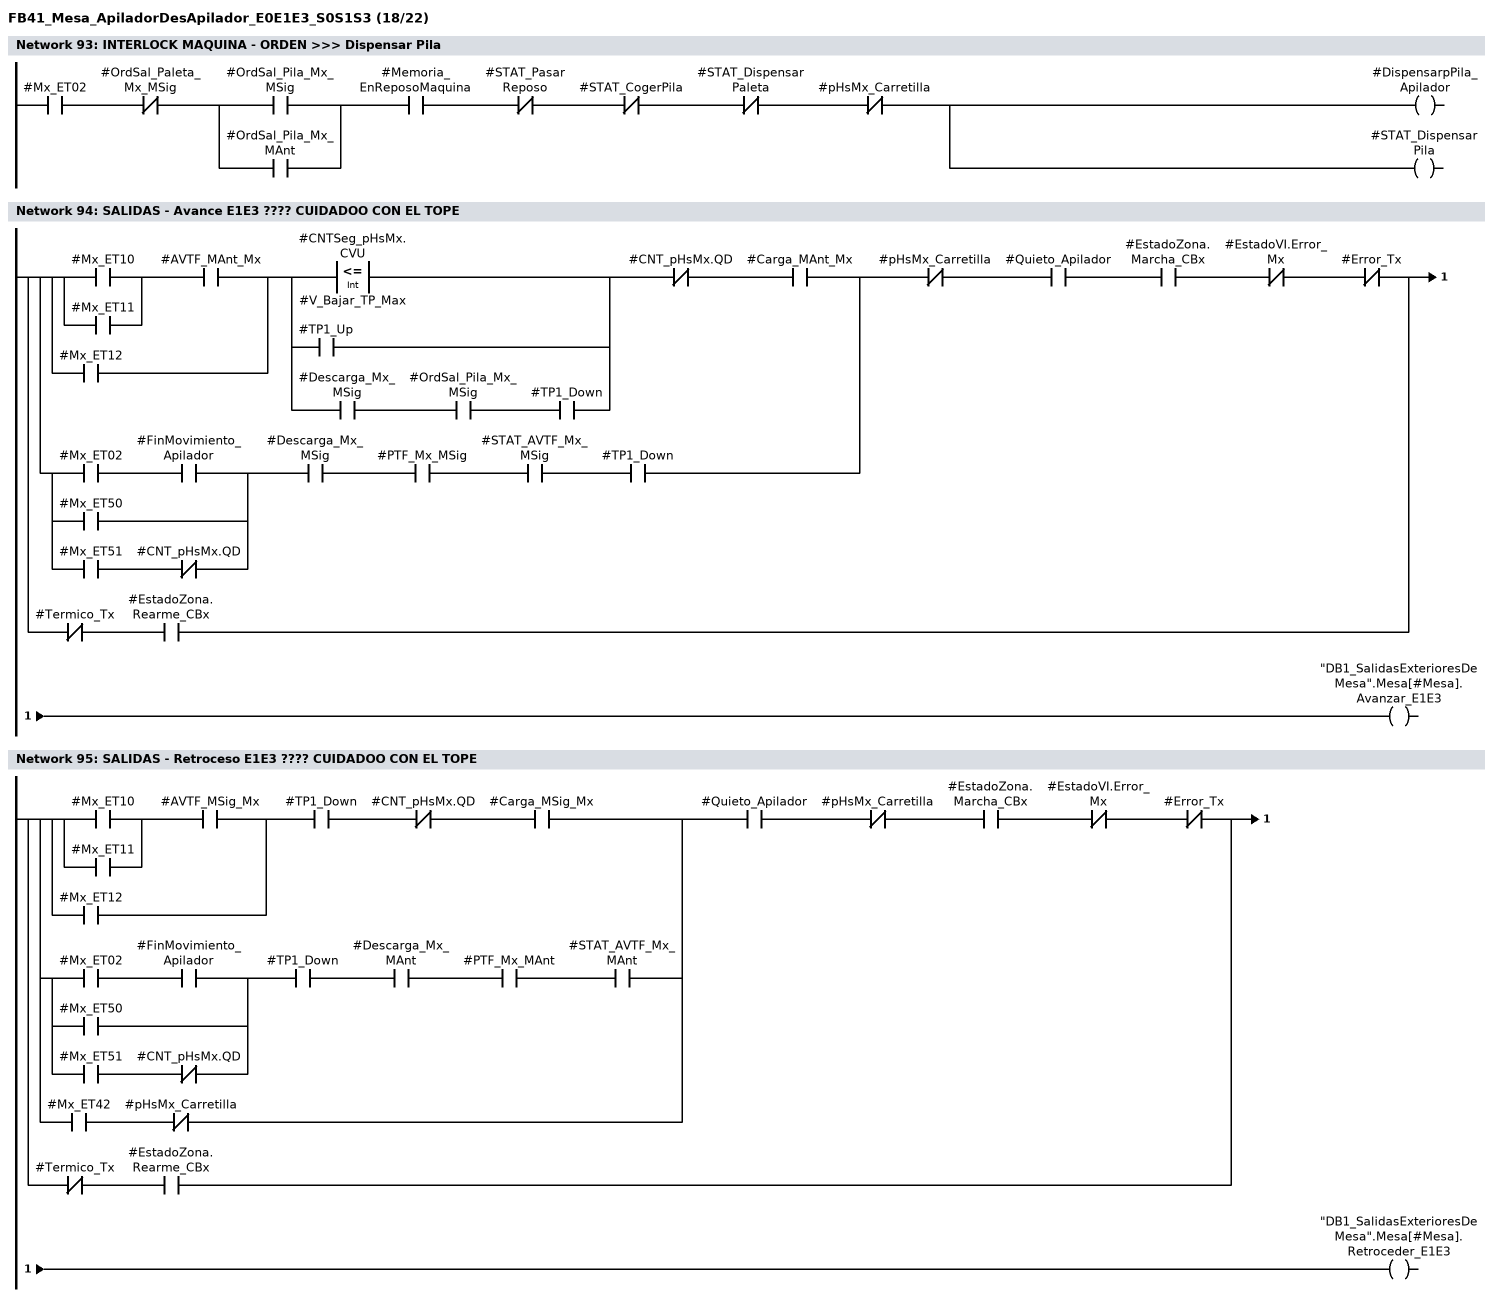
   RUNG wire#powerrail
      Contact( #Mx_ET02 )
      I_Contact( #OrdSal_Paleta_Mx_MSig )
      wire#w1
      Contact( #OrdSal_Pila_Mx_MSig )
      wire#w2
      Contact( #Memoria_EnReposoMaquina )
      I_Contact( #STAT_PasarReposo )
      I_Contact( #STAT_CogerPila )
      I_Contact( #STAT_DispensarPaleta )
      I_Contact( #pHsMx_Carretilla )
      wire#w3
      Coil( #DispensarpPila_Apilador )
   END_RUNG
   RUNG wire#w1
      Contact( #OrdSal_Pila_Mx_MAnt )
   END_RUNG wire#w2
   RUNG wire#w3
      Coil( #STAT_DispensarPila )
   END_RUNG
   // the same network as SCL:
   #DispensarpPila_Apilador := #Mx_ET02 AND NOT #OrdSal_Paleta_Mx_MSig AND (#OrdSal_Pila_Mx_MSig OR #OrdSal_Pila_Mx_MAnt) AND #Memoria_EnReposoMaquina AND NOT #STAT_PasarReposo AND NOT #STAT_CogerPila AND NOT #STAT_DispensarPaleta AND NOT #pHsMx_Carretilla;
   #STAT_DispensarPila := #DispensarpPila_Apilador;
END_REGION

REGION Network 94: SALIDAS - Avance E1E3 ???? CUIDADOO CON EL TOPE
   RUNG wire#powerrail
      Contact( #Mx_ET10 )
      wire#w1
      Contact( #AVTF_MAnt_Mx )
      wire#w2
      { S7_Templates := "SrcType := Int" } LE_Contact(in1 := #CNTSeg_pHsMx.CVU, in2 := #V_Bajar_TP_Max)
      wire#w3
      I_Contact( #CNT_pHsMx.QD )
      Contact( #Carga_MAnt_Mx )
      wire#w4
      I_Contact( #pHsMx_Carretilla )
      Contact( #Quieto_Apilador )
      Contact( #EstadoZona.Marcha_CBx )
      I_Contact( #EstadoVI.Error_Mx )
      I_Contact( #Error_Tx )
      wire#w6
      Coil( "DB1_SalidasExterioresDeMesa".Mesa[#Mesa].Avanzar_E1E3 )
   END_RUNG
   RUNG wire#powerrail
      Contact( #Mx_ET11 )
   END_RUNG wire#w1
   RUNG wire#powerrail
      Contact( #Mx_ET12 )
   END_RUNG wire#w2
   RUNG wire#w2
      Contact( #TP1_Up )
   END_RUNG wire#w3
   RUNG wire#w2
      Contact( #Descarga_Mx_MSig )
      Contact( #OrdSal_Pila_Mx_MSig )
      Contact( #TP1_Down )
   END_RUNG wire#w3
   RUNG wire#powerrail
      Contact( #Mx_ET02 )
      Contact( #FinMovimiento_Apilador )
      wire#w5
      Contact( #Descarga_Mx_MSig )
      Contact( #PTF_Mx_MSig )
      Contact( #STAT_AVTF_Mx_MSig )
      Contact( #TP1_Down )
   END_RUNG wire#w4
   RUNG wire#powerrail
      Contact( #Mx_ET50 )
   END_RUNG wire#w5
   RUNG wire#powerrail
      Contact( #Mx_ET51 )
      I_Contact( #CNT_pHsMx.QD )
   END_RUNG wire#w5
   RUNG wire#powerrail
      I_Contact( #Termico_Tx )
      Contact( #EstadoZona.Rearme_CBx )
   END_RUNG wire#w6
   // the same network as SCL:
   "DB1_SalidasExterioresDeMesa".Mesa[#Mesa].Avanzar_E1E3 := ((((((#Mx_ET10 OR #Mx_ET11) AND #AVTF_MAnt_Mx) OR #Mx_ET12) AND ((#CNTSeg_pHsMx.CVU <= #V_Bajar_TP_Max) OR #TP1_Up OR (#Descarga_Mx_MSig AND #OrdSal_Pila_Mx_MSig AND #TP1_Down)) AND NOT #CNT_pHsMx.QD AND #Carga_MAnt_Mx) OR (((#Mx_ET02 AND #FinMovimiento_Apilador) OR #Mx_ET50 OR (#Mx_ET51 AND NOT #CNT_pHsMx.QD)) AND #Descarga_Mx_MSig AND #PTF_Mx_MSig AND #STAT_AVTF_Mx_MSig AND #TP1_Down)) AND NOT #pHsMx_Carretilla AND #Quieto_Apilador AND #EstadoZona.Marcha_CBx AND NOT #EstadoVI.Error_Mx AND NOT #Error_Tx) OR (NOT #Termico_Tx AND #EstadoZona.Rearme_CBx);
END_REGION

REGION Network 95: SALIDAS - Retroceso E1E3 ???? CUIDADOO CON EL TOPE
   RUNG wire#powerrail
      Contact( #Mx_ET10 )
      wire#w1
      Contact( #AVTF_MSig_Mx )
      wire#w2
      Contact( #TP1_Down )
      I_Contact( #CNT_pHsMx.QD )
      Contact( #Carga_MSig_Mx )
      wire#w3
      Contact( #Quieto_Apilador )
      I_Contact( #pHsMx_Carretilla )
      Contact( #EstadoZona.Marcha_CBx )
      I_Contact( #EstadoVI.Error_Mx )
      I_Contact( #Error_Tx )
      wire#w5
      Coil( "DB1_SalidasExterioresDeMesa".Mesa[#Mesa].Retroceder_E1E3 )
   END_RUNG
   RUNG wire#powerrail
      Contact( #Mx_ET11 )
   END_RUNG wire#w1
   RUNG wire#powerrail
      Contact( #Mx_ET12 )
   END_RUNG wire#w2
   RUNG wire#powerrail
      Contact( #Mx_ET02 )
      Contact( #FinMovimiento_Apilador )
      wire#w4
      Contact( #TP1_Down )
      Contact( #Descarga_Mx_MAnt )
      Contact( #PTF_Mx_MAnt )
      Contact( #STAT_AVTF_Mx_MAnt )
   END_RUNG wire#w3
   RUNG wire#powerrail
      Contact( #Mx_ET50 )
   END_RUNG wire#w4
   RUNG wire#powerrail
      Contact( #Mx_ET51 )
      I_Contact( #CNT_pHsMx.QD )
   END_RUNG wire#w4
   RUNG wire#powerrail
      Contact( #Mx_ET42 )
      I_Contact( #pHsMx_Carretilla )
   END_RUNG wire#w3
   RUNG wire#powerrail
      I_Contact( #Termico_Tx )
      Contact( #EstadoZona.Rearme_CBx )
   END_RUNG wire#w5
   // the same network as SCL:
   "DB1_SalidasExterioresDeMesa".Mesa[#Mesa].Retroceder_E1E3 := ((((((#Mx_ET10 OR #Mx_ET11) AND #AVTF_MSig_Mx) OR #Mx_ET12) AND #TP1_Down AND NOT #CNT_pHsMx.QD AND #Carga_MSig_Mx) OR (((#Mx_ET02 AND #FinMovimiento_Apilador) OR #Mx_ET50 OR (#Mx_ET51 AND NOT #CNT_pHsMx.QD)) AND #TP1_Down AND #Descarga_Mx_MAnt AND #PTF_Mx_MAnt AND #STAT_AVTF_Mx_MAnt) OR (#Mx_ET42 AND NOT #pHsMx_Carretilla)) AND #Quieto_Apilador AND NOT #pHsMx_Carretilla AND #EstadoZona.Marcha_CBx AND NOT #EstadoVI.Error_Mx AND NOT #Error_Tx) OR (NOT #Termico_Tx AND #EstadoZona.Rearme_CBx);
END_REGION

REGION Network 96: SALIDAS - Parar Tx
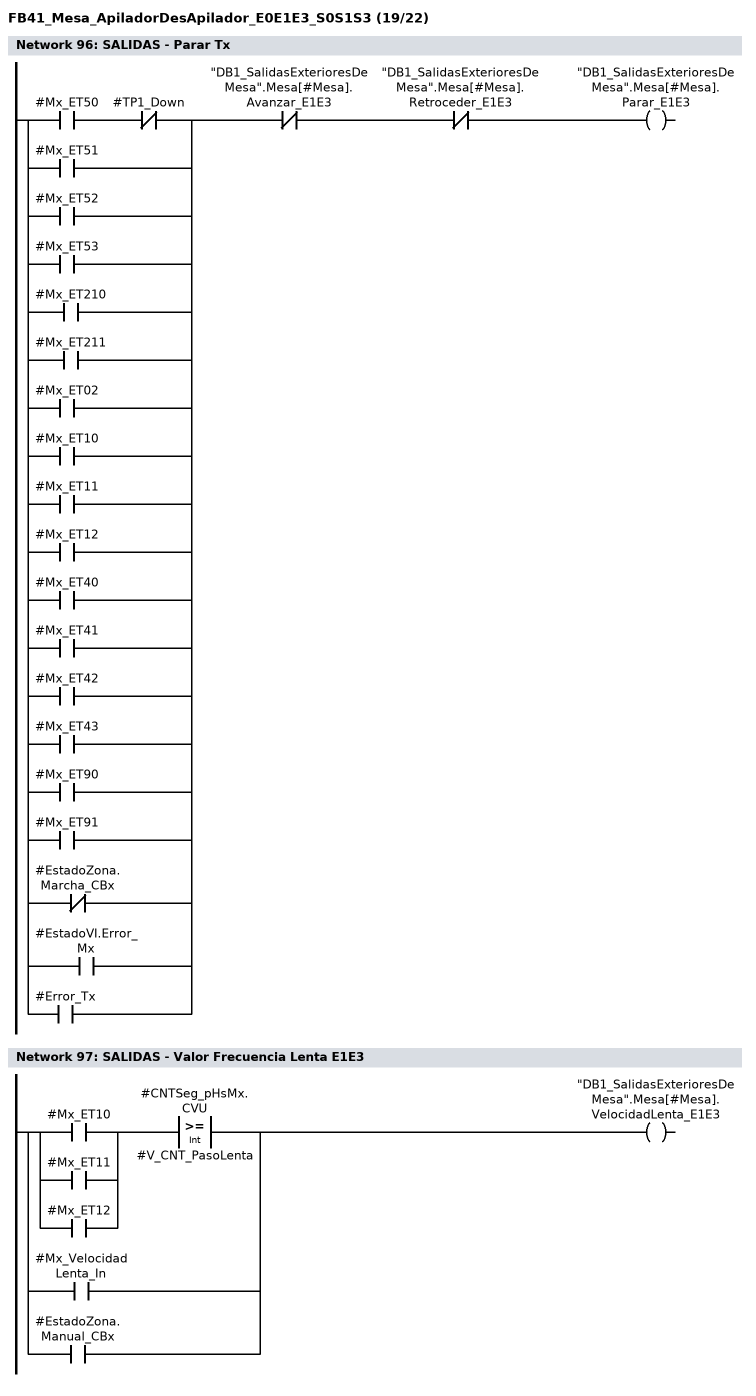
   RUNG wire#powerrail
      Contact( #Mx_ET50 )
      I_Contact( #TP1_Down )
      wire#w1
      I_Contact( "DB1_SalidasExterioresDeMesa".Mesa[#Mesa].Avanzar_E1E3 )
      I_Contact( "DB1_SalidasExterioresDeMesa".Mesa[#Mesa].Retroceder_E1E3 )
      Coil( "DB1_SalidasExterioresDeMesa".Mesa[#Mesa].Parar_E1E3 )
   END_RUNG
   RUNG wire#powerrail
      Contact( #Mx_ET51 )
   END_RUNG wire#w1
   RUNG wire#powerrail
      Contact( #Mx_ET52 )
   END_RUNG wire#w1
   RUNG wire#powerrail
      Contact( #Mx_ET53 )
   END_RUNG wire#w1
   RUNG wire#powerrail
      Contact( #Mx_ET210 )
   END_RUNG wire#w1
   RUNG wire#powerrail
      Contact( #Mx_ET211 )
   END_RUNG wire#w1
   RUNG wire#powerrail
      Contact( #Mx_ET02 )
   END_RUNG wire#w1
   RUNG wire#powerrail
      Contact( #Mx_ET10 )
   END_RUNG wire#w1
   RUNG wire#powerrail
      Contact( #Mx_ET11 )
   END_RUNG wire#w1
   RUNG wire#powerrail
      Contact( #Mx_ET12 )
   END_RUNG wire#w1
   RUNG wire#powerrail
      Contact( #Mx_ET40 )
   END_RUNG wire#w1
   RUNG wire#powerrail
      Contact( #Mx_ET41 )
   END_RUNG wire#w1
   RUNG wire#powerrail
      Contact( #Mx_ET42 )
   END_RUNG wire#w1
   RUNG wire#powerrail
      Contact( #Mx_ET43 )
   END_RUNG wire#w1
   RUNG wire#powerrail
      Contact( #Mx_ET90 )
   END_RUNG wire#w1
   RUNG wire#powerrail
      Contact( #Mx_ET91 )
   END_RUNG wire#w1
   RUNG wire#powerrail
      I_Contact( #EstadoZona.Marcha_CBx )
   END_RUNG wire#w1
   RUNG wire#powerrail
      Contact( #EstadoVI.Error_Mx )
   END_RUNG wire#w1
   RUNG wire#powerrail
      Contact( #Error_Tx )
   END_RUNG wire#w1
   // the same network as SCL:
   "DB1_SalidasExterioresDeMesa".Mesa[#Mesa].Parar_E1E3 := ((#Mx_ET50 AND NOT #TP1_Down) OR #Mx_ET51 OR #Mx_ET52 OR #Mx_ET53 OR #Mx_ET210 OR #Mx_ET211 OR #Mx_ET02 OR #Mx_ET10 OR #Mx_ET11 OR #Mx_ET12 OR #Mx_ET40 OR #Mx_ET41 OR #Mx_ET42 OR #Mx_ET43 OR #Mx_ET90 OR #Mx_ET91 OR NOT #EstadoZona.Marcha_CBx OR #EstadoVI.Error_Mx OR #Error_Tx) AND NOT "DB1_SalidasExterioresDeMesa".Mesa[#Mesa].Avanzar_E1E3 AND NOT "DB1_SalidasExterioresDeMesa".Mesa[#Mesa].Retroceder_E1E3;
END_REGION

REGION Network 97: SALIDAS - Valor Frecuencia Lenta E1E3
   RUNG wire#powerrail
      Contact( #Mx_ET10 )
      wire#w1
      { S7_Templates := "SrcType := Int" } GE_Contact(in1 := #CNTSeg_pHsMx.CVU, in2 := #V_CNT_PasoLenta)
      wire#w2
      Coil( "DB1_SalidasExterioresDeMesa".Mesa[#Mesa].VelocidadLenta_E1E3 )
   END_RUNG
   RUNG wire#powerrail
      Contact( #Mx_ET11 )
   END_RUNG wire#w1
   RUNG wire#powerrail
      Contact( #Mx_ET12 )
   END_RUNG wire#w1
   RUNG wire#powerrail
      Contact( #Mx_VelocidadLenta_In )
   END_RUNG wire#w2
   RUNG wire#powerrail
      Contact( #EstadoZona.Manual_CBx )
   END_RUNG wire#w2
   // the same network as SCL:
   "DB1_SalidasExterioresDeMesa".Mesa[#Mesa].VelocidadLenta_E1E3 := ((#Mx_ET10 OR #Mx_ET11 OR #Mx_ET12) AND (#CNTSeg_pHsMx.CVU >= #V_CNT_PasoLenta)) OR #Mx_VelocidadLenta_In OR #EstadoZona.Manual_CBx;
END_REGION

REGION Network 98: SALIDAS - Bajar Tope TP1 NOTA: Tope E1 >> S3 ???? CUIDADOO CON EL TOPE
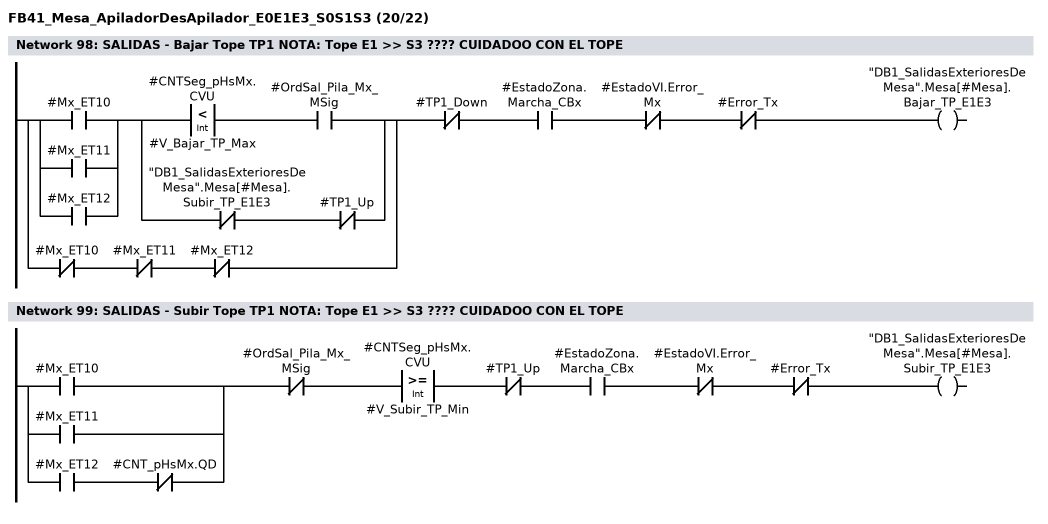
   RUNG wire#powerrail
      Contact( #Mx_ET10 )
      wire#w1
      { S7_Templates := "SrcType := Int" } LT_Contact(in1 := #CNTSeg_pHsMx.CVU, in2 := #V_Bajar_TP_Max)
      Contact( #OrdSal_Pila_Mx_MSig )
      wire#w2
      I_Contact( #TP1_Down )
      Contact( #EstadoZona.Marcha_CBx )
      I_Contact( #EstadoVI.Error_Mx )
      I_Contact( #Error_Tx )
      Coil( "DB1_SalidasExterioresDeMesa".Mesa[#Mesa].Bajar_TP_E1E3 )
   END_RUNG
   RUNG wire#powerrail
      Contact( #Mx_ET11 )
   END_RUNG wire#w1
   RUNG wire#powerrail
      Contact( #Mx_ET12 )
   END_RUNG wire#w1
   RUNG wire#w1
      I_Contact( "DB1_SalidasExterioresDeMesa".Mesa[#Mesa].Subir_TP_E1E3 )
      I_Contact( #TP1_Up )
   END_RUNG wire#w2
   RUNG wire#powerrail
      I_Contact( #Mx_ET10 )
      I_Contact( #Mx_ET11 )
      I_Contact( #Mx_ET12 )
   END_RUNG wire#w2
   // the same network as SCL:
   "DB1_SalidasExterioresDeMesa".Mesa[#Mesa].Bajar_TP_E1E3 := (((#Mx_ET10 OR #Mx_ET11 OR #Mx_ET12) AND (((#CNTSeg_pHsMx.CVU < #V_Bajar_TP_Max) AND #OrdSal_Pila_Mx_MSig) OR (NOT "DB1_SalidasExterioresDeMesa".Mesa[#Mesa].Subir_TP_E1E3 AND NOT #TP1_Up))) OR (NOT #Mx_ET10 AND NOT #Mx_ET11 AND NOT #Mx_ET12)) AND NOT #TP1_Down AND #EstadoZona.Marcha_CBx AND NOT #EstadoVI.Error_Mx AND NOT #Error_Tx;
END_REGION

REGION Network 99: SALIDAS - Subir Tope TP1 NOTA: Tope E1 >> S3 ???? CUIDADOO CON EL TOPE
   RUNG wire#powerrail
      Contact( #Mx_ET10 )
      wire#w1
      I_Contact( #OrdSal_Pila_Mx_MSig )
      { S7_Templates := "SrcType := Int" } GE_Contact(in1 := #CNTSeg_pHsMx.CVU, in2 := #V_Subir_TP_Min)
      I_Contact( #TP1_Up )
      Contact( #EstadoZona.Marcha_CBx )
      I_Contact( #EstadoVI.Error_Mx )
      I_Contact( #Error_Tx )
      Coil( "DB1_SalidasExterioresDeMesa".Mesa[#Mesa].Subir_TP_E1E3 )
   END_RUNG
   RUNG wire#powerrail
      Contact( #Mx_ET11 )
   END_RUNG wire#w1
   RUNG wire#powerrail
      Contact( #Mx_ET12 )
      I_Contact( #CNT_pHsMx.QD )
   END_RUNG wire#w1
   // the same network as SCL:
   "DB1_SalidasExterioresDeMesa".Mesa[#Mesa].Subir_TP_E1E3 := (#Mx_ET10 OR #Mx_ET11 OR (#Mx_ET12 AND NOT #CNT_pHsMx.QD)) AND NOT #OrdSal_Pila_Mx_MSig AND (#CNTSeg_pHsMx.CVU >= #V_Subir_TP_Min) AND NOT #TP1_Up AND #EstadoZona.Marcha_CBx AND NOT #EstadoVI.Error_Mx AND NOT #Error_Tx;
END_REGION

REGION Network 100: ESTADOS DE LA MESA
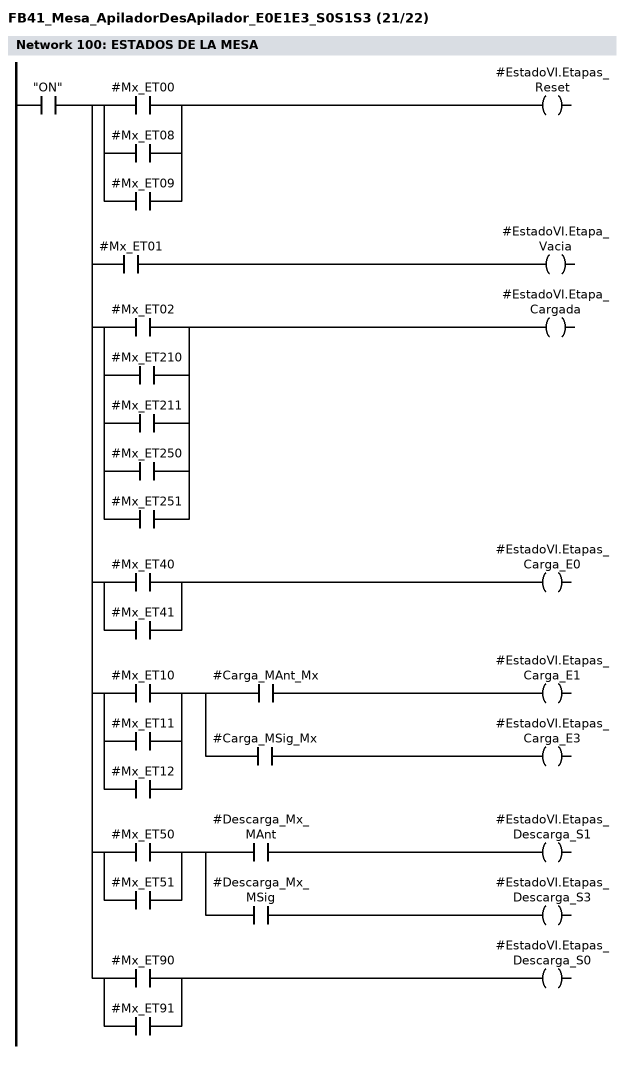
   RUNG wire#powerrail
      Contact( "ON" )
      wire#w1
      Contact( #Mx_ET00 )
      wire#w2
      Coil( #EstadoVI.Etapas_Reset )
   END_RUNG
   RUNG wire#w1
      Contact( #Mx_ET08 )
   END_RUNG wire#w2
   RUNG wire#w1
      Contact( #Mx_ET09 )
   END_RUNG wire#w2
   RUNG wire#w1
      Contact( #Mx_ET01 )
      Coil( #EstadoVI.Etapa_Vacia )
   END_RUNG
   RUNG wire#w1
      Contact( #Mx_ET02 )
      wire#w3
      Coil( #EstadoVI.Etapa_Cargada )
   END_RUNG
   RUNG wire#w1
      Contact( #Mx_ET210 )
   END_RUNG wire#w3
   RUNG wire#w1
      Contact( #Mx_ET211 )
   END_RUNG wire#w3
   RUNG wire#w1
      Contact( #Mx_ET250 )
   END_RUNG wire#w3
   RUNG wire#w1
      Contact( #Mx_ET251 )
   END_RUNG wire#w3
   RUNG wire#w1
      Contact( #Mx_ET40 )
      wire#w4
      Coil( #EstadoVI.Etapas_Carga_E0 )
   END_RUNG
   RUNG wire#w1
      Contact( #Mx_ET41 )
   END_RUNG wire#w4
   RUNG wire#w1
      Contact( #Mx_ET10 )
      wire#w5
      Contact( #Carga_MAnt_Mx )
      Coil( #EstadoVI.Etapas_Carga_E1 )
   END_RUNG
   RUNG wire#w1
      Contact( #Mx_ET11 )
   END_RUNG wire#w5
   RUNG wire#w1
      Contact( #Mx_ET12 )
   END_RUNG wire#w5
   RUNG wire#w5
      Contact( #Carga_MSig_Mx )
      Coil( #EstadoVI.Etapas_Carga_E3 )
   END_RUNG
   RUNG wire#w1
      Contact( #Mx_ET50 )
      wire#w6
      Contact( #Descarga_Mx_MAnt )
      Coil( #EstadoVI.Etapas_Descarga_S1 )
   END_RUNG
   RUNG wire#w1
      Contact( #Mx_ET51 )
   END_RUNG wire#w6
   RUNG wire#w6
      Contact( #Descarga_Mx_MSig )
      Coil( #EstadoVI.Etapas_Descarga_S3 )
   END_RUNG
   RUNG wire#w1
      Contact( #Mx_ET90 )
      wire#w7
      Coil( #EstadoVI.Etapas_Descarga_S0 )
   END_RUNG
   RUNG wire#w1
      Contact( #Mx_ET91 )
   END_RUNG wire#w7
   // the same network as SCL:
   #EstadoVI.Etapas_Reset := "ON" AND (#Mx_ET00 OR #Mx_ET08 OR #Mx_ET09);
   #EstadoVI.Etapa_Vacia := "ON" AND #Mx_ET01;
   #EstadoVI.Etapa_Cargada := "ON" AND (#Mx_ET02 OR #Mx_ET210 OR #Mx_ET211 OR #Mx_ET250 OR #Mx_ET251);
   #EstadoVI.Etapas_Carga_E0 := "ON" AND (#Mx_ET40 OR #Mx_ET41);
   #_w1 := "ON" AND (#Mx_ET10 OR #Mx_ET11 OR #Mx_ET12);
   #EstadoVI.Etapas_Carga_E1 := #_w1 AND #Carga_MAnt_Mx;
   #EstadoVI.Etapas_Carga_E3 := #_w1 AND #Carga_MSig_Mx;
   #_w2 := "ON" AND (#Mx_ET50 OR #Mx_ET51);
   #EstadoVI.Etapas_Descarga_S1 := #_w2 AND #Descarga_Mx_MAnt;
   #EstadoVI.Etapas_Descarga_S3 := #_w2 AND #Descarga_Mx_MSig;
   #EstadoVI.Etapas_Descarga_S0 := "ON" AND (#Mx_ET90 OR #Mx_ET91);
END_REGION

REGION Network 101: ENTRADAS DE LA MESA
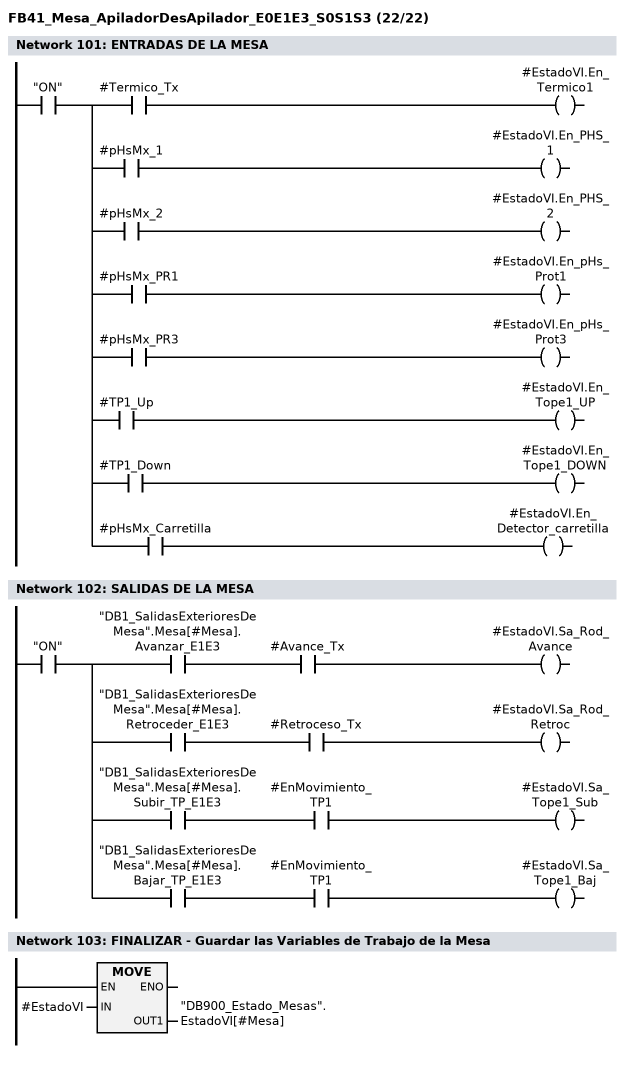
   RUNG wire#powerrail
      Contact( "ON" )
      wire#w1
      Contact( #Termico_Tx )
      Coil( #EstadoVI.En_Termico1 )
   END_RUNG
   RUNG wire#w1
      Contact( #pHsMx_1 )
      Coil( #EstadoVI.En_PHS_1 )
   END_RUNG
   RUNG wire#w1
      Contact( #pHsMx_2 )
      Coil( #EstadoVI.En_PHS_2 )
   END_RUNG
   RUNG wire#w1
      Contact( #pHsMx_PR1 )
      Coil( #EstadoVI.En_pHs_Prot1 )
   END_RUNG
   RUNG wire#w1
      Contact( #pHsMx_PR3 )
      Coil( #EstadoVI.En_pHs_Prot3 )
   END_RUNG
   RUNG wire#w1
      Contact( #TP1_Up )
      Coil( #EstadoVI.En_Tope1_UP )
   END_RUNG
   RUNG wire#w1
      Contact( #TP1_Down )
      Coil( #EstadoVI.En_Tope1_DOWN )
   END_RUNG
   RUNG wire#w1
      Contact( #pHsMx_Carretilla )
      Coil( #EstadoVI.En_Detector_carretilla )
   END_RUNG
   // the same network as SCL:
   #EstadoVI.En_Termico1 := "ON" AND #Termico_Tx;
   #EstadoVI.En_PHS_1 := "ON" AND #pHsMx_1;
   #EstadoVI.En_PHS_2 := "ON" AND #pHsMx_2;
   #EstadoVI.En_pHs_Prot1 := "ON" AND #pHsMx_PR1;
   #EstadoVI.En_pHs_Prot3 := "ON" AND #pHsMx_PR3;
   #EstadoVI.En_Tope1_UP := "ON" AND #TP1_Up;
   #EstadoVI.En_Tope1_DOWN := "ON" AND #TP1_Down;
   #EstadoVI.En_Detector_carretilla := "ON" AND #pHsMx_Carretilla;
END_REGION

REGION Network 102: SALIDAS DE LA MESA
   RUNG wire#powerrail
      Contact( "ON" )
      wire#w1
      Contact( "DB1_SalidasExterioresDeMesa".Mesa[#Mesa].Avanzar_E1E3 )
      Contact( #Avance_Tx )
      Coil( #EstadoVI.Sa_Rod_Avance )
   END_RUNG
   RUNG wire#w1
      Contact( "DB1_SalidasExterioresDeMesa".Mesa[#Mesa].Retroceder_E1E3 )
      Contact( #Retroceso_Tx )
      Coil( #EstadoVI.Sa_Rod_Retroc )
   END_RUNG
   RUNG wire#w1
      Contact( "DB1_SalidasExterioresDeMesa".Mesa[#Mesa].Subir_TP_E1E3 )
      Contact( #EnMovimiento_TP1 )
      Coil( #EstadoVI.Sa_Tope1_Sub )
   END_RUNG
   RUNG wire#w1
      Contact( "DB1_SalidasExterioresDeMesa".Mesa[#Mesa].Bajar_TP_E1E3 )
      Contact( #EnMovimiento_TP1 )
      Coil( #EstadoVI.Sa_Tope1_Baj )
   END_RUNG
   // the same network as SCL:
   #EstadoVI.Sa_Rod_Avance := "ON" AND "DB1_SalidasExterioresDeMesa".Mesa[#Mesa].Avanzar_E1E3 AND #Avance_Tx;
   #EstadoVI.Sa_Rod_Retroc := "ON" AND "DB1_SalidasExterioresDeMesa".Mesa[#Mesa].Retroceder_E1E3 AND #Retroceso_Tx;
   #EstadoVI.Sa_Tope1_Sub := "ON" AND "DB1_SalidasExterioresDeMesa".Mesa[#Mesa].Subir_TP_E1E3 AND #EnMovimiento_TP1;
   #EstadoVI.Sa_Tope1_Baj := "ON" AND "DB1_SalidasExterioresDeMesa".Mesa[#Mesa].Bajar_TP_E1E3 AND #EnMovimiento_TP1;
END_REGION

